REGION Network 14: ACTIVATE HANDWHEEL / ACTIVATE HANDWHEEL 1
   RUNG wire#powerrail
      I_Contact( "DB2001_MODES_GENERAL".MG1.INCREMENTAL."1_MICRA_SELECTED" )
      I_Contact( "DB2001_MODES_GENERAL".MG1.INCREMENTAL."10_MICRA_SELECTED" )
      I_Contact( "DB2001_MODES_GENERAL".MG1.INCREMENTAL."100_MICRA_SELECTED" )
      I_Contact( "DB2001_MODES_GENERAL".MG1.INCREMENTAL."1000_MICRA_SELECTED" )
      Not()
      Contact( #SP.SELECTED )
      Contact( "DB2001_MODES_GENERAL".MG1.INCREMENTAL.INCREMENTAL_MODE_SELECTED )
      Coil( #SpindleDB.A_HW1 )
   END_RUNG
   // the same network as SCL:
   #SpindleDB.A_HW1 := NOT (NOT "DB2001_MODES_GENERAL".MG1.INCREMENTAL."1_MICRA_SELECTED" AND NOT "DB2001_MODES_GENERAL".MG1.INCREMENTAL."10_MICRA_SELECTED" AND NOT "DB2001_MODES_GENERAL".MG1.INCREMENTAL."100_MICRA_SELECTED" AND NOT "DB2001_MODES_GENERAL".MG1.INCREMENTAL."1000_MICRA_SELECTED") AND #SP.SELECTED AND "DB2001_MODES_GENERAL".MG1.INCREMENTAL.INCREMENTAL_MODE_SELECTED;
END_REGION

REGION Network 15: SPINDLE INCREMENTAL MODE SELECTED
   RUNG wire#powerrail
      I_Contact( #SpindleDB.A_INC1 )
      I_Contact( #SpindleDB.A_INC10 )
      I_Contact( #SpindleDB.A_INC100 )
      I_Contact( #SpindleDB.A_INC1000 )
      Not()
      Contact( "DB2001_MODES_GENERAL".MG1.INCREMENTAL.INCREMENTAL_MODE_SELECTED )
      Coil( #SP.CONT_INCRMTL_MODE )
   END_RUNG
   // the same network as SCL:
   #SP.CONT_INCRMTL_MODE := NOT (NOT #SpindleDB.A_INC1 AND NOT #SpindleDB.A_INC10 AND NOT #SpindleDB.A_INC100 AND NOT #SpindleDB.A_INC1000) AND "DB2001_MODES_GENERAL".MG1.INCREMENTAL.INCREMENTAL_MODE_SELECTED;
END_REGION

REGION Network 16: JOG MINUS REQUEST
   RUNG wire#powerrail
      Contact( #HMI_REQ_LINE )
      Contact( "LTLP_HMIProInterfaceData".pMinus )
      wire#w1
      Coil( #SP.HMI_JOG_MINUS_RQ )
   END_RUNG
   RUNG wire#powerrail
      Contact( "DB7224_HMI_AXES".NC_AXES.SOFTKEYS.RIGHT.JOG_MINUS )
      wire#w2
      Contact( "DB2100_GENERAL".MACHINE_READY_POWER_ENABLED )
      Contact( #SP.SELECTED )
   END_RUNG wire#w1
   RUNG wire#powerrail
      Contact( "DB2122_HT10".INPUTS.JOG_MIINUS_I )
   END_RUNG wire#w2
   // the same network as SCL:
   #SP.HMI_JOG_MINUS_RQ := (#HMI_REQ_LINE AND "LTLP_HMIProInterfaceData".pMinus) OR (("DB7224_HMI_AXES".NC_AXES.SOFTKEYS.RIGHT.JOG_MINUS OR "DB2122_HT10".INPUTS.JOG_MIINUS_I) AND "DB2100_GENERAL".MACHINE_READY_POWER_ENABLED AND #SP.SELECTED);
END_REGION

REGION Network 17: JOG MINUS COMMAND
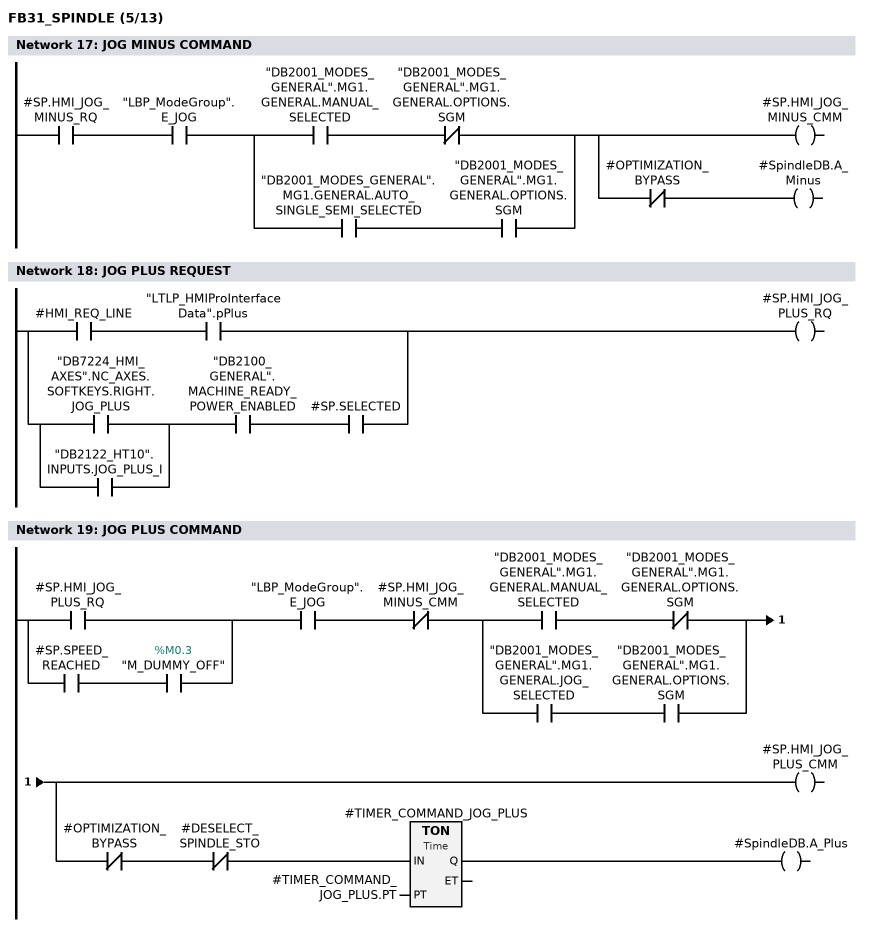
   RUNG wire#powerrail
      Contact( #SP.HMI_JOG_MINUS_RQ )
      Contact( "LBP_ModeGroup".E_JOG )
      wire#w1
      Contact( "DB2001_MODES_GENERAL".MG1.GENERAL.MANUAL_SELECTED )
      I_Contact( "DB2001_MODES_GENERAL".MG1.GENERAL.OPTIONS.SGM )
      wire#w2
      Coil( #SP.HMI_JOG_MINUS_CMM )
   END_RUNG
   RUNG wire#w1
      Contact( "DB2001_MODES_GENERAL".MG1.GENERAL.AUTO_SINGLE_SEMI_SELECTED )
      Contact( "DB2001_MODES_GENERAL".MG1.GENERAL.OPTIONS.SGM )
   END_RUNG wire#w2
   RUNG wire#w2
      I_Contact( #OPTIMIZATION_BYPASS )
      Coil( #SpindleDB.A_Minus )
   END_RUNG
   // the same network as SCL:
   #SP.HMI_JOG_MINUS_CMM := #SP.HMI_JOG_MINUS_RQ AND "LBP_ModeGroup".E_JOG AND (("DB2001_MODES_GENERAL".MG1.GENERAL.MANUAL_SELECTED AND NOT "DB2001_MODES_GENERAL".MG1.GENERAL.OPTIONS.SGM) OR ("DB2001_MODES_GENERAL".MG1.GENERAL.AUTO_SINGLE_SEMI_SELECTED AND "DB2001_MODES_GENERAL".MG1.GENERAL.OPTIONS.SGM));
   #SpindleDB.A_Minus := #SP.HMI_JOG_MINUS_CMM AND NOT #OPTIMIZATION_BYPASS;
END_REGION

REGION Network 18: JOG PLUS REQUEST
   RUNG wire#powerrail
      Contact( #HMI_REQ_LINE )
      Contact( "LTLP_HMIProInterfaceData".pPlus )
      wire#w1
      Coil( #SP.HMI_JOG_PLUS_RQ )
   END_RUNG
   RUNG wire#powerrail
      Contact( "DB7224_HMI_AXES".NC_AXES.SOFTKEYS.RIGHT.JOG_PLUS )
      wire#w2
      Contact( "DB2100_GENERAL".MACHINE_READY_POWER_ENABLED )
      Contact( #SP.SELECTED )
   END_RUNG wire#w1
   RUNG wire#powerrail
      Contact( "DB2122_HT10".INPUTS.JOG_PLUS_I )
   END_RUNG wire#w2
   // the same network as SCL:
   #SP.HMI_JOG_PLUS_RQ := (#HMI_REQ_LINE AND "LTLP_HMIProInterfaceData".pPlus) OR (("DB7224_HMI_AXES".NC_AXES.SOFTKEYS.RIGHT.JOG_PLUS OR "DB2122_HT10".INPUTS.JOG_PLUS_I) AND "DB2100_GENERAL".MACHINE_READY_POWER_ENABLED AND #SP.SELECTED);
END_REGION

REGION Network 19: JOG PLUS COMMAND
   RUNG wire#powerrail
      Contact( #SP.HMI_JOG_PLUS_RQ )
      wire#w1
      Contact( "LBP_ModeGroup".E_JOG )
      I_Contact( #SP.HMI_JOG_MINUS_CMM )
      wire#w2
      Contact( "DB2001_MODES_GENERAL".MG1.GENERAL.MANUAL_SELECTED )
      I_Contact( "DB2001_MODES_GENERAL".MG1.GENERAL.OPTIONS.SGM )
      wire#w3
      Coil( #SP.HMI_JOG_PLUS_CMM )
   END_RUNG
   RUNG wire#powerrail
      Contact( #SP.SPEED_REACHED )
      Contact( "M_DUMMY_OFF" )
   END_RUNG wire#w1
   RUNG wire#w2
      Contact( "DB2001_MODES_GENERAL".MG1.GENERAL.JOG_SELECTED )
      Contact( "DB2001_MODES_GENERAL".MG1.GENERAL.OPTIONS.SGM )
   END_RUNG wire#w3
   RUNG wire#w3
      I_Contact( #OPTIMIZATION_BYPASS )
      I_Contact( #DESELECT_SPINDLE_STO )
      { S7_Templates := "time_type := Time" } #TIMER_COMMAND_JOG_PLUS.TON(pt := #TIMER_COMMAND_JOG_PLUS.PT, et =>)
      Coil( #SpindleDB.A_Plus )
   END_RUNG
   // the same network as SCL:
   #SP.HMI_JOG_PLUS_CMM := (#SP.HMI_JOG_PLUS_RQ OR (#SP.SPEED_REACHED AND "M_DUMMY_OFF")) AND "LBP_ModeGroup".E_JOG AND NOT #SP.HMI_JOG_MINUS_CMM AND (("DB2001_MODES_GENERAL".MG1.GENERAL.MANUAL_SELECTED AND NOT "DB2001_MODES_GENERAL".MG1.GENERAL.OPTIONS.SGM) OR ("DB2001_MODES_GENERAL".MG1.GENERAL.JOG_SELECTED AND "DB2001_MODES_GENERAL".MG1.GENERAL.OPTIONS.SGM));
   #TIMER_COMMAND_JOG_PLUS(IN := #SP.HMI_JOG_PLUS_CMM AND NOT #OPTIMIZATION_BYPASS AND NOT #DESELECT_SPINDLE_STO,   // TON
                           PT := #TIMER_COMMAND_JOG_PLUS.PT);
   #SpindleDB.A_Plus := #TIMER_COMMAND_JOG_PLUS.Q;
END_REGION

REGION Network 20: OVERRIDE / FEED OVERRIDE
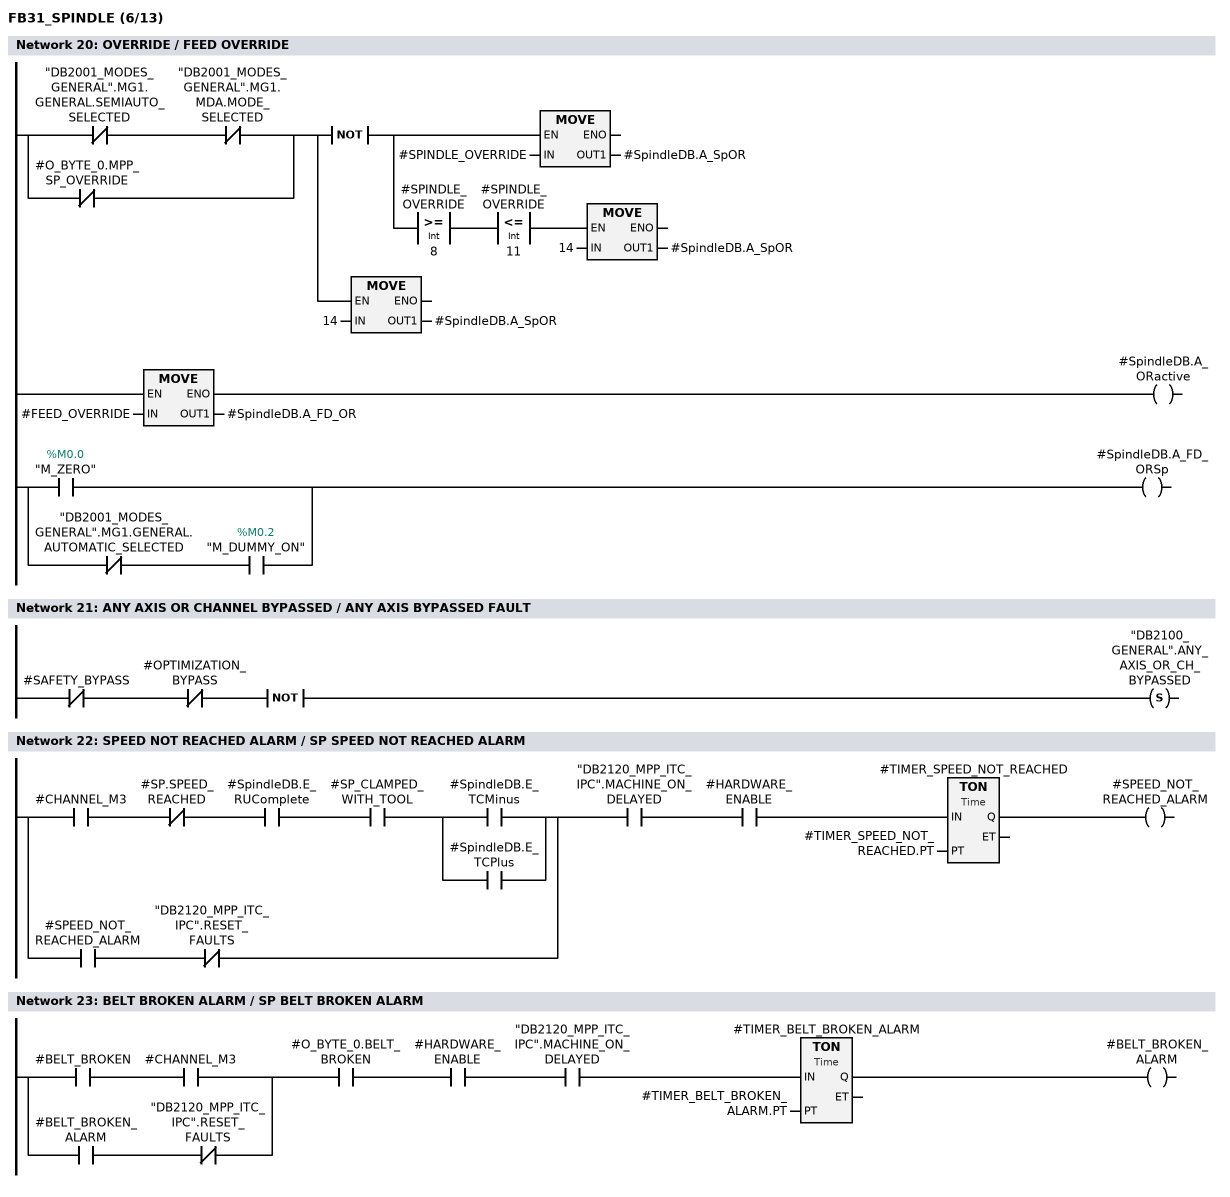
   RUNG wire#powerrail
      I_Contact( "DB2001_MODES_GENERAL".MG1.GENERAL.SEMIAUTO_SELECTED )
      I_Contact( "DB2001_MODES_GENERAL".MG1.MDA.MODE_SELECTED )
      wire#w1
      Not()
      wire#w2
      { S7_GenerateENO := "TRUE" } Move(in := #SPINDLE_OVERRIDE, out1 => #SpindleDB.A_SpOR)
   END_RUNG
   RUNG wire#powerrail
      I_Contact( #O_BYTE_0.MPP_SP_OVERRIDE )
   END_RUNG wire#w1
   RUNG wire#w2
      { S7_Templates := "SrcType := Int" } GE_Contact(in1 := #SPINDLE_OVERRIDE, in2 := 8)
      { S7_Templates := "SrcType := Int" } LE_Contact(in1 := #SPINDLE_OVERRIDE, in2 := 11)
      { S7_GenerateENO := "TRUE" } Move(in := 14, out1 => #SpindleDB.A_SpOR)
   END_RUNG
   RUNG wire#w1
      { S7_GenerateENO := "TRUE" } Move(in := 14, out1 => #SpindleDB.A_SpOR)
   END_RUNG
   RUNG wire#powerrail
      { S7_GenerateENO := "TRUE" } Move(in := #FEED_OVERRIDE, out1 => #SpindleDB.A_FD_OR)
      Coil( #SpindleDB.A_ORactive )
   END_RUNG
   RUNG wire#powerrail
      Contact( "M_ZERO" )
      wire#w3
      Coil( #SpindleDB.A_FD_ORSp )
   END_RUNG
   RUNG wire#powerrail
      I_Contact( "DB2001_MODES_GENERAL".MG1.GENERAL.AUTOMATIC_SELECTED )
      Contact( "M_DUMMY_ON" )
   END_RUNG wire#w3
   // the same network as SCL:
   // ENO of a box is taken as its EN; it also drops when the box reports an error
   #_w1 := (NOT "DB2001_MODES_GENERAL".MG1.GENERAL.SEMIAUTO_SELECTED AND NOT "DB2001_MODES_GENERAL".MG1.MDA.MODE_SELECTED) OR NOT #O_BYTE_0.MPP_SP_OVERRIDE;
   IF NOT #_w1 THEN #SpindleDB.A_SpOR := #SPINDLE_OVERRIDE; END_IF;
   IF NOT #_w1 AND (#SPINDLE_OVERRIDE >= 8) AND (#SPINDLE_OVERRIDE <= 11) THEN
       #SpindleDB.A_SpOR := 14;
   END_IF;
   IF #_w1 THEN #SpindleDB.A_SpOR := 14; END_IF;
   #SpindleDB.A_FD_OR := #FEED_OVERRIDE;
   #SpindleDB.A_ORactive := TRUE;
   #SpindleDB.A_FD_ORSp := "M_ZERO" OR (NOT "DB2001_MODES_GENERAL".MG1.GENERAL.AUTOMATIC_SELECTED AND "M_DUMMY_ON");
END_REGION

REGION Network 21: ANY AXIS OR CHANNEL BYPASSED / ANY AXIS BYPASSED FAULT
   RUNG wire#powerrail
      I_Contact( #SAFETY_BYPASS )
      I_Contact( #OPTIMIZATION_BYPASS )
      Not()
      S_Coil( "DB2100_GENERAL".ANY_AXIS_OR_CH_BYPASSED )
   END_RUNG
   // the same network as SCL:
   IF NOT (NOT #SAFETY_BYPASS AND NOT #OPTIMIZATION_BYPASS) THEN
       "DB2100_GENERAL".ANY_AXIS_OR_CH_BYPASSED := TRUE;
   END_IF;
END_REGION

REGION Network 22: SPEED NOT REACHED ALARM / SP SPEED NOT REACHED ALARM
   RUNG wire#powerrail
      Contact( #CHANNEL_M3 )
      I_Contact( #SP.SPEED_REACHED )
      Contact( #SpindleDB.E_RUComplete )
      Contact( #SP_CLAMPED_WITH_TOOL )
      wire#w1
      Contact( #SpindleDB.E_TCMinus )
      wire#w2
      Contact( "DB2120_MPP_ITC_IPC".MACHINE_ON_DELAYED )
      Contact( #HARDWARE_ENABLE )
      { S7_Templates := "time_type := Time" } #TIMER_SPEED_NOT_REACHED.TON(pt := #TIMER_SPEED_NOT_REACHED.PT, et =>)
      Coil( #SPEED_NOT_REACHED_ALARM )
   END_RUNG
   RUNG wire#w1
      Contact( #SpindleDB.E_TCPlus )
   END_RUNG wire#w2
   RUNG wire#powerrail
      Contact( #SPEED_NOT_REACHED_ALARM )
      I_Contact( "DB2120_MPP_ITC_IPC".RESET_FAULTS )
   END_RUNG wire#w2
   // the same network as SCL:
   #TIMER_SPEED_NOT_REACHED(IN := ((#CHANNEL_M3 AND NOT #SP.SPEED_REACHED AND #SpindleDB.E_RUComplete AND #SP_CLAMPED_WITH_TOOL AND (#SpindleDB.E_TCMinus OR #SpindleDB.E_TCPlus)) OR (#SPEED_NOT_REACHED_ALARM AND NOT "DB2120_MPP_ITC_IPC".RESET_FAULTS)) AND "DB2120_MPP_ITC_IPC".MACHINE_ON_DELAYED AND #HARDWARE_ENABLE,   // TON
                           PT := #TIMER_SPEED_NOT_REACHED.PT);
   #SPEED_NOT_REACHED_ALARM := #TIMER_SPEED_NOT_REACHED.Q;
END_REGION

REGION Network 23: BELT BROKEN ALARM / SP BELT BROKEN ALARM
   RUNG wire#powerrail
      Contact( #BELT_BROKEN )
      Contact( #CHANNEL_M3 )
      wire#w1
      Contact( #O_BYTE_0.BELT_BROKEN )
      Contact( #HARDWARE_ENABLE )
      Contact( "DB2120_MPP_ITC_IPC".MACHINE_ON_DELAYED )
      { S7_Templates := "time_type := Time" } #TIMER_BELT_BROKEN_ALARM.TON(pt := #TIMER_BELT_BROKEN_ALARM.PT, et =>)
      Coil( #BELT_BROKEN_ALARM )
   END_RUNG
   RUNG wire#powerrail
      Contact( #BELT_BROKEN_ALARM )
      I_Contact( "DB2120_MPP_ITC_IPC".RESET_FAULTS )
   END_RUNG wire#w1
   // the same network as SCL:
   #TIMER_BELT_BROKEN_ALARM(IN := ((#BELT_BROKEN AND #CHANNEL_M3) OR (#BELT_BROKEN_ALARM AND NOT "DB2120_MPP_ITC_IPC".RESET_FAULTS)) AND #O_BYTE_0.BELT_BROKEN AND #HARDWARE_ENABLE AND "DB2120_MPP_ITC_IPC".MACHINE_ON_DELAYED,   // TON
                           PT := #TIMER_BELT_BROKEN_ALARM.PT);
   #BELT_BROKEN_ALARM := #TIMER_BELT_BROKEN_ALARM.Q;
END_REGION

REGION Network 24: COOLING ALARM / SP COOLING ALARM
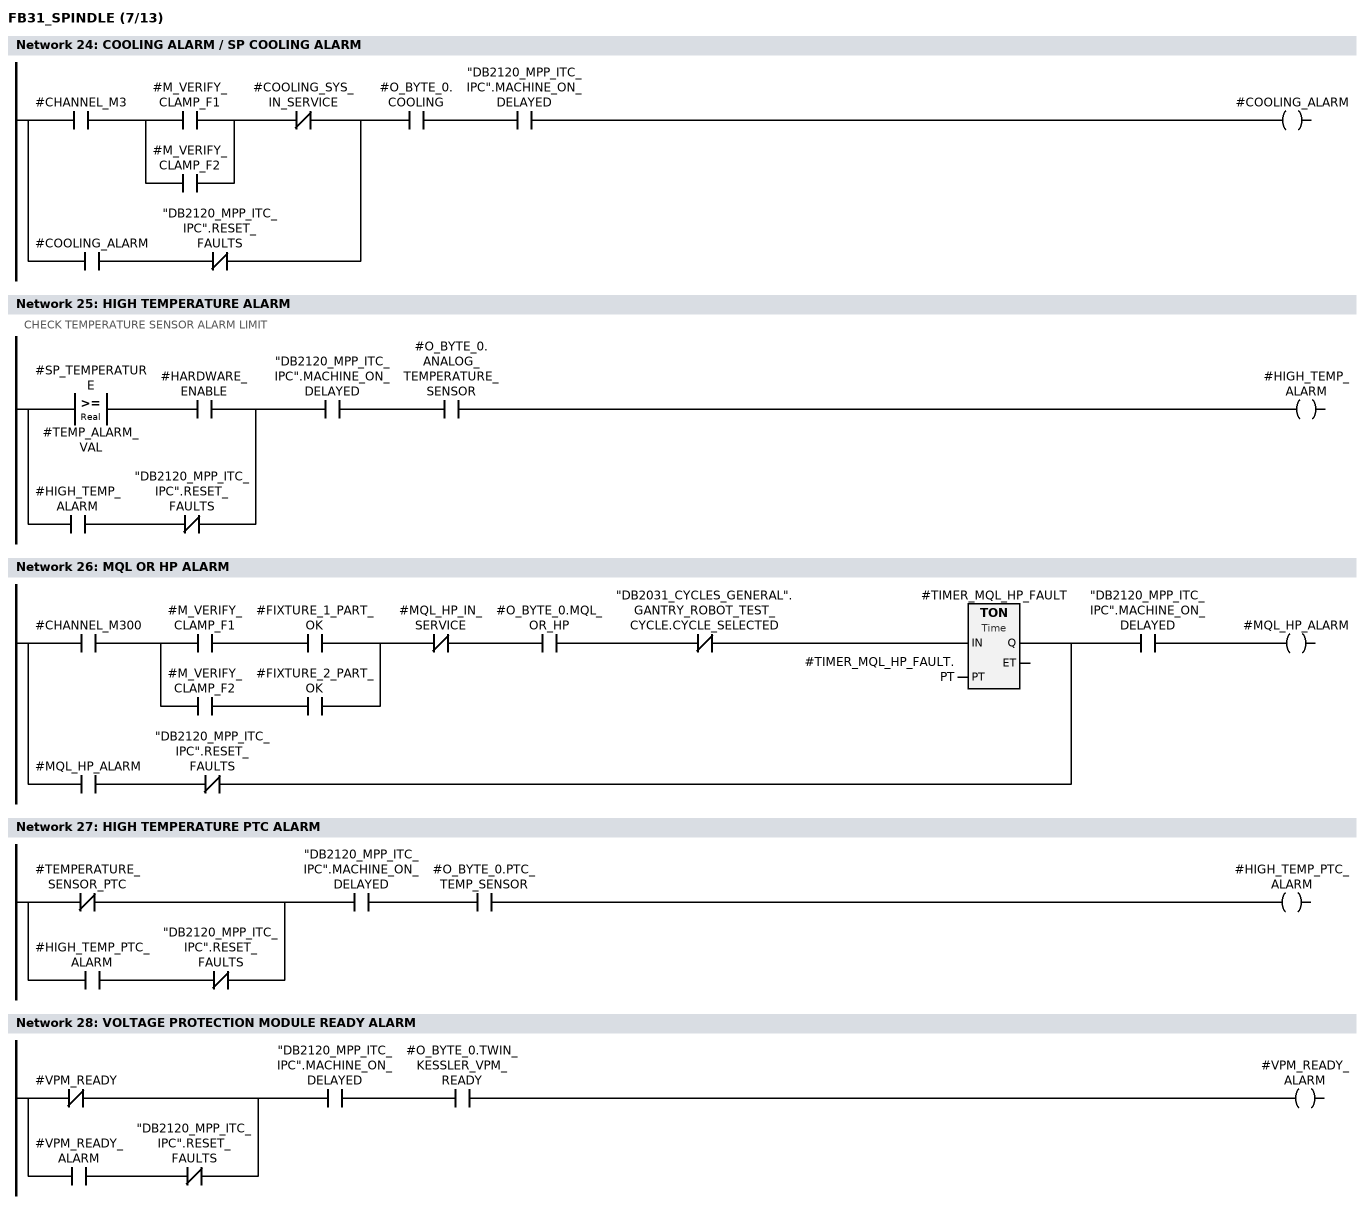
   RUNG wire#powerrail
      Contact( #CHANNEL_M3 )
      wire#w1
      Contact( #M_VERIFY_CLAMP_F1 )
      wire#w2
      I_Contact( #COOLING_SYS_IN_SERVICE )
      wire#w3
      Contact( #O_BYTE_0.COOLING )
      Contact( "DB2120_MPP_ITC_IPC".MACHINE_ON_DELAYED )
      Coil( #COOLING_ALARM )
   END_RUNG
   RUNG wire#w1
      Contact( #M_VERIFY_CLAMP_F2 )
   END_RUNG wire#w2
   RUNG wire#powerrail
      Contact( #COOLING_ALARM )
      I_Contact( "DB2120_MPP_ITC_IPC".RESET_FAULTS )
   END_RUNG wire#w3
   // the same network as SCL:
   #COOLING_ALARM := ((#CHANNEL_M3 AND (#M_VERIFY_CLAMP_F1 OR #M_VERIFY_CLAMP_F2) AND NOT #COOLING_SYS_IN_SERVICE) OR (#COOLING_ALARM AND NOT "DB2120_MPP_ITC_IPC".RESET_FAULTS)) AND #O_BYTE_0.COOLING AND "DB2120_MPP_ITC_IPC".MACHINE_ON_DELAYED;
END_REGION

REGION Network 25: HIGH TEMPERATURE ALARM
   // CHECK TEMPERATURE SENSOR ALARM LIMIT
   RUNG wire#powerrail
      { S7_Templates := "SrcType := Real" } GE_Contact(in1 := #SP_TEMPERATURE, in2 := #TEMP_ALARM_VAL)
      Contact( #HARDWARE_ENABLE )
      wire#w1
      Contact( "DB2120_MPP_ITC_IPC".MACHINE_ON_DELAYED )
      Contact( #O_BYTE_0.ANALOG_TEMPERATURE_SENSOR )
      Coil( #HIGH_TEMP_ALARM )
   END_RUNG
   RUNG wire#powerrail
      Contact( #HIGH_TEMP_ALARM )
      I_Contact( "DB2120_MPP_ITC_IPC".RESET_FAULTS )
   END_RUNG wire#w1
   // the same network as SCL:
   #HIGH_TEMP_ALARM := (((#SP_TEMPERATURE >= #TEMP_ALARM_VAL) AND #HARDWARE_ENABLE) OR (#HIGH_TEMP_ALARM AND NOT "DB2120_MPP_ITC_IPC".RESET_FAULTS)) AND "DB2120_MPP_ITC_IPC".MACHINE_ON_DELAYED AND #O_BYTE_0.ANALOG_TEMPERATURE_SENSOR;
END_REGION

REGION Network 26: MQL OR HP ALARM
   RUNG wire#powerrail
      Contact( #CHANNEL_M300 )
      wire#w1
      Contact( #M_VERIFY_CLAMP_F1 )
      Contact( #FIXTURE_1_PART_OK )
      wire#w2
      I_Contact( #MQL_HP_IN_SERVICE )
      Contact( #O_BYTE_0.MQL_OR_HP )
      I_Contact( "DB2031_CYCLES_GENERAL".GANTRY_ROBOT_TEST_CYCLE.CYCLE_SELECTED )
      { S7_Templates := "time_type := Time" } #TIMER_MQL_HP_FAULT.TON(pt := #TIMER_MQL_HP_FAULT.PT, et =>)
      wire#w3
      Contact( "DB2120_MPP_ITC_IPC".MACHINE_ON_DELAYED )
      Coil( #MQL_HP_ALARM )
   END_RUNG
   RUNG wire#w1
      Contact( #M_VERIFY_CLAMP_F2 )
      Contact( #FIXTURE_2_PART_OK )
   END_RUNG wire#w2
   RUNG wire#powerrail
      Contact( #MQL_HP_ALARM )
      I_Contact( "DB2120_MPP_ITC_IPC".RESET_FAULTS )
   END_RUNG wire#w3
   // the same network as SCL:
   #TIMER_MQL_HP_FAULT(IN := #CHANNEL_M300 AND ((#M_VERIFY_CLAMP_F1 AND #FIXTURE_1_PART_OK) OR (#M_VERIFY_CLAMP_F2 AND #FIXTURE_2_PART_OK)) AND NOT #MQL_HP_IN_SERVICE AND #O_BYTE_0.MQL_OR_HP AND NOT "DB2031_CYCLES_GENERAL".GANTRY_ROBOT_TEST_CYCLE.CYCLE_SELECTED,   // TON
                       PT := #TIMER_MQL_HP_FAULT.PT);
   #MQL_HP_ALARM := (#TIMER_MQL_HP_FAULT.Q OR (#MQL_HP_ALARM AND NOT "DB2120_MPP_ITC_IPC".RESET_FAULTS)) AND "DB2120_MPP_ITC_IPC".MACHINE_ON_DELAYED;
END_REGION

REGION Network 27: HIGH TEMPERATURE PTC ALARM
   RUNG wire#powerrail
      I_Contact( #TEMPERATURE_SENSOR_PTC )
      wire#w1
      Contact( "DB2120_MPP_ITC_IPC".MACHINE_ON_DELAYED )
      Contact( #O_BYTE_0.PTC_TEMP_SENSOR )
      Coil( #HIGH_TEMP_PTC_ALARM )
   END_RUNG
   RUNG wire#powerrail
      Contact( #HIGH_TEMP_PTC_ALARM )
      I_Contact( "DB2120_MPP_ITC_IPC".RESET_FAULTS )
   END_RUNG wire#w1
   // the same network as SCL:
   #HIGH_TEMP_PTC_ALARM := (NOT #TEMPERATURE_SENSOR_PTC OR (#HIGH_TEMP_PTC_ALARM AND NOT "DB2120_MPP_ITC_IPC".RESET_FAULTS)) AND "DB2120_MPP_ITC_IPC".MACHINE_ON_DELAYED AND #O_BYTE_0.PTC_TEMP_SENSOR;
END_REGION

REGION Network 28: VOLTAGE PROTECTION MODULE READY ALARM
   RUNG wire#powerrail
      I_Contact( #VPM_READY )
      wire#w1
      Contact( "DB2120_MPP_ITC_IPC".MACHINE_ON_DELAYED )
      Contact( #O_BYTE_0.TWIN_KESSLER_VPM_READY )
      Coil( #VPM_READY_ALARM )
   END_RUNG
   RUNG wire#powerrail
      Contact( #VPM_READY_ALARM )
      I_Contact( "DB2120_MPP_ITC_IPC".RESET_FAULTS )
   END_RUNG wire#w1
   // the same network as SCL:
   #VPM_READY_ALARM := (NOT #VPM_READY OR (#VPM_READY_ALARM AND NOT "DB2120_MPP_ITC_IPC".RESET_FAULTS)) AND "DB2120_MPP_ITC_IPC".MACHINE_ON_DELAYED AND #O_BYTE_0.TWIN_KESSLER_VPM_READY;
END_REGION

REGION Network 29: RETURN HOME POSITION AND STOP END OF CYCLE ALARMS / RHP&SEOC ALARMS
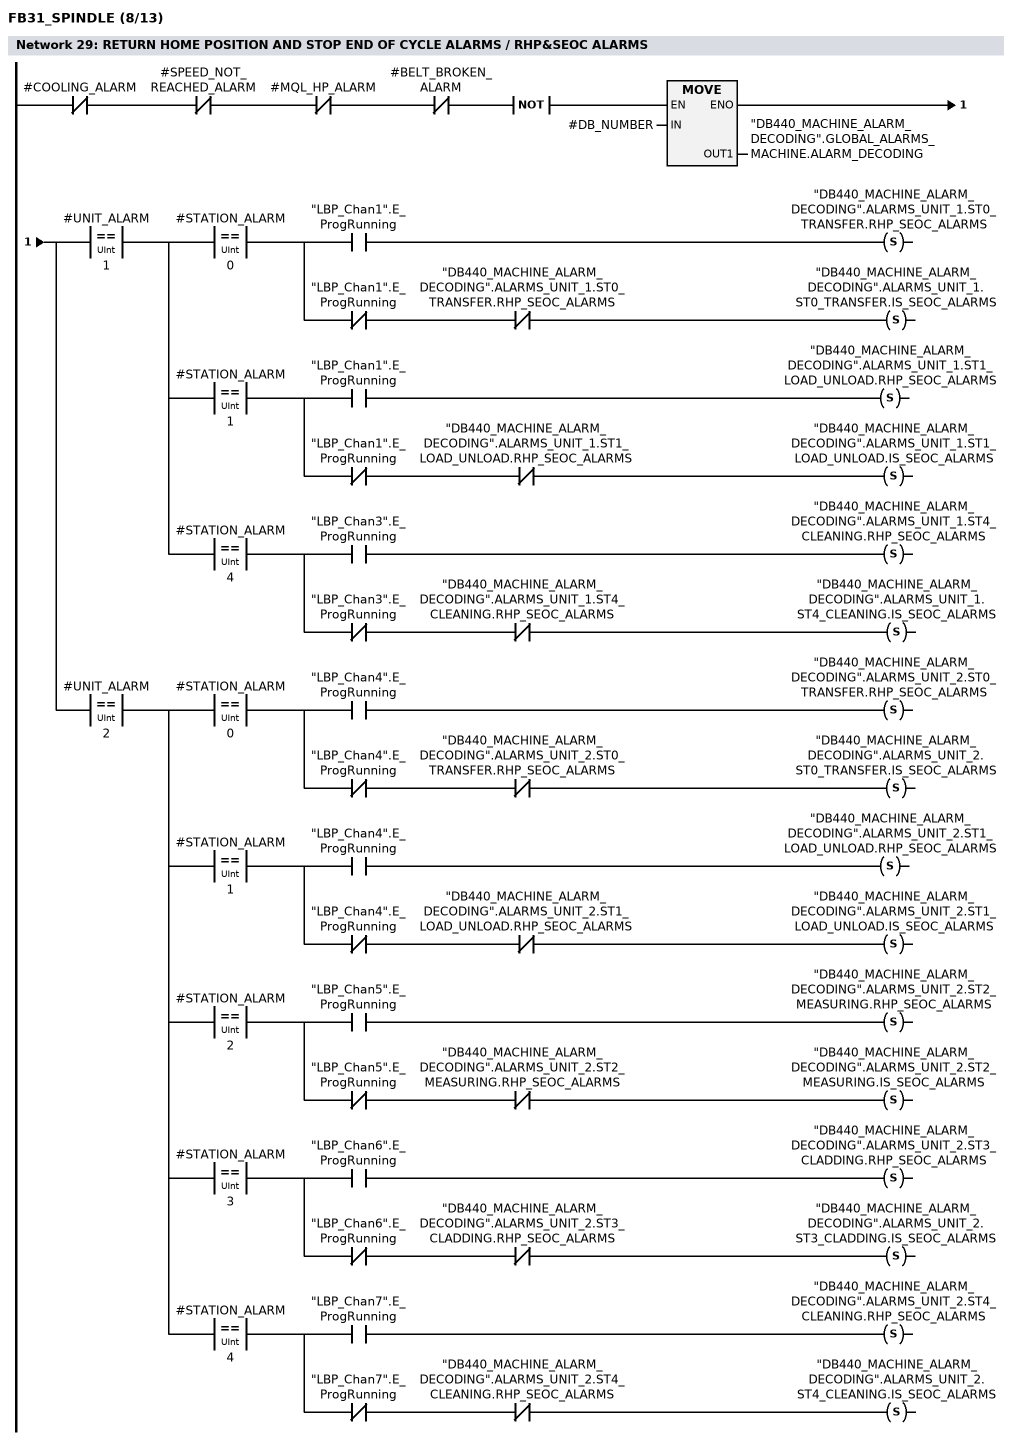
   RUNG wire#powerrail
      I_Contact( #COOLING_ALARM )
      I_Contact( #SPEED_NOT_REACHED_ALARM )
      I_Contact( #MQL_HP_ALARM )
      I_Contact( #BELT_BROKEN_ALARM )
      Not()
      { S7_GenerateENO := "TRUE" } Move(in := #DB_NUMBER, out1 => "DB440_MACHINE_ALARM_DECODING".GLOBAL_ALARMS_MACHINE.ALARM_DECODING)
      wire#w1
      { S7_Templates := "SrcType := UInt" } EQ_Contact(in1 := #UNIT_ALARM, in2 := 1)
      wire#w2
      { S7_Templates := "SrcType := UInt" } EQ_Contact(in1 := #STATION_ALARM, in2 := 0)
      wire#w3
      Contact( "LBP_Chan1".E_ProgRunning )
      S_Coil( "DB440_MACHINE_ALARM_DECODING".ALARMS_UNIT_1.ST0_TRANSFER.RHP_SEOC_ALARMS )
   END_RUNG
   RUNG wire#w3
      I_Contact( "LBP_Chan1".E_ProgRunning )
      I_Contact( "DB440_MACHINE_ALARM_DECODING".ALARMS_UNIT_1.ST0_TRANSFER.RHP_SEOC_ALARMS )
      S_Coil( "DB440_MACHINE_ALARM_DECODING".ALARMS_UNIT_1.ST0_TRANSFER.IS_SEOC_ALARMS )
   END_RUNG
   RUNG wire#w2
      { S7_Templates := "SrcType := UInt" } EQ_Contact(in1 := #STATION_ALARM, in2 := 1)
      wire#w4
      Contact( "LBP_Chan1".E_ProgRunning )
      S_Coil( "DB440_MACHINE_ALARM_DECODING".ALARMS_UNIT_1.ST1_LOAD_UNLOAD.RHP_SEOC_ALARMS )
   END_RUNG
   RUNG wire#w4
      I_Contact( "LBP_Chan1".E_ProgRunning )
      I_Contact( "DB440_MACHINE_ALARM_DECODING".ALARMS_UNIT_1.ST1_LOAD_UNLOAD.RHP_SEOC_ALARMS )
      S_Coil( "DB440_MACHINE_ALARM_DECODING".ALARMS_UNIT_1.ST1_LOAD_UNLOAD.IS_SEOC_ALARMS )
   END_RUNG
   RUNG wire#w2
      { S7_Templates := "SrcType := UInt" } EQ_Contact(in1 := #STATION_ALARM, in2 := 4)
      wire#w5
      Contact( "LBP_Chan3".E_ProgRunning )
      S_Coil( "DB440_MACHINE_ALARM_DECODING".ALARMS_UNIT_1.ST4_CLEANING.RHP_SEOC_ALARMS )
   END_RUNG
   RUNG wire#w5
      I_Contact( "LBP_Chan3".E_ProgRunning )
      I_Contact( "DB440_MACHINE_ALARM_DECODING".ALARMS_UNIT_1.ST4_CLEANING.RHP_SEOC_ALARMS )
      S_Coil( "DB440_MACHINE_ALARM_DECODING".ALARMS_UNIT_1.ST4_CLEANING.IS_SEOC_ALARMS )
   END_RUNG
   RUNG wire#w1
      { S7_Templates := "SrcType := UInt" } EQ_Contact(in1 := #UNIT_ALARM, in2 := 2)
      wire#w6
      { S7_Templates := "SrcType := UInt" } EQ_Contact(in1 := #STATION_ALARM, in2 := 0)
      wire#w7
      Contact( "LBP_Chan4".E_ProgRunning )
      S_Coil( "DB440_MACHINE_ALARM_DECODING".ALARMS_UNIT_2.ST0_TRANSFER.RHP_SEOC_ALARMS )
   END_RUNG
   RUNG wire#w7
      I_Contact( "LBP_Chan4".E_ProgRunning )
      I_Contact( "DB440_MACHINE_ALARM_DECODING".ALARMS_UNIT_2.ST0_TRANSFER.RHP_SEOC_ALARMS )
      S_Coil( "DB440_MACHINE_ALARM_DECODING".ALARMS_UNIT_2.ST0_TRANSFER.IS_SEOC_ALARMS )
   END_RUNG
   RUNG wire#w6
      { S7_Templates := "SrcType := UInt" } EQ_Contact(in1 := #STATION_ALARM, in2 := 1)
      wire#w8
      Contact( "LBP_Chan4".E_ProgRunning )
      S_Coil( "DB440_MACHINE_ALARM_DECODING".ALARMS_UNIT_2.ST1_LOAD_UNLOAD.RHP_SEOC_ALARMS )
   END_RUNG
   RUNG wire#w8
      I_Contact( "LBP_Chan4".E_ProgRunning )
      I_Contact( "DB440_MACHINE_ALARM_DECODING".ALARMS_UNIT_2.ST1_LOAD_UNLOAD.RHP_SEOC_ALARMS )
      S_Coil( "DB440_MACHINE_ALARM_DECODING".ALARMS_UNIT_2.ST1_LOAD_UNLOAD.IS_SEOC_ALARMS )
   END_RUNG
   RUNG wire#w6
      { S7_Templates := "SrcType := UInt" } EQ_Contact(in1 := #STATION_ALARM, in2 := 2)
      wire#w9
      Contact( "LBP_Chan5".E_ProgRunning )
      S_Coil( "DB440_MACHINE_ALARM_DECODING".ALARMS_UNIT_2.ST2_MEASURING.RHP_SEOC_ALARMS )
   END_RUNG
   RUNG wire#w9
      I_Contact( "LBP_Chan5".E_ProgRunning )
      I_Contact( "DB440_MACHINE_ALARM_DECODING".ALARMS_UNIT_2.ST2_MEASURING.RHP_SEOC_ALARMS )
      S_Coil( "DB440_MACHINE_ALARM_DECODING".ALARMS_UNIT_2.ST2_MEASURING.IS_SEOC_ALARMS )
   END_RUNG
   RUNG wire#w6
      { S7_Templates := "SrcType := UInt" } EQ_Contact(in1 := #STATION_ALARM, in2 := 3)
      wire#w10
      Contact( "LBP_Chan6".E_ProgRunning )
      S_Coil( "DB440_MACHINE_ALARM_DECODING".ALARMS_UNIT_2.ST3_CLADDING.RHP_SEOC_ALARMS )
   END_RUNG
   RUNG wire#w10
      I_Contact( "LBP_Chan6".E_ProgRunning )
      I_Contact( "DB440_MACHINE_ALARM_DECODING".ALARMS_UNIT_2.ST3_CLADDING.RHP_SEOC_ALARMS )
      S_Coil( "DB440_MACHINE_ALARM_DECODING".ALARMS_UNIT_2.ST3_CLADDING.IS_SEOC_ALARMS )
   END_RUNG
   RUNG wire#w6
      { S7_Templates := "SrcType := UInt" } EQ_Contact(in1 := #STATION_ALARM, in2 := 4)
      wire#w11
      Contact( "LBP_Chan7".E_ProgRunning )
      S_Coil( "DB440_MACHINE_ALARM_DECODING".ALARMS_UNIT_2.ST4_CLEANING.RHP_SEOC_ALARMS )
   END_RUNG
   RUNG wire#w11
      I_Contact( "LBP_Chan7".E_ProgRunning )
      I_Contact( "DB440_MACHINE_ALARM_DECODING".ALARMS_UNIT_2.ST4_CLEANING.RHP_SEOC_ALARMS )
      S_Coil( "DB440_MACHINE_ALARM_DECODING".ALARMS_UNIT_2.ST4_CLEANING.IS_SEOC_ALARMS )
   END_RUNG
   // the same network as SCL:
   // ENO of a box is taken as its EN; it also drops when the box reports an error
   #_w1 := NOT (NOT #COOLING_ALARM AND NOT #SPEED_NOT_REACHED_ALARM AND NOT #MQL_HP_ALARM AND NOT #BELT_BROKEN_ALARM);
   IF #_w1 THEN "DB440_MACHINE_ALARM_DECODING".GLOBAL_ALARMS_MACHINE.ALARM_DECODING := #DB_NUMBER; END_IF;
   #_w2 := #_w1 AND (#UNIT_ALARM = 1);
   #_w3 := #_w2 AND (#STATION_ALARM = 0);
   IF #_w3 AND "LBP_Chan1".E_ProgRunning THEN
       "DB440_MACHINE_ALARM_DECODING".ALARMS_UNIT_1.ST0_TRANSFER.RHP_SEOC_ALARMS := TRUE;
   END_IF;
   IF #_w3 AND NOT "LBP_Chan1".E_ProgRunning AND NOT "DB440_MACHINE_ALARM_DECODING".ALARMS_UNIT_1.ST0_TRANSFER.RHP_SEOC_ALARMS THEN
       "DB440_MACHINE_ALARM_DECODING".ALARMS_UNIT_1.ST0_TRANSFER.IS_SEOC_ALARMS := TRUE;
   END_IF;
   #_w4 := #_w2 AND (#STATION_ALARM = 1);
   IF #_w4 AND "LBP_Chan1".E_ProgRunning THEN
       "DB440_MACHINE_ALARM_DECODING".ALARMS_UNIT_1.ST1_LOAD_UNLOAD.RHP_SEOC_ALARMS := TRUE;
   END_IF;
   IF #_w4 AND NOT "LBP_Chan1".E_ProgRunning AND NOT "DB440_MACHINE_ALARM_DECODING".ALARMS_UNIT_1.ST1_LOAD_UNLOAD.RHP_SEOC_ALARMS THEN
       "DB440_MACHINE_ALARM_DECODING".ALARMS_UNIT_1.ST1_LOAD_UNLOAD.IS_SEOC_ALARMS := TRUE;
   END_IF;
   #_w5 := #_w2 AND (#STATION_ALARM = 4);
   IF #_w5 AND "LBP_Chan3".E_ProgRunning THEN
       "DB440_MACHINE_ALARM_DECODING".ALARMS_UNIT_1.ST4_CLEANING.RHP_SEOC_ALARMS := TRUE;
   END_IF;
   IF #_w5 AND NOT "LBP_Chan3".E_ProgRunning AND NOT "DB440_MACHINE_ALARM_DECODING".ALARMS_UNIT_1.ST4_CLEANING.RHP_SEOC_ALARMS THEN
       "DB440_MACHINE_ALARM_DECODING".ALARMS_UNIT_1.ST4_CLEANING.IS_SEOC_ALARMS := TRUE;
   END_IF;
   #_w6 := #_w1 AND (#UNIT_ALARM = 2);
   #_w7 := #_w6 AND (#STATION_ALARM = 0);
   IF #_w7 AND "LBP_Chan4".E_ProgRunning THEN
       "DB440_MACHINE_ALARM_DECODING".ALARMS_UNIT_2.ST0_TRANSFER.RHP_SEOC_ALARMS := TRUE;
   END_IF;
   IF #_w7 AND NOT "LBP_Chan4".E_ProgRunning AND NOT "DB440_MACHINE_ALARM_DECODING".ALARMS_UNIT_2.ST0_TRANSFER.RHP_SEOC_ALARMS THEN
       "DB440_MACHINE_ALARM_DECODING".ALARMS_UNIT_2.ST0_TRANSFER.IS_SEOC_ALARMS := TRUE;
   END_IF;
   #_w8 := #_w6 AND (#STATION_ALARM = 1);
   IF #_w8 AND "LBP_Chan4".E_ProgRunning THEN
       "DB440_MACHINE_ALARM_DECODING".ALARMS_UNIT_2.ST1_LOAD_UNLOAD.RHP_SEOC_ALARMS := TRUE;
   END_IF;
   IF #_w8 AND NOT "LBP_Chan4".E_ProgRunning AND NOT "DB440_MACHINE_ALARM_DECODING".ALARMS_UNIT_2.ST1_LOAD_UNLOAD.RHP_SEOC_ALARMS THEN
       "DB440_MACHINE_ALARM_DECODING".ALARMS_UNIT_2.ST1_LOAD_UNLOAD.IS_SEOC_ALARMS := TRUE;
   END_IF;
   #_w9 := #_w6 AND (#STATION_ALARM = 2);
   IF #_w9 AND "LBP_Chan5".E_ProgRunning THEN
       "DB440_MACHINE_ALARM_DECODING".ALARMS_UNIT_2.ST2_MEASURING.RHP_SEOC_ALARMS := TRUE;
   END_IF;
   IF #_w9 AND NOT "LBP_Chan5".E_ProgRunning AND NOT "DB440_MACHINE_ALARM_DECODING".ALARMS_UNIT_2.ST2_MEASURING.RHP_SEOC_ALARMS THEN
       "DB440_MACHINE_ALARM_DECODING".ALARMS_UNIT_2.ST2_MEASURING.IS_SEOC_ALARMS := TRUE;
   END_IF;
   #_w10 := #_w6 AND (#STATION_ALARM = 3);
   IF #_w10 AND "LBP_Chan6".E_ProgRunning THEN
       "DB440_MACHINE_ALARM_DECODING".ALARMS_UNIT_2.ST3_CLADDING.RHP_SEOC_ALARMS := TRUE;
   END_IF;
   IF #_w10 AND NOT "LBP_Chan6".E_ProgRunning AND NOT "DB440_MACHINE_ALARM_DECODING".ALARMS_UNIT_2.ST3_CLADDING.RHP_SEOC_ALARMS THEN
       "DB440_MACHINE_ALARM_DECODING".ALARMS_UNIT_2.ST3_CLADDING.IS_SEOC_ALARMS := TRUE;
   END_IF;
   #_w11 := #_w6 AND (#STATION_ALARM = 4);
   IF #_w11 AND "LBP_Chan7".E_ProgRunning THEN
       "DB440_MACHINE_ALARM_DECODING".ALARMS_UNIT_2.ST4_CLEANING.RHP_SEOC_ALARMS := TRUE;
   END_IF;
   IF #_w11 AND NOT "LBP_Chan7".E_ProgRunning AND NOT "DB440_MACHINE_ALARM_DECODING".ALARMS_UNIT_2.ST4_CLEANING.RHP_SEOC_ALARMS THEN
       "DB440_MACHINE_ALARM_DECODING".ALARMS_UNIT_2.ST4_CLEANING.IS_SEOC_ALARMS := TRUE;
   END_IF;
END_REGION

REGION Network 30: STOP END OF CYCLE ALARMS / SEOC ALARMS
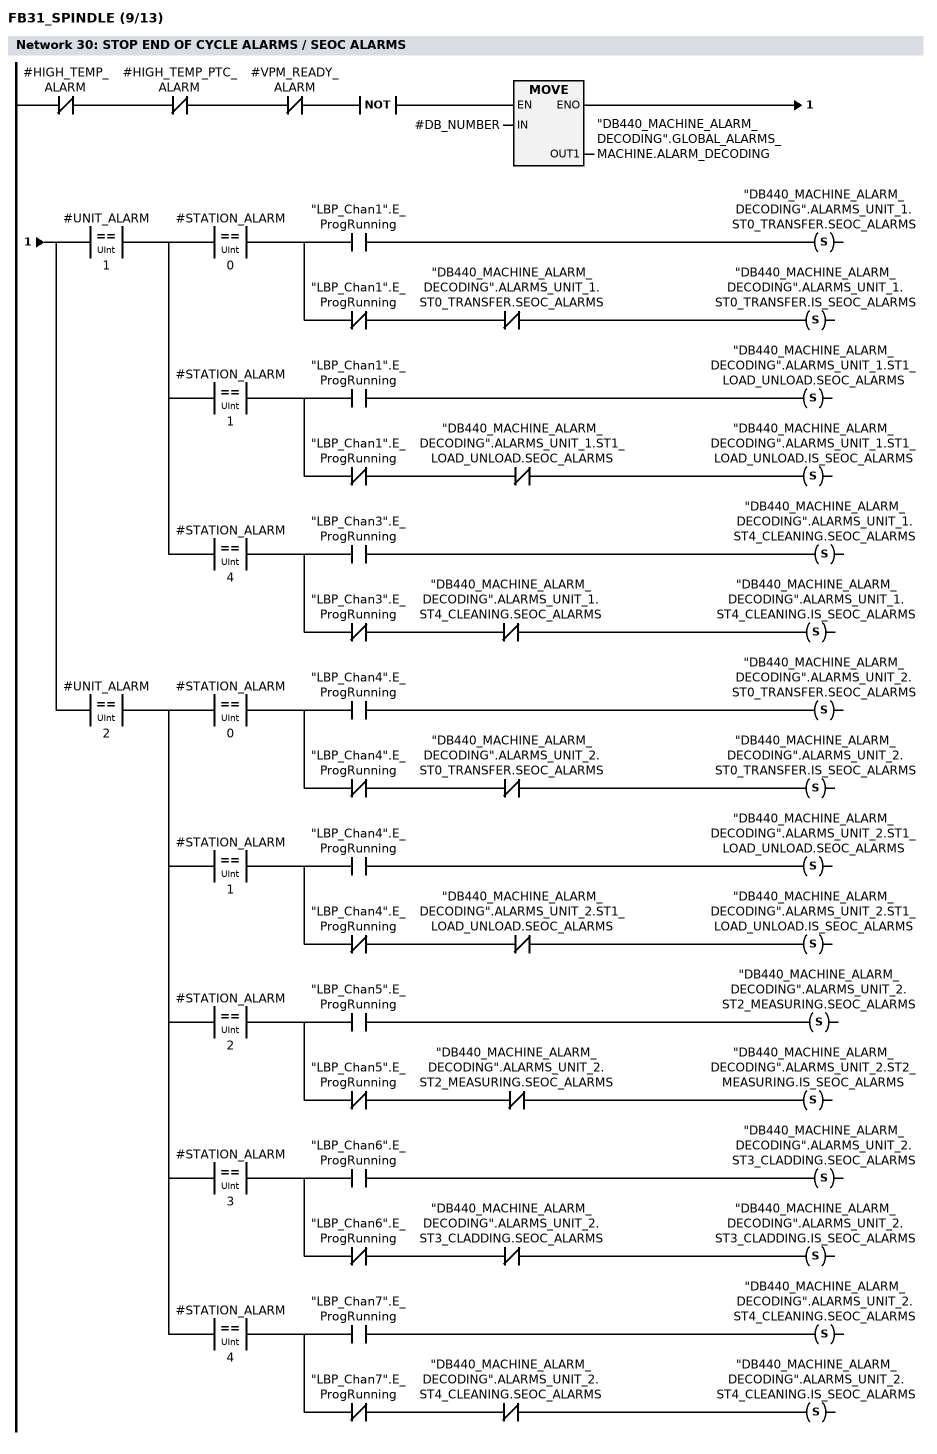
   RUNG wire#powerrail
      I_Contact( #HIGH_TEMP_ALARM )
      I_Contact( #HIGH_TEMP_PTC_ALARM )
      I_Contact( #VPM_READY_ALARM )
      Not()
      { S7_GenerateENO := "TRUE" } Move(in := #DB_NUMBER, out1 => "DB440_MACHINE_ALARM_DECODING".GLOBAL_ALARMS_MACHINE.ALARM_DECODING)
      wire#w1
      { S7_Templates := "SrcType := UInt" } EQ_Contact(in1 := #UNIT_ALARM, in2 := 1)
      wire#w2
      { S7_Templates := "SrcType := UInt" } EQ_Contact(in1 := #STATION_ALARM, in2 := 0)
      wire#w3
      Contact( "LBP_Chan1".E_ProgRunning )
      S_Coil( "DB440_MACHINE_ALARM_DECODING".ALARMS_UNIT_1.ST0_TRANSFER.SEOC_ALARMS )
   END_RUNG
   RUNG wire#w3
      I_Contact( "LBP_Chan1".E_ProgRunning )
      I_Contact( "DB440_MACHINE_ALARM_DECODING".ALARMS_UNIT_1.ST0_TRANSFER.SEOC_ALARMS )
      S_Coil( "DB440_MACHINE_ALARM_DECODING".ALARMS_UNIT_1.ST0_TRANSFER.IS_SEOC_ALARMS )
   END_RUNG
   RUNG wire#w2
      { S7_Templates := "SrcType := UInt" } EQ_Contact(in1 := #STATION_ALARM, in2 := 1)
      wire#w4
      Contact( "LBP_Chan1".E_ProgRunning )
      S_Coil( "DB440_MACHINE_ALARM_DECODING".ALARMS_UNIT_1.ST1_LOAD_UNLOAD.SEOC_ALARMS )
   END_RUNG
   RUNG wire#w4
      I_Contact( "LBP_Chan1".E_ProgRunning )
      I_Contact( "DB440_MACHINE_ALARM_DECODING".ALARMS_UNIT_1.ST1_LOAD_UNLOAD.SEOC_ALARMS )
      S_Coil( "DB440_MACHINE_ALARM_DECODING".ALARMS_UNIT_1.ST1_LOAD_UNLOAD.IS_SEOC_ALARMS )
   END_RUNG
   RUNG wire#w2
      { S7_Templates := "SrcType := UInt" } EQ_Contact(in1 := #STATION_ALARM, in2 := 4)
      wire#w5
      Contact( "LBP_Chan3".E_ProgRunning )
      S_Coil( "DB440_MACHINE_ALARM_DECODING".ALARMS_UNIT_1.ST4_CLEANING.SEOC_ALARMS )
   END_RUNG
   RUNG wire#w5
      I_Contact( "LBP_Chan3".E_ProgRunning )
      I_Contact( "DB440_MACHINE_ALARM_DECODING".ALARMS_UNIT_1.ST4_CLEANING.SEOC_ALARMS )
      S_Coil( "DB440_MACHINE_ALARM_DECODING".ALARMS_UNIT_1.ST4_CLEANING.IS_SEOC_ALARMS )
   END_RUNG
   RUNG wire#w1
      { S7_Templates := "SrcType := UInt" } EQ_Contact(in1 := #UNIT_ALARM, in2 := 2)
      wire#w6
      { S7_Templates := "SrcType := UInt" } EQ_Contact(in1 := #STATION_ALARM, in2 := 0)
      wire#w7
      Contact( "LBP_Chan4".E_ProgRunning )
      S_Coil( "DB440_MACHINE_ALARM_DECODING".ALARMS_UNIT_2.ST0_TRANSFER.SEOC_ALARMS )
   END_RUNG
   RUNG wire#w7
      I_Contact( "LBP_Chan4".E_ProgRunning )
      I_Contact( "DB440_MACHINE_ALARM_DECODING".ALARMS_UNIT_2.ST0_TRANSFER.SEOC_ALARMS )
      S_Coil( "DB440_MACHINE_ALARM_DECODING".ALARMS_UNIT_2.ST0_TRANSFER.IS_SEOC_ALARMS )
   END_RUNG
   RUNG wire#w6
      { S7_Templates := "SrcType := UInt" } EQ_Contact(in1 := #STATION_ALARM, in2 := 1)
      wire#w8
      Contact( "LBP_Chan4".E_ProgRunning )
      S_Coil( "DB440_MACHINE_ALARM_DECODING".ALARMS_UNIT_2.ST1_LOAD_UNLOAD.SEOC_ALARMS )
   END_RUNG
   RUNG wire#w8
      I_Contact( "LBP_Chan4".E_ProgRunning )
      I_Contact( "DB440_MACHINE_ALARM_DECODING".ALARMS_UNIT_2.ST1_LOAD_UNLOAD.SEOC_ALARMS )
      S_Coil( "DB440_MACHINE_ALARM_DECODING".ALARMS_UNIT_2.ST1_LOAD_UNLOAD.IS_SEOC_ALARMS )
   END_RUNG
   RUNG wire#w6
      { S7_Templates := "SrcType := UInt" } EQ_Contact(in1 := #STATION_ALARM, in2 := 2)
      wire#w9
      Contact( "LBP_Chan5".E_ProgRunning )
      S_Coil( "DB440_MACHINE_ALARM_DECODING".ALARMS_UNIT_2.ST2_MEASURING.SEOC_ALARMS )
   END_RUNG
   RUNG wire#w9
      I_Contact( "LBP_Chan5".E_ProgRunning )
      I_Contact( "DB440_MACHINE_ALARM_DECODING".ALARMS_UNIT_2.ST2_MEASURING.SEOC_ALARMS )
      S_Coil( "DB440_MACHINE_ALARM_DECODING".ALARMS_UNIT_2.ST2_MEASURING.IS_SEOC_ALARMS )
   END_RUNG
   RUNG wire#w6
      { S7_Templates := "SrcType := UInt" } EQ_Contact(in1 := #STATION_ALARM, in2 := 3)
      wire#w10
      Contact( "LBP_Chan6".E_ProgRunning )
      S_Coil( "DB440_MACHINE_ALARM_DECODING".ALARMS_UNIT_2.ST3_CLADDING.SEOC_ALARMS )
   END_RUNG
   RUNG wire#w10
      I_Contact( "LBP_Chan6".E_ProgRunning )
      I_Contact( "DB440_MACHINE_ALARM_DECODING".ALARMS_UNIT_2.ST3_CLADDING.SEOC_ALARMS )
      S_Coil( "DB440_MACHINE_ALARM_DECODING".ALARMS_UNIT_2.ST3_CLADDING.IS_SEOC_ALARMS )
   END_RUNG
   RUNG wire#w6
      { S7_Templates := "SrcType := UInt" } EQ_Contact(in1 := #STATION_ALARM, in2 := 4)
      wire#w11
      Contact( "LBP_Chan7".E_ProgRunning )
      S_Coil( "DB440_MACHINE_ALARM_DECODING".ALARMS_UNIT_2.ST4_CLEANING.SEOC_ALARMS )
   END_RUNG
   RUNG wire#w11
      I_Contact( "LBP_Chan7".E_ProgRunning )
      I_Contact( "DB440_MACHINE_ALARM_DECODING".ALARMS_UNIT_2.ST4_CLEANING.SEOC_ALARMS )
      S_Coil( "DB440_MACHINE_ALARM_DECODING".ALARMS_UNIT_2.ST4_CLEANING.IS_SEOC_ALARMS )
   END_RUNG
   // the same network as SCL:
   // ENO of a box is taken as its EN; it also drops when the box reports an error
   #_w1 := NOT (NOT #HIGH_TEMP_ALARM AND NOT #HIGH_TEMP_PTC_ALARM AND NOT #VPM_READY_ALARM);
   IF #_w1 THEN "DB440_MACHINE_ALARM_DECODING".GLOBAL_ALARMS_MACHINE.ALARM_DECODING := #DB_NUMBER; END_IF;
   #_w2 := #_w1 AND (#UNIT_ALARM = 1);
   #_w3 := #_w2 AND (#STATION_ALARM = 0);
   IF #_w3 AND "LBP_Chan1".E_ProgRunning THEN
       "DB440_MACHINE_ALARM_DECODING".ALARMS_UNIT_1.ST0_TRANSFER.SEOC_ALARMS := TRUE;
   END_IF;
   IF #_w3 AND NOT "LBP_Chan1".E_ProgRunning AND NOT "DB440_MACHINE_ALARM_DECODING".ALARMS_UNIT_1.ST0_TRANSFER.SEOC_ALARMS THEN
       "DB440_MACHINE_ALARM_DECODING".ALARMS_UNIT_1.ST0_TRANSFER.IS_SEOC_ALARMS := TRUE;
   END_IF;
   #_w4 := #_w2 AND (#STATION_ALARM = 1);
   IF #_w4 AND "LBP_Chan1".E_ProgRunning THEN
       "DB440_MACHINE_ALARM_DECODING".ALARMS_UNIT_1.ST1_LOAD_UNLOAD.SEOC_ALARMS := TRUE;
   END_IF;
   IF #_w4 AND NOT "LBP_Chan1".E_ProgRunning AND NOT "DB440_MACHINE_ALARM_DECODING".ALARMS_UNIT_1.ST1_LOAD_UNLOAD.SEOC_ALARMS THEN
       "DB440_MACHINE_ALARM_DECODING".ALARMS_UNIT_1.ST1_LOAD_UNLOAD.IS_SEOC_ALARMS := TRUE;
   END_IF;
   #_w5 := #_w2 AND (#STATION_ALARM = 4);
   IF #_w5 AND "LBP_Chan3".E_ProgRunning THEN
       "DB440_MACHINE_ALARM_DECODING".ALARMS_UNIT_1.ST4_CLEANING.SEOC_ALARMS := TRUE;
   END_IF;
   IF #_w5 AND NOT "LBP_Chan3".E_ProgRunning AND NOT "DB440_MACHINE_ALARM_DECODING".ALARMS_UNIT_1.ST4_CLEANING.SEOC_ALARMS THEN
       "DB440_MACHINE_ALARM_DECODING".ALARMS_UNIT_1.ST4_CLEANING.IS_SEOC_ALARMS := TRUE;
   END_IF;
   #_w6 := #_w1 AND (#UNIT_ALARM = 2);
   #_w7 := #_w6 AND (#STATION_ALARM = 0);
   IF #_w7 AND "LBP_Chan4".E_ProgRunning THEN
       "DB440_MACHINE_ALARM_DECODING".ALARMS_UNIT_2.ST0_TRANSFER.SEOC_ALARMS := TRUE;
   END_IF;
   IF #_w7 AND NOT "LBP_Chan4".E_ProgRunning AND NOT "DB440_MACHINE_ALARM_DECODING".ALARMS_UNIT_2.ST0_TRANSFER.SEOC_ALARMS THEN
       "DB440_MACHINE_ALARM_DECODING".ALARMS_UNIT_2.ST0_TRANSFER.IS_SEOC_ALARMS := TRUE;
   END_IF;
   #_w8 := #_w6 AND (#STATION_ALARM = 1);
   IF #_w8 AND "LBP_Chan4".E_ProgRunning THEN
       "DB440_MACHINE_ALARM_DECODING".ALARMS_UNIT_2.ST1_LOAD_UNLOAD.SEOC_ALARMS := TRUE;
   END_IF;
   IF #_w8 AND NOT "LBP_Chan4".E_ProgRunning AND NOT "DB440_MACHINE_ALARM_DECODING".ALARMS_UNIT_2.ST1_LOAD_UNLOAD.SEOC_ALARMS THEN
       "DB440_MACHINE_ALARM_DECODING".ALARMS_UNIT_2.ST1_LOAD_UNLOAD.IS_SEOC_ALARMS := TRUE;
   END_IF;
   #_w9 := #_w6 AND (#STATION_ALARM = 2);
   IF #_w9 AND "LBP_Chan5".E_ProgRunning THEN
       "DB440_MACHINE_ALARM_DECODING".ALARMS_UNIT_2.ST2_MEASURING.SEOC_ALARMS := TRUE;
   END_IF;
   IF #_w9 AND NOT "LBP_Chan5".E_ProgRunning AND NOT "DB440_MACHINE_ALARM_DECODING".ALARMS_UNIT_2.ST2_MEASURING.SEOC_ALARMS THEN
       "DB440_MACHINE_ALARM_DECODING".ALARMS_UNIT_2.ST2_MEASURING.IS_SEOC_ALARMS := TRUE;
   END_IF;
   #_w10 := #_w6 AND (#STATION_ALARM = 3);
   IF #_w10 AND "LBP_Chan6".E_ProgRunning THEN
       "DB440_MACHINE_ALARM_DECODING".ALARMS_UNIT_2.ST3_CLADDING.SEOC_ALARMS := TRUE;
   END_IF;
   IF #_w10 AND NOT "LBP_Chan6".E_ProgRunning AND NOT "DB440_MACHINE_ALARM_DECODING".ALARMS_UNIT_2.ST3_CLADDING.SEOC_ALARMS THEN
       "DB440_MACHINE_ALARM_DECODING".ALARMS_UNIT_2.ST3_CLADDING.IS_SEOC_ALARMS := TRUE;
   END_IF;
   #_w11 := #_w6 AND (#STATION_ALARM = 4);
   IF #_w11 AND "LBP_Chan7".E_ProgRunning THEN
       "DB440_MACHINE_ALARM_DECODING".ALARMS_UNIT_2.ST4_CLEANING.SEOC_ALARMS := TRUE;
   END_IF;
   IF #_w11 AND NOT "LBP_Chan7".E_ProgRunning AND NOT "DB440_MACHINE_ALARM_DECODING".ALARMS_UNIT_2.ST4_CLEANING.SEOC_ALARMS THEN
       "DB440_MACHINE_ALARM_DECODING".ALARMS_UNIT_2.ST4_CLEANING.IS_SEOC_ALARMS := TRUE;
   END_IF;
END_REGION

REGION Network 31: RETURN HOME POSITION AND RUN OUT ALARMS
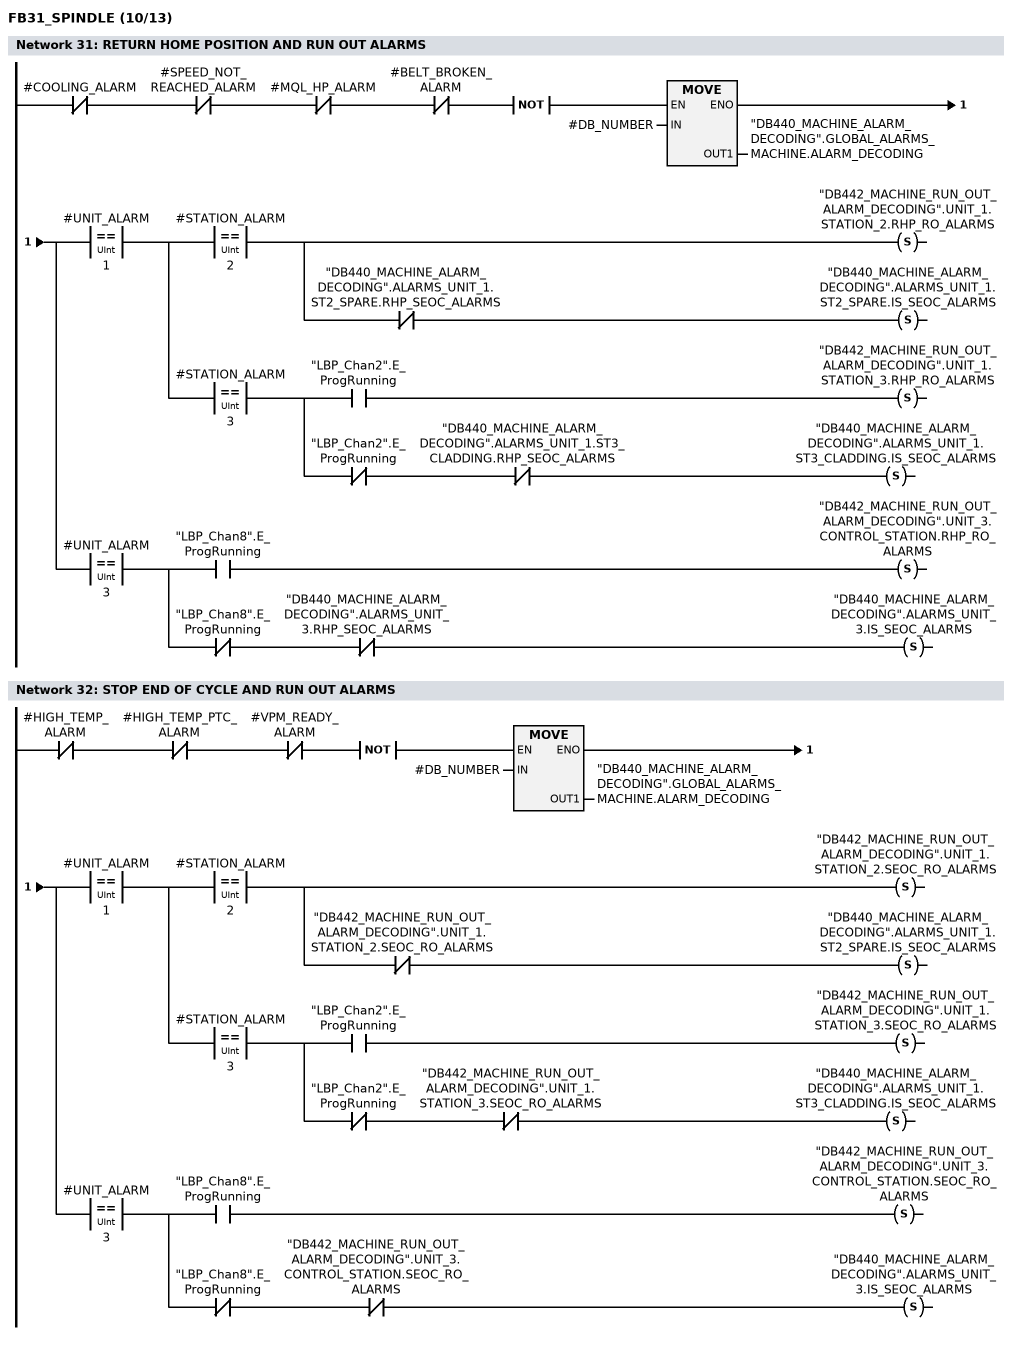
   RUNG wire#powerrail
      I_Contact( #COOLING_ALARM )
      I_Contact( #SPEED_NOT_REACHED_ALARM )
      I_Contact( #MQL_HP_ALARM )
      I_Contact( #BELT_BROKEN_ALARM )
      Not()
      Move(in := #DB_NUMBER, out1 => "DB440_MACHINE_ALARM_DECODING".GLOBAL_ALARMS_MACHINE.ALARM_DECODING)
      wire#w1
      { S7_Templates := "SrcType := UInt" } EQ_Contact(in1 := #UNIT_ALARM, in2 := 1)
      wire#w2
      { S7_Templates := "SrcType := UInt" } EQ_Contact(in1 := #STATION_ALARM, in2 := 2)
      wire#w3
      S_Coil( "DB442_MACHINE_RUN_OUT_ALARM_DECODING".UNIT_1.STATION_2.RHP_RO_ALARMS )
   END_RUNG
   RUNG wire#w3
      I_Contact( "DB440_MACHINE_ALARM_DECODING".ALARMS_UNIT_1.ST2_SPARE.RHP_SEOC_ALARMS )
      S_Coil( "DB440_MACHINE_ALARM_DECODING".ALARMS_UNIT_1.ST2_SPARE.IS_SEOC_ALARMS )
   END_RUNG
   RUNG wire#w2
      { S7_Templates := "SrcType := UInt" } EQ_Contact(in1 := #STATION_ALARM, in2 := 3)
      wire#w4
      Contact( "LBP_Chan2".E_ProgRunning )
      S_Coil( "DB442_MACHINE_RUN_OUT_ALARM_DECODING".UNIT_1.STATION_3.RHP_RO_ALARMS )
   END_RUNG
   RUNG wire#w4
      I_Contact( "LBP_Chan2".E_ProgRunning )
      I_Contact( "DB440_MACHINE_ALARM_DECODING".ALARMS_UNIT_1.ST3_CLADDING.RHP_SEOC_ALARMS )
      S_Coil( "DB440_MACHINE_ALARM_DECODING".ALARMS_UNIT_1.ST3_CLADDING.IS_SEOC_ALARMS )
   END_RUNG
   RUNG wire#w1
      { S7_Templates := "SrcType := UInt" } EQ_Contact(in1 := #UNIT_ALARM, in2 := 3)
      wire#w5
      Contact( "LBP_Chan8".E_ProgRunning )
      S_Coil( "DB442_MACHINE_RUN_OUT_ALARM_DECODING".UNIT_3.CONTROL_STATION.RHP_RO_ALARMS )
   END_RUNG
   RUNG wire#w5
      I_Contact( "LBP_Chan8".E_ProgRunning )
      I_Contact( "DB440_MACHINE_ALARM_DECODING".ALARMS_UNIT_3.RHP_SEOC_ALARMS )
      S_Coil( "DB440_MACHINE_ALARM_DECODING".ALARMS_UNIT_3.IS_SEOC_ALARMS )
   END_RUNG
   // the same network as SCL:
   #_w1 := NOT (NOT #COOLING_ALARM AND NOT #SPEED_NOT_REACHED_ALARM AND NOT #MQL_HP_ALARM AND NOT #BELT_BROKEN_ALARM);
   IF #_w1 THEN "DB440_MACHINE_ALARM_DECODING".GLOBAL_ALARMS_MACHINE.ALARM_DECODING := #DB_NUMBER; END_IF;
   #_w2 := #_w1 AND (#UNIT_ALARM = 1);
   #_w3 := #_w2 AND (#STATION_ALARM = 2);
   IF #_w3 THEN "DB442_MACHINE_RUN_OUT_ALARM_DECODING".UNIT_1.STATION_2.RHP_RO_ALARMS := TRUE; END_IF;
   IF #_w3 AND NOT "DB440_MACHINE_ALARM_DECODING".ALARMS_UNIT_1.ST2_SPARE.RHP_SEOC_ALARMS THEN
       "DB440_MACHINE_ALARM_DECODING".ALARMS_UNIT_1.ST2_SPARE.IS_SEOC_ALARMS := TRUE;
   END_IF;
   #_w4 := #_w2 AND (#STATION_ALARM = 3);
   IF #_w4 AND "LBP_Chan2".E_ProgRunning THEN
       "DB442_MACHINE_RUN_OUT_ALARM_DECODING".UNIT_1.STATION_3.RHP_RO_ALARMS := TRUE;
   END_IF;
   IF #_w4 AND NOT "LBP_Chan2".E_ProgRunning AND NOT "DB440_MACHINE_ALARM_DECODING".ALARMS_UNIT_1.ST3_CLADDING.RHP_SEOC_ALARMS THEN
       "DB440_MACHINE_ALARM_DECODING".ALARMS_UNIT_1.ST3_CLADDING.IS_SEOC_ALARMS := TRUE;
   END_IF;
   #_w5 := #_w1 AND (#UNIT_ALARM = 3);
   IF #_w5 AND "LBP_Chan8".E_ProgRunning THEN
       "DB442_MACHINE_RUN_OUT_ALARM_DECODING".UNIT_3.CONTROL_STATION.RHP_RO_ALARMS := TRUE;
   END_IF;
   IF #_w5 AND NOT "LBP_Chan8".E_ProgRunning AND NOT "DB440_MACHINE_ALARM_DECODING".ALARMS_UNIT_3.RHP_SEOC_ALARMS THEN
       "DB440_MACHINE_ALARM_DECODING".ALARMS_UNIT_3.IS_SEOC_ALARMS := TRUE;
   END_IF;
END_REGION

REGION Network 32: STOP END OF CYCLE AND RUN OUT ALARMS
   RUNG wire#powerrail
      I_Contact( #HIGH_TEMP_ALARM )
      I_Contact( #HIGH_TEMP_PTC_ALARM )
      I_Contact( #VPM_READY_ALARM )
      Not()
      { S7_GenerateENO := "TRUE" } Move(in := #DB_NUMBER, out1 => "DB440_MACHINE_ALARM_DECODING".GLOBAL_ALARMS_MACHINE.ALARM_DECODING)
      wire#w1
      { S7_Templates := "SrcType := UInt" } EQ_Contact(in1 := #UNIT_ALARM, in2 := 1)
      wire#w2
      { S7_Templates := "SrcType := UInt" } EQ_Contact(in1 := #STATION_ALARM, in2 := 2)
      wire#w3
      S_Coil( "DB442_MACHINE_RUN_OUT_ALARM_DECODING".UNIT_1.STATION_2.SEOC_RO_ALARMS )
   END_RUNG
   RUNG wire#w3
      I_Contact( "DB442_MACHINE_RUN_OUT_ALARM_DECODING".UNIT_1.STATION_2.SEOC_RO_ALARMS )
      S_Coil( "DB440_MACHINE_ALARM_DECODING".ALARMS_UNIT_1.ST2_SPARE.IS_SEOC_ALARMS )
   END_RUNG
   RUNG wire#w2
      { S7_Templates := "SrcType := UInt" } EQ_Contact(in1 := #STATION_ALARM, in2 := 3)
      wire#w4
      Contact( "LBP_Chan2".E_ProgRunning )
      S_Coil( "DB442_MACHINE_RUN_OUT_ALARM_DECODING".UNIT_1.STATION_3.SEOC_RO_ALARMS )
   END_RUNG
   RUNG wire#w4
      I_Contact( "LBP_Chan2".E_ProgRunning )
      I_Contact( "DB442_MACHINE_RUN_OUT_ALARM_DECODING".UNIT_1.STATION_3.SEOC_RO_ALARMS )
      S_Coil( "DB440_MACHINE_ALARM_DECODING".ALARMS_UNIT_1.ST3_CLADDING.IS_SEOC_ALARMS )
   END_RUNG
   RUNG wire#w1
      { S7_Templates := "SrcType := UInt" } EQ_Contact(in1 := #UNIT_ALARM, in2 := 3)
      wire#w5
      Contact( "LBP_Chan8".E_ProgRunning )
      S_Coil( "DB442_MACHINE_RUN_OUT_ALARM_DECODING".UNIT_3.CONTROL_STATION.SEOC_RO_ALARMS )
   END_RUNG
   RUNG wire#w5
      I_Contact( "LBP_Chan8".E_ProgRunning )
      I_Contact( "DB442_MACHINE_RUN_OUT_ALARM_DECODING".UNIT_3.CONTROL_STATION.SEOC_RO_ALARMS )
      S_Coil( "DB440_MACHINE_ALARM_DECODING".ALARMS_UNIT_3.IS_SEOC_ALARMS )
   END_RUNG
   // the same network as SCL:
   // ENO of a box is taken as its EN; it also drops when the box reports an error
   #_w1 := NOT (NOT #HIGH_TEMP_ALARM AND NOT #HIGH_TEMP_PTC_ALARM AND NOT #VPM_READY_ALARM);
   IF #_w1 THEN "DB440_MACHINE_ALARM_DECODING".GLOBAL_ALARMS_MACHINE.ALARM_DECODING := #DB_NUMBER; END_IF;
   #_w2 := #_w1 AND (#UNIT_ALARM = 1);
   #_w3 := #_w2 AND (#STATION_ALARM = 2);
   IF #_w3 THEN "DB442_MACHINE_RUN_OUT_ALARM_DECODING".UNIT_1.STATION_2.SEOC_RO_ALARMS := TRUE; END_IF;
   IF #_w3 AND NOT "DB442_MACHINE_RUN_OUT_ALARM_DECODING".UNIT_1.STATION_2.SEOC_RO_ALARMS THEN
       "DB440_MACHINE_ALARM_DECODING".ALARMS_UNIT_1.ST2_SPARE.IS_SEOC_ALARMS := TRUE;
   END_IF;
   #_w4 := #_w2 AND (#STATION_ALARM = 3);
   IF #_w4 AND "LBP_Chan2".E_ProgRunning THEN
       "DB442_MACHINE_RUN_OUT_ALARM_DECODING".UNIT_1.STATION_3.SEOC_RO_ALARMS := TRUE;
   END_IF;
   IF #_w4 AND NOT "LBP_Chan2".E_ProgRunning AND NOT "DB442_MACHINE_RUN_OUT_ALARM_DECODING".UNIT_1.STATION_3.SEOC_RO_ALARMS THEN
       "DB440_MACHINE_ALARM_DECODING".ALARMS_UNIT_1.ST3_CLADDING.IS_SEOC_ALARMS := TRUE;
   END_IF;
   #_w5 := #_w1 AND (#UNIT_ALARM = 3);
   IF #_w5 AND "LBP_Chan8".E_ProgRunning THEN
       "DB442_MACHINE_RUN_OUT_ALARM_DECODING".UNIT_3.CONTROL_STATION.SEOC_RO_ALARMS := TRUE;
   END_IF;
   IF #_w5 AND NOT "LBP_Chan8".E_ProgRunning AND NOT "DB442_MACHINE_RUN_OUT_ALARM_DECODING".UNIT_3.CONTROL_STATION.SEOC_RO_ALARMS THEN
       "DB440_MACHINE_ALARM_DECODING".ALARMS_UNIT_3.IS_SEOC_ALARMS := TRUE;
   END_IF;
END_REGION

REGION Network 33: PROGRESSIVE STOP POWDER ALARMS
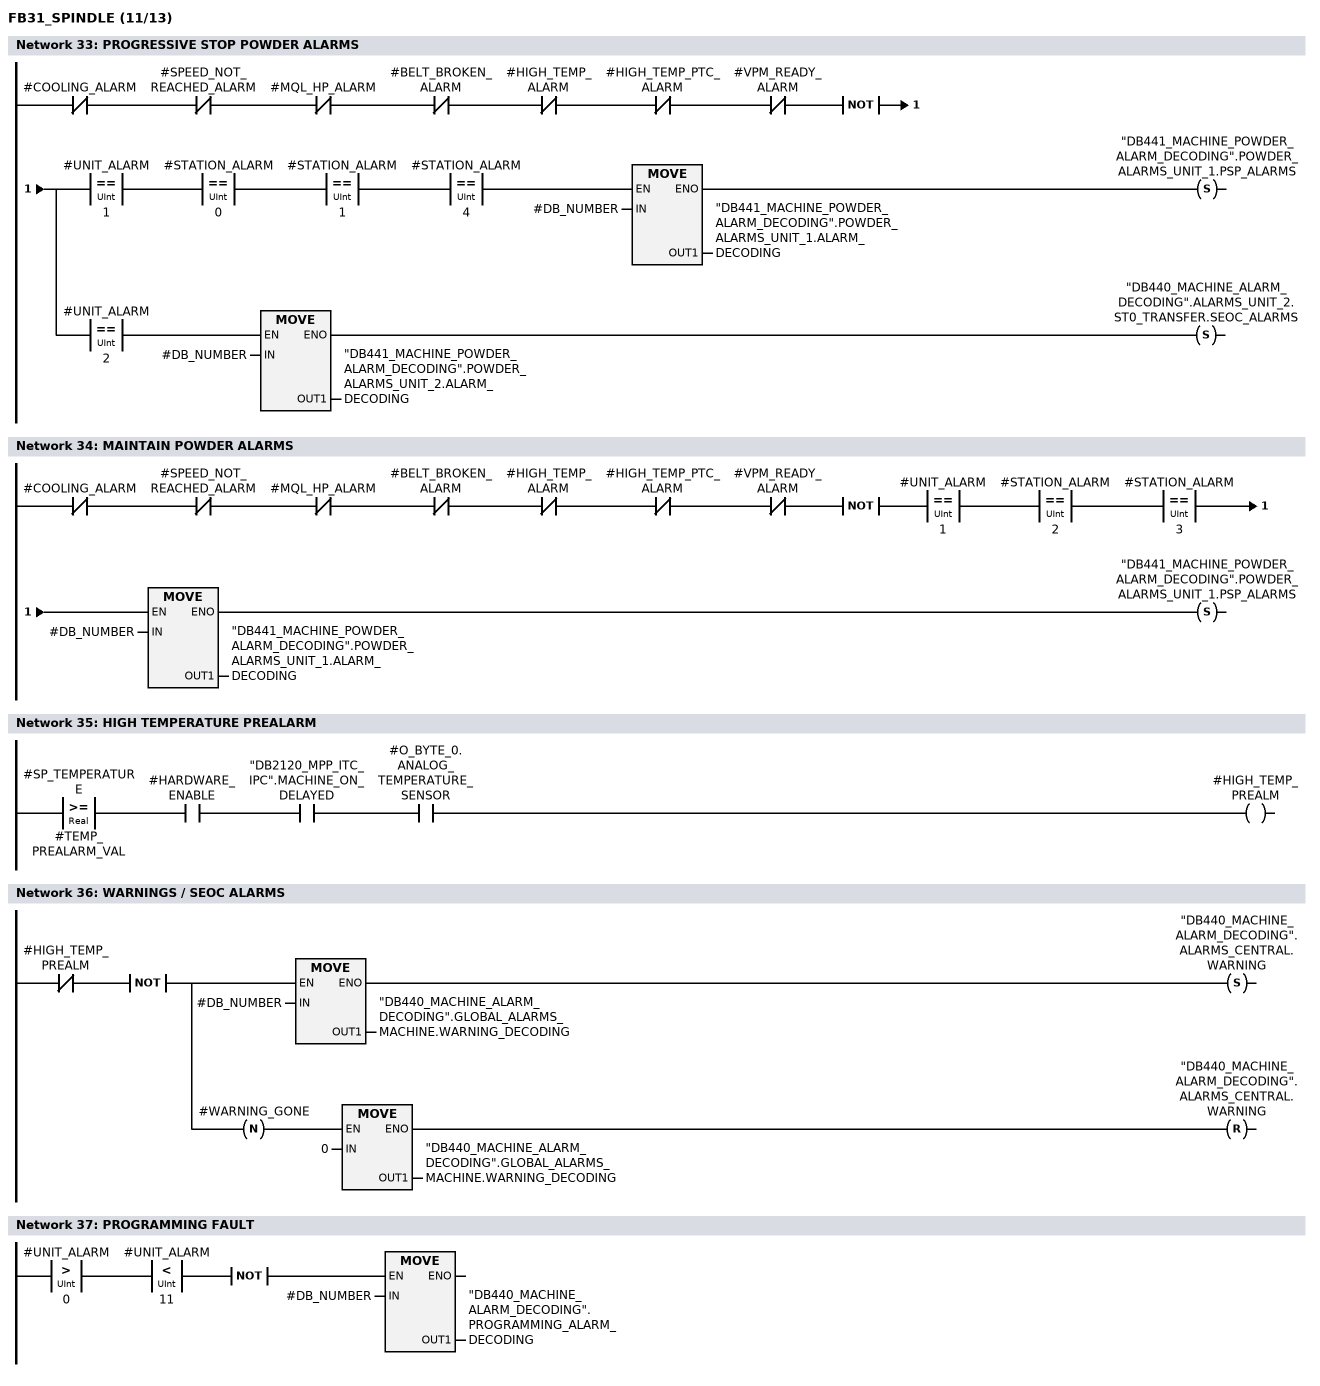
   RUNG wire#powerrail
      I_Contact( #COOLING_ALARM )
      I_Contact( #SPEED_NOT_REACHED_ALARM )
      I_Contact( #MQL_HP_ALARM )
      I_Contact( #BELT_BROKEN_ALARM )
      I_Contact( #HIGH_TEMP_ALARM )
      I_Contact( #HIGH_TEMP_PTC_ALARM )
      I_Contact( #VPM_READY_ALARM )
      Not()
      wire#w1
      { S7_Templates := "SrcType := UInt" } EQ_Contact(in1 := #UNIT_ALARM, in2 := 1)
      { S7_Templates := "SrcType := UInt" } EQ_Contact(in1 := #STATION_ALARM, in2 := 0)
      { S7_Templates := "SrcType := UInt" } EQ_Contact(in1 := #STATION_ALARM, in2 := 1)
      { S7_Templates := "SrcType := UInt" } EQ_Contact(in1 := #STATION_ALARM, in2 := 4)
      { S7_GenerateENO := "TRUE" } Move(in := #DB_NUMBER, out1 => "DB441_MACHINE_POWDER_ALARM_DECODING".POWDER_ALARMS_UNIT_1.ALARM_DECODING)
      S_Coil( "DB441_MACHINE_POWDER_ALARM_DECODING".POWDER_ALARMS_UNIT_1.PSP_ALARMS )
   END_RUNG
   RUNG wire#w1
      { S7_Templates := "SrcType := UInt" } EQ_Contact(in1 := #UNIT_ALARM, in2 := 2)
      { S7_GenerateENO := "TRUE" } Move(in := #DB_NUMBER, out1 => "DB441_MACHINE_POWDER_ALARM_DECODING".POWDER_ALARMS_UNIT_2.ALARM_DECODING)
      S_Coil( "DB440_MACHINE_ALARM_DECODING".ALARMS_UNIT_2.ST0_TRANSFER.SEOC_ALARMS )
   END_RUNG
   // the same network as SCL:
   // ENO of a box is taken as its EN; it also drops when the box reports an error
   #_w1 := NOT (NOT #COOLING_ALARM AND NOT #SPEED_NOT_REACHED_ALARM AND NOT #MQL_HP_ALARM AND NOT #BELT_BROKEN_ALARM AND NOT #HIGH_TEMP_ALARM AND NOT #HIGH_TEMP_PTC_ALARM AND NOT #VPM_READY_ALARM);
   IF #_w1 AND (#UNIT_ALARM = 1) AND (#STATION_ALARM = 0) AND (#STATION_ALARM = 1) AND (#STATION_ALARM = 4) THEN
       "DB441_MACHINE_POWDER_ALARM_DECODING".POWDER_ALARMS_UNIT_1.ALARM_DECODING := #DB_NUMBER;
       "DB441_MACHINE_POWDER_ALARM_DECODING".POWDER_ALARMS_UNIT_1.PSP_ALARMS := TRUE;
   END_IF;
   IF #_w1 AND (#UNIT_ALARM = 2) THEN
       "DB441_MACHINE_POWDER_ALARM_DECODING".POWDER_ALARMS_UNIT_2.ALARM_DECODING := #DB_NUMBER;
       "DB440_MACHINE_ALARM_DECODING".ALARMS_UNIT_2.ST0_TRANSFER.SEOC_ALARMS := TRUE;
   END_IF;
END_REGION

REGION Network 34: MAINTAIN POWDER ALARMS
   RUNG wire#powerrail
      I_Contact( #COOLING_ALARM )
      I_Contact( #SPEED_NOT_REACHED_ALARM )
      I_Contact( #MQL_HP_ALARM )
      I_Contact( #BELT_BROKEN_ALARM )
      I_Contact( #HIGH_TEMP_ALARM )
      I_Contact( #HIGH_TEMP_PTC_ALARM )
      I_Contact( #VPM_READY_ALARM )
      Not()
      { S7_Templates := "SrcType := UInt" } EQ_Contact(in1 := #UNIT_ALARM, in2 := 1)
      { S7_Templates := "SrcType := UInt" } EQ_Contact(in1 := #STATION_ALARM, in2 := 2)
      { S7_Templates := "SrcType := UInt" } EQ_Contact(in1 := #STATION_ALARM, in2 := 3)
      { S7_GenerateENO := "TRUE" } Move(in := #DB_NUMBER, out1 => "DB441_MACHINE_POWDER_ALARM_DECODING".POWDER_ALARMS_UNIT_1.ALARM_DECODING)
      S_Coil( "DB441_MACHINE_POWDER_ALARM_DECODING".POWDER_ALARMS_UNIT_1.PSP_ALARMS )
   END_RUNG
   // the same network as SCL:
   // ENO of a box is taken as its EN; it also drops when the box reports an error
   IF NOT (NOT #COOLING_ALARM AND NOT #SPEED_NOT_REACHED_ALARM AND NOT #MQL_HP_ALARM AND NOT #BELT_BROKEN_ALARM AND NOT #HIGH_TEMP_ALARM AND NOT #HIGH_TEMP_PTC_ALARM AND NOT #VPM_READY_ALARM) AND (#UNIT_ALARM = 1) AND (#STATION_ALARM = 2) AND (#STATION_ALARM = 3) THEN
       "DB441_MACHINE_POWDER_ALARM_DECODING".POWDER_ALARMS_UNIT_1.ALARM_DECODING := #DB_NUMBER;
       "DB441_MACHINE_POWDER_ALARM_DECODING".POWDER_ALARMS_UNIT_1.PSP_ALARMS := TRUE;
   END_IF;
END_REGION

REGION Network 35: HIGH TEMPERATURE PREALARM
   RUNG wire#powerrail
      { S7_Templates := "SrcType := Real" } GE_Contact(in1 := #SP_TEMPERATURE, in2 := #TEMP_PREALARM_VAL)
      Contact( #HARDWARE_ENABLE )
      Contact( "DB2120_MPP_ITC_IPC".MACHINE_ON_DELAYED )
      Contact( #O_BYTE_0.ANALOG_TEMPERATURE_SENSOR )
      Coil( #HIGH_TEMP_PREALM )
   END_RUNG
   // the same network as SCL:
   #HIGH_TEMP_PREALM := (#SP_TEMPERATURE >= #TEMP_PREALARM_VAL) AND #HARDWARE_ENABLE AND "DB2120_MPP_ITC_IPC".MACHINE_ON_DELAYED AND #O_BYTE_0.ANALOG_TEMPERATURE_SENSOR;
END_REGION

REGION Network 36: WARNINGS / SEOC ALARMS
   RUNG wire#powerrail
      I_Contact( #HIGH_TEMP_PREALM )
      Not()
      wire#w1
      { S7_GenerateENO := "TRUE" } Move(in := #DB_NUMBER, out1 => "DB440_MACHINE_ALARM_DECODING".GLOBAL_ALARMS_MACHINE.WARNING_DECODING)
      S_Coil( "DB440_MACHINE_ALARM_DECODING".ALARMS_CENTRAL.WARNING )
   END_RUNG
   RUNG wire#w1
      N_Trig( #WARNING_GONE )
      { S7_GenerateENO := "TRUE" } Move(in := 0, out1 => "DB440_MACHINE_ALARM_DECODING".GLOBAL_ALARMS_MACHINE.WARNING_DECODING)
      R_Coil( "DB440_MACHINE_ALARM_DECODING".ALARMS_CENTRAL.WARNING )
   END_RUNG
   // the same network as SCL:
   // ENO of a box is taken as its EN; it also drops when the box reports an error
   #_w1 := NOT (NOT #HIGH_TEMP_PREALM);
   IF #_w1 THEN
       "DB440_MACHINE_ALARM_DECODING".GLOBAL_ALARMS_MACHINE.WARNING_DECODING := #DB_NUMBER;
       "DB440_MACHINE_ALARM_DECODING".ALARMS_CENTRAL.WARNING := TRUE;
   END_IF;
   #_w2 := NOT #_w1 AND #WARNING_GONE;   // falling edge
   #WARNING_GONE := #_w1;
   IF #_w2 THEN
       "DB440_MACHINE_ALARM_DECODING".GLOBAL_ALARMS_MACHINE.WARNING_DECODING := 0;
       "DB440_MACHINE_ALARM_DECODING".ALARMS_CENTRAL.WARNING := FALSE;
   END_IF;
END_REGION

REGION Network 37: PROGRAMMING FAULT
   RUNG wire#powerrail
      { S7_Templates := "SrcType := UInt" } GT_Contact(in1 := #UNIT_ALARM, in2 := 0)
      { S7_Templates := "SrcType := UInt" } LT_Contact(in1 := #UNIT_ALARM, in2 := 11)
      Not()
      Move(in := #DB_NUMBER, out1 => "DB440_MACHINE_ALARM_DECODING".PROGRAMMING_ALARM_DECODING)
   END_RUNG
   // the same network as SCL:
   IF NOT ((#UNIT_ALARM > 0) AND (#UNIT_ALARM < 11)) THEN
       "DB440_MACHINE_ALARM_DECODING".PROGRAMMING_ALARM_DECODING := #DB_NUMBER;
   END_IF;
END_REGION

REGION Network 38: OPERATOR HELP / HELP
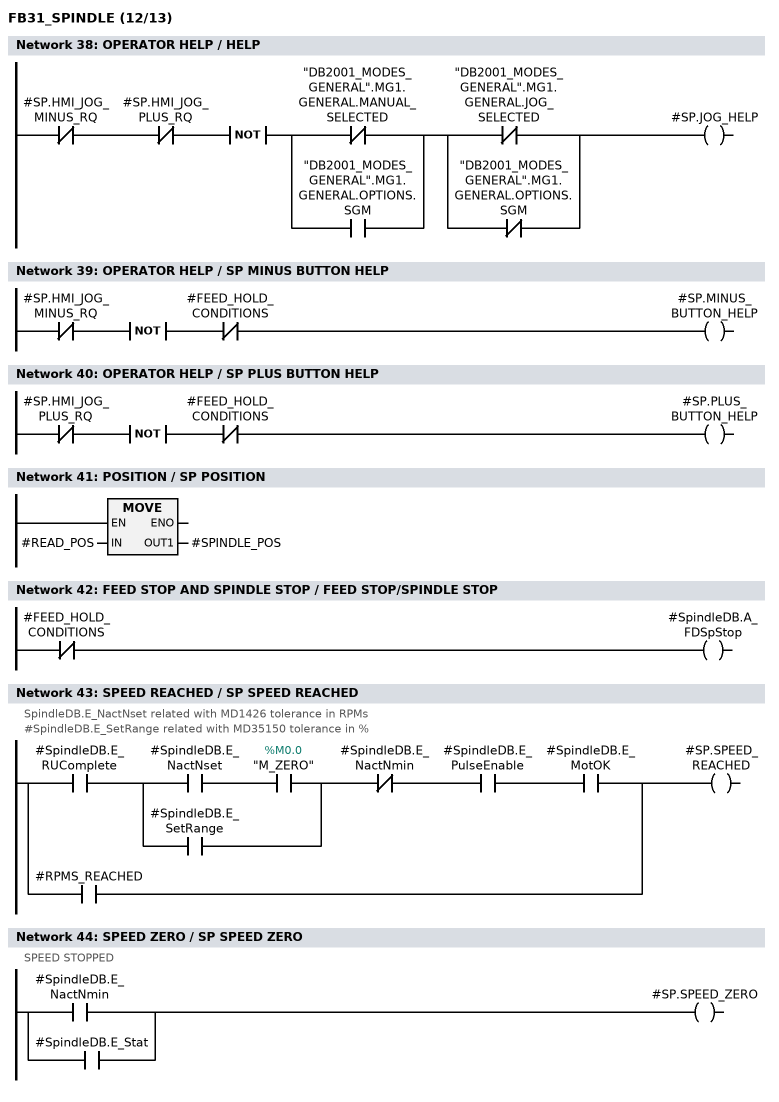
   RUNG wire#powerrail
      I_Contact( #SP.HMI_JOG_MINUS_RQ )
      I_Contact( #SP.HMI_JOG_PLUS_RQ )
      Not()
      wire#w1
      I_Contact( "DB2001_MODES_GENERAL".MG1.GENERAL.MANUAL_SELECTED )
      wire#w2
      I_Contact( "DB2001_MODES_GENERAL".MG1.GENERAL.JOG_SELECTED )
      wire#w3
      Coil( #SP.JOG_HELP )
   END_RUNG
   RUNG wire#w1
      Contact( "DB2001_MODES_GENERAL".MG1.GENERAL.OPTIONS.SGM )
   END_RUNG wire#w2
   RUNG wire#w2
      I_Contact( "DB2001_MODES_GENERAL".MG1.GENERAL.OPTIONS.SGM )
   END_RUNG wire#w3
   // the same network as SCL:
   #SP.JOG_HELP := NOT (NOT #SP.HMI_JOG_MINUS_RQ AND NOT #SP.HMI_JOG_PLUS_RQ) AND (NOT "DB2001_MODES_GENERAL".MG1.GENERAL.MANUAL_SELECTED OR "DB2001_MODES_GENERAL".MG1.GENERAL.OPTIONS.SGM) AND (NOT "DB2001_MODES_GENERAL".MG1.GENERAL.JOG_SELECTED OR NOT "DB2001_MODES_GENERAL".MG1.GENERAL.OPTIONS.SGM);
END_REGION

REGION Network 39: OPERATOR HELP / SP MINUS BUTTON HELP
   RUNG wire#powerrail
      I_Contact( #SP.HMI_JOG_MINUS_RQ )
      Not()
      I_Contact( #FEED_HOLD_CONDITIONS )
      Coil( #SP.MINUS_BUTTON_HELP )
   END_RUNG
   // the same network as SCL:
   #SP.MINUS_BUTTON_HELP := NOT (NOT #SP.HMI_JOG_MINUS_RQ) AND NOT #FEED_HOLD_CONDITIONS;
END_REGION

REGION Network 40: OPERATOR HELP / SP PLUS BUTTON HELP
   RUNG wire#powerrail
      I_Contact( #SP.HMI_JOG_PLUS_RQ )
      Not()
      I_Contact( #FEED_HOLD_CONDITIONS )
      Coil( #SP.PLUS_BUTTON_HELP )
   END_RUNG
   // the same network as SCL:
   #SP.PLUS_BUTTON_HELP := NOT (NOT #SP.HMI_JOG_PLUS_RQ) AND NOT #FEED_HOLD_CONDITIONS;
END_REGION

REGION Network 41: POSITION / SP POSITION
   RUNG wire#powerrail
      { S7_GenerateENO := "TRUE" } Move(in := #READ_POS, out1 => #SPINDLE_POS)
   END_RUNG
   // the same network as SCL:
   #SPINDLE_POS := #READ_POS;
END_REGION

REGION Network 42: FEED STOP AND SPINDLE STOP / FEED STOP/SPINDLE STOP
   RUNG wire#powerrail
      I_Contact( #FEED_HOLD_CONDITIONS )
      Coil( #SpindleDB.A_FDSpStop )
   END_RUNG
   // the same network as SCL:
   #SpindleDB.A_FDSpStop := NOT #FEED_HOLD_CONDITIONS;
END_REGION

REGION Network 43: SPEED REACHED / SP SPEED REACHED
   // SpindleDB.E_NactNset related with MD1426 tolerance in RPMs
   // #SpindleDB.E_SetRange related with MD35150 tolerance in %
   RUNG wire#powerrail
      Contact( #SpindleDB.E_RUComplete )
      wire#w1
      Contact( #SpindleDB.E_NactNset )
      Contact( "M_ZERO" )
      wire#w2
      I_Contact( #SpindleDB.E_NactNmin )
      Contact( #SpindleDB.E_PulseEnable )
      Contact( #SpindleDB.E_MotOK )
      wire#w3
      Coil( #SP.SPEED_REACHED )
   END_RUNG
   RUNG wire#w1
      Contact( #SpindleDB.E_SetRange )
   END_RUNG wire#w2
   RUNG wire#powerrail
      Contact( #RPMS_REACHED )
   END_RUNG wire#w3
   // the same network as SCL:
   #SP.SPEED_REACHED := (#SpindleDB.E_RUComplete AND ((#SpindleDB.E_NactNset AND "M_ZERO") OR #SpindleDB.E_SetRange) AND NOT #SpindleDB.E_NactNmin AND #SpindleDB.E_PulseEnable AND #SpindleDB.E_MotOK) OR #RPMS_REACHED;
END_REGION

REGION Network 44: SPEED ZERO / SP SPEED ZERO
   // SPEED STOPPED
   RUNG wire#powerrail
      Contact( #SpindleDB.E_NactNmin )
      wire#w1
      Coil( #SP.SPEED_ZERO )
   END_RUNG
   RUNG wire#powerrail
      Contact( #SpindleDB.E_Stat )
   END_RUNG wire#w1
   // the same network as SCL:
   #SP.SPEED_ZERO := #SpindleDB.E_NactNmin OR #SpindleDB.E_Stat;
END_REGION

REGION Network 45: CALL FB33 SAFETY POSITIONS
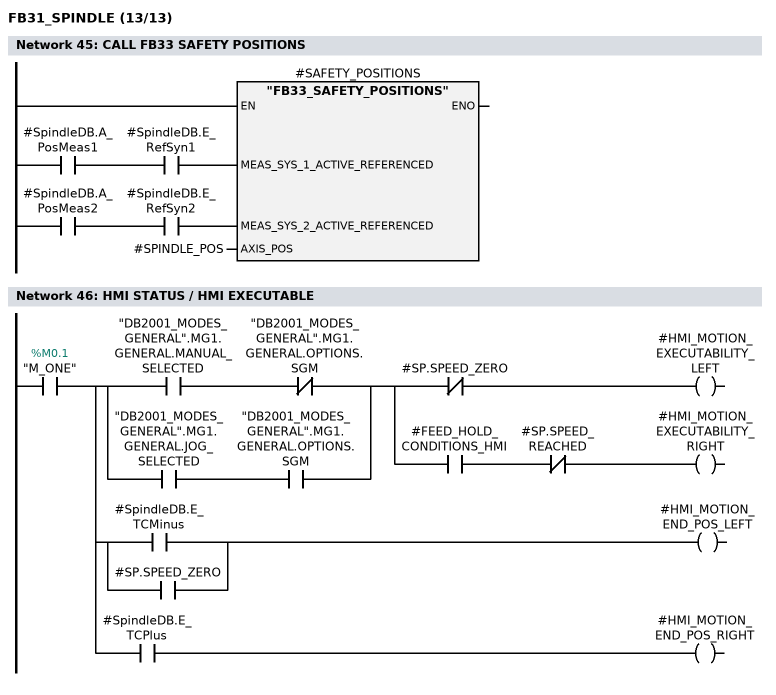
   RUNG wire#powerrail
      #SAFETY_POSITIONS(MEAS_SYS_1_ACTIVE_REFERENCED := wire#w1, MEAS_SYS_2_ACTIVE_REFERENCED := wire#w2, AXIS_POS := #SPINDLE_POS)
   END_RUNG
   RUNG wire#powerrail
      Contact( #SpindleDB.A_PosMeas1 )
      Contact( #SpindleDB.E_RefSyn1 )
   END_RUNG wire#w1
   RUNG wire#powerrail
      Contact( #SpindleDB.A_PosMeas2 )
      Contact( #SpindleDB.E_RefSyn2 )
   END_RUNG wire#w2
   // the same network as SCL:
   #SAFETY_POSITIONS(MEAS_SYS_1_ACTIVE_REFERENCED := #SpindleDB.A_PosMeas1 AND #SpindleDB.E_RefSyn1,   // "FB33_SAFETY_POSITIONS"
                     MEAS_SYS_2_ACTIVE_REFERENCED := #SpindleDB.A_PosMeas2 AND #SpindleDB.E_RefSyn2,
                     AXIS_POS := #SPINDLE_POS);
END_REGION

REGION Network 46: HMI STATUS / HMI EXECUTABLE
   RUNG wire#powerrail
      Contact( "M_ONE" )
      wire#w1
      Contact( "DB2001_MODES_GENERAL".MG1.GENERAL.MANUAL_SELECTED )
      I_Contact( "DB2001_MODES_GENERAL".MG1.GENERAL.OPTIONS.SGM )
      wire#w2
      I_Contact( #SP.SPEED_ZERO )
      Coil( #HMI_MOTION_EXECUTABILITY_LEFT )
   END_RUNG
   RUNG wire#w1
      Contact( "DB2001_MODES_GENERAL".MG1.GENERAL.JOG_SELECTED )
      Contact( "DB2001_MODES_GENERAL".MG1.GENERAL.OPTIONS.SGM )
   END_RUNG wire#w2
   RUNG wire#w2
      Contact( #FEED_HOLD_CONDITIONS_HMI )
      I_Contact( #SP.SPEED_REACHED )
      Coil( #HMI_MOTION_EXECUTABILITY_RIGHT )
   END_RUNG
   RUNG wire#w1
      Contact( #SpindleDB.E_TCMinus )
      wire#w3
      Coil( #HMI_MOTION_END_POS_LEFT )
   END_RUNG
   RUNG wire#w1
      Contact( #SP.SPEED_ZERO )
   END_RUNG wire#w3
   RUNG wire#w1
      Contact( #SpindleDB.E_TCPlus )
      Coil( #HMI_MOTION_END_POS_RIGHT )
   END_RUNG
   // the same network as SCL:
   #_w1 := "M_ONE" AND (("DB2001_MODES_GENERAL".MG1.GENERAL.MANUAL_SELECTED AND NOT "DB2001_MODES_GENERAL".MG1.GENERAL.OPTIONS.SGM) OR ("DB2001_MODES_GENERAL".MG1.GENERAL.JOG_SELECTED AND "DB2001_MODES_GENERAL".MG1.GENERAL.OPTIONS.SGM));
   #HMI_MOTION_EXECUTABILITY_LEFT := #_w1 AND NOT #SP.SPEED_ZERO;
   #HMI_MOTION_EXECUTABILITY_RIGHT := #_w1 AND #FEED_HOLD_CONDITIONS_HMI AND NOT #SP.SPEED_REACHED;
   #HMI_MOTION_END_POS_LEFT := "M_ONE" AND (#SpindleDB.E_TCMinus OR #SP.SPEED_ZERO);
   #HMI_MOTION_END_POS_RIGHT := "M_ONE" AND #SpindleDB.E_TCPlus;
END_REGION
END_FUNCTION_BLOCK

FUNCTION_BLOCK "FB33_SAFETY_POSITIONS"   // FB33, LAD
{ S7_Optimized_Access := 'FALSE' }
VERSION : 0.1
// stored: AutoNumber true, IsIECCheckEnabled false, SetENOAutomatically false, UDAEnableTagReadback false
   VAR_INPUT
      MEAS_SYS_1_ACTIVE_REFERENCED : Bool;   // MEASURING SYSTEM 1 ACTIVE AND REFERENCED
      MEAS_SYS_2_ACTIVE_REFERENCED : Bool;   // MEASURING SYSTEM 2 ACTIVE AND REFERENCED
      AXIS_POS : Real;   // AXIS POSITION
   END_VAR
   VAR DB_SPECIFIC
      AX_POS_0_DEGREES : Struct   // AXIS POSITION 0 DEGREES
         TOLERANCE : Real := 0.005;   // TOLERANCE
         POSITION_0_TOLERANCE_PLUS : Real;   // POSITION TOLERANCE PLUS
         POSITION_0_TOLERANCE_MINUS : Real;   // POSITION TOLERANCE MINUS
         POSITION_360_TOLERANCE_PLUS : Real;   // POSITION TOLERANCE PLUS
         POSITION_360_TOLERANCE_MINUS : Real;   // POSITION TOLERANCE MINUS
         IN_POSITION : Bool;   // AXIS POSITION 0 DEGREES
      END_STRUCT;
      AX_POS_90_DEGREES : Struct   // AXIS POSITION 90 DEGREES
         TOLERANCE : Real := 0.005;   // TOLERANCE
         POSITION_TOLERANCE_PLUS : Real;   // POSITION TOLERANCE PLUS
         POSITION_TOLERANCE_MINUS : Real;   // POSITION TOLERANCE MINUS
         IN_POSITION : Bool;   // AXIS POSITION 90 DEGREES
      END_STRUCT;
      AX_POS_180_DEGREES : Struct   // AXIS POSITION 180 DEGREES
         TOLERANCE : Real := 0.005;   // TOLERANCE
         POSITION_TOLERANCE_PLUS : Real;   // POSITION TOLERANCE PLUS
         POSITION_TOLERANCE_MINUS : Real;   // POSITION TOLERANCE MINUS
         IN_POSITION : Bool;   // AXIS POSITION 180 DEGREES
      END_STRUCT;
      AX_POS_270_DEGREES : Struct   // AXIS POSITION 270 DEGREES
         TOLERANCE : Real := 0.005;   // TOLERANCE
         POSITION_TOLERANCE_PLUS : Real;   // POSITION TOLERANCE PLUS
         POSITION_TOLERANCE_MINUS : Real;   // POSITION TOLERANCE MINUS
         IN_POSITION : Bool;   // AXIS POSITION 270 DEGREES
      END_STRUCT;
      AX_POS_MINUS_90_DEGREES : Bool;   // AXIS POSITION MINUS 90 DEGREES
      AX_POS_MINUS_180_DEGREES : Bool;   // AXIS POSITION MINUS 180 DEGREES
      AX_POS_MINUS_270_DEGREES : Bool;   // AXIS POSITION MINUS 270 DEGREES
      SAFETY_POSITION_1 : Struct   // HOME POSITION
         HMI_POSITION : Real := 1.1;   // HMI POSITION
         TOLERANCE_PLUS : Real := 0.01;   // TOLERANCE PLUS
         TOLERANCE_MINUS : Real := 0.01;   // TOLERANCE MINUS
         POSITION_TOLERANCE_PLUS : Real;   // POSITION TOLERANCE PLUS
         POSITION_TOLERANCE_MINUS : Real;   // POSITION TOLERANCE MINUS
         IN_POSITION : Bool;   // HOME POSITION
         GREATER_TOLERANCE_PLUS : Bool;   // GREATER THAN TOLERANCE PLUS
         GREATER_TOLERANCE_MINUS : Bool;   // GREATER TOLERANCE MINUS
         LOWER_TOLERANCE_PLUS : Bool;   // LOWER TOLERANCE PLUS
         LOWER_TOLERANCE_MINUS : Bool;   // LOWER TOLERANCE MINUS
      END_STRUCT;
      SAFETY_POSITION_2 : Struct   // CLEAR FIXTURE AXIS
         HMI_POSITION : Real := 1.1;   // HMI POSITION
         TOLERANCE_PLUS : Real := 0.01;   // TOLERANCE PLUS
         TOLERANCE_MINUS : Real := 0.01;   // TOLERANCE MINUS
         POSITION_TOLERANCE_PLUS : Real;   // POSITION TOLERANCE PLUS
         POSITION_TOLERANCE_MINUS : Real;   // POSITION TOLERANCE MINUS
         IN_POSITION : Bool;   // IN POSITION
         GREATER_TOLERANCE_PLUS : Bool;   // GREATER TOLERANCE PLUS
         GREATER_TOLERANCE_MINUS : Bool;   // CLEAR FIXTURE AXIS
         LOWER_TOLERANCE_PLUS : Bool;   // LOWER TOLERANCE PLUS
         LOWER_TOLERANCE_MINUS : Bool;   // LOWER TOLERANCE MINUS
      END_STRUCT;
      SAFETY_POSITION_3 : Struct   // TOOL CHANGE POSITION
         HMI_POSITION : Real := 1.1;   // HMI POSITION
         TOLERANCE_PLUS : Real := 0.01;   // TOLERANCE
         TOLERANCE_MINUS : Real := 0.01;   // TOLERANCE MINUS
         POSITION_TOLERANCE_PLUS : Real;   // POSITION TOLERANCE PLUS
         POSITION_TOLERANCE_MINUS : Real;   // POSITION TOLERANCE MINUS
         IN_POSITION : Bool;   // TOOL CHANGE POSITION
         GREATER_TOLERANCE_PLUS : Bool;   // GREATER TOLERANCE PLUS
         GREATER_TOLERANCE_MINUS : Bool;   // GREATER TOLERANCE MINUS
         LOWER_TOLERANCE_PLUS : Bool;   // LOWER TOLERANCE PLUS
         LOWER_TOLERANCE_MINUS : Bool;   // LOWER TOLERANCE MINUS
      END_STRUCT;
      SAFETY_POSITION_4 : Struct   // RETURNED
         HMI_POSITION : Real := 1.1;   // HMI POSITION
         TOLERANCE_PLUS : Real := 0.01;   // TOLERANCE PLUS
         TOLERANCE_MINUS : Real := 0.01;   // TOLERANCE MINUS
         POSITION_TOLERANCE_PLUS : Real;   // POSITION TOLERANCE PLUS
         POSITION_TOLERANCE_MINUS : Real;   // POSITION TOLERANCE MINUS
         IN_POSITION : Bool;   // RETURNED
         GREATER_TOLERANCE_PLUS : Bool;   // GREATER TOLERANCE PLUS
         GREATER_TOLERANCE_MINUS : Bool;   // GREATER TOLERANCE MINUS
         LOWER_TOLERANCE_PLUS : Bool;   // LOWER TOLERANCE PLUS
         LOWER_TOLERANCE_MINUS : Bool;   // LOWER TOLERANCE MINUS
      END_STRUCT;
      SAFETY_POSITION_5 : Struct   // ADVANCED
         HMI_POSITION : Real := 1.1;   // HMI POSITION
         TOLERANCE_PLUS : Real := 0.01;   // TOLERANCE_PLUS
         TOLERANCE_MINUS : Real := 0.01;   // TOLERANCE MINUS
         POSITION_TOLERANCE_PLUS : Real;   // POSITION TOLERANCE PLUS
         POSITION_TOLERANCE_MINUS : Real;   // POSITION TOLERANCE MINUS
         IN_POSITION : Bool;   // ADVANCED
         GREATER_TOLERANCE_PLUS : Bool;   // GREATER TOLERANCE PLUS
         GREATER_TOLERANCE_MINUS : Bool;   // GREATER TOLERANCE MINUS
         LOWER_TOLERANCE_PLUS : Bool;   // LOWER TOLERANCE PLUS
         LOWER_TOLERANCE_MINUS : Bool;   // LOWER TOLERANCE MINUS
      END_STRUCT;
      SAFETY_POSITION_6 : Struct
         HMI_POSITION : Real := 1.1;   // HMI POSITION
         TOLERANCE_PLUS : Real := 0.01;   // TOLERANCE PLUS
         TOLERANCE_MINUS : Real := 0.01;   // TOLERANCE MINUS
         POSITION_TOLERANCE_PLUS : Real;   // POSITION TOLERANCE PLUS
         POSITION_TOLERANCE_MINUS : Real;   // POSITION TOLERANCE MINUS
         IN_POSITION : Bool;   // IN POSITION
         GREATER_TOLERANCE_PLUS : Bool;   // GREATER TOLERANCE PLUS
         GREATER_TOLERANCE_MINUS : Bool;   // GREATER TOLERANCE MINUS
         LOWER_TOLERANCE_PLUS : Bool;   // LOWER TOLERANCE PLUS
         LOWER_TOLERANCE_MINUS : Bool;   // LOWER TOLERANCE MINUS
      END_STRUCT;
      SAFETY_POSITION_7 : Struct
         HMI_POSITION : Real := 1.1;   // HMI POSITION
         TOLERANCE_PLUS : Real := 0.01;   // TOLERANCE PLUS
         TOLERANCE_MINUS : Real := 0.01;   // TOLERANCE MINUS
         POSITION_TOLERANCE_PLUS : Real;   // POSITION TOLERANCE PLUS
         POSITION_TOLERANCE_MINUS : Real;   // POSITION TOLERANCE MINUS
         IN_POSITION : Bool;   // IN POSITION
         GREATER_TOLERANCE_PLUS : Bool;   // GREATER TOLERANCE PLUS
         GREATER_TOLERANCE_MINUS : Bool;   // GREATER TOLERANCE MINUS
         LOWER_TOLERANCE_PLUS : Bool;   // LOWER TOLERANCE PLUS
         LOWER_TOLERANCE_MINUS : Bool;   // LOWER TOLERANCE MINUS
      END_STRUCT;
      SAFETY_POSITION_8 : Struct
         HMI_POSITION : Real := 1.1;   // HMI POSITION
         TOLERANCE_PLUS : Real := 0.01;   // TOLERANCE PLUS
         TOLERANCE_MINUS : Real := 0.01;   // TOLERANCE MINUS
         POSITION_TOLERANCE_PLUS : Real;   // POSITION TOLERANCE PLUS
         POSITION_TOLERANCE_MINUS : Real;   // POSITION TOLERANCE MINUS
         IN_POSITION : Bool;   // IN POSITION
         GREATER_TOLERANCE_PLUS : Bool;   // GREATER TOLERANCE PLUS
         GREATER_TOLERANCE_MINUS : Bool;   // GREATER TOLERANCE MINUS
         LOWER_TOLERANCE_PLUS : Bool;   // LOWER TOLERANCE PLUS
         LOWER_TOLERANCE_MINUS : Bool;   // LOWER TOLERANCE MINUS
      END_STRUCT;
      SAFETY_POSITION_9 : Struct
         HMI_POSITION : Real := 1.1;   // HMI POSITION
         TOLERANCE_PLUS : Real := 0.01;   // TOLERANCE PLUS
         TOLERANCE_MINUS : Real := 0.01;   // TOLERANCE MINUS
         POSITION_TOLERANCE_PLUS : Real;   // POSITION TOLERANCE PLUS
         POSITION_TOLERANCE_MINUS : Real;   // POSITION TOLERANCE MINUS
         IN_POSITION : Bool;   // IN POSITION
         GREATER_TOLERANCE_PLUS : Bool;   // GREATER TOLERANCE PLUS
         GREATER_TOLERANCE_MINUS : Bool;   // GREATER TOLERANCE MINUS
         LOWER_TOLERANCE_PLUS : Bool;   // LOWER TOLERANCE PLUS
         LOWER_TOLERANCE_MINUS : Bool;   // LOWER TOLERANCE MINUS
      END_STRUCT;
      SAFETY_POSITION_10 : Struct
         HMI_POSITION : Real := 1.1;   // HMI POSITION
         TOLERANCE_PLUS : Real := 0.01;   // TOLERANCE PLUS
         TOLERANCE_MINUS : Real := 0.01;   // TOLERANCE MINUS
         POSITION_TOLERANCE_PLUS : Real;   // POSITION TOLERANCE PLUS
         POSITION_TOLERANCE_MINUS : Real;   // POSITION TOLERANCE MINUS
         IN_POSITION : Bool;   // IN POSITION
         GREATER_TOLERANCE_PLUS : Bool;   // GREATER TOLERANCE PLUS
         GREATER_TOLERANCE_MINUS : Bool;   // GREATER TOLERANCE MINUS
         LOWER_TOLERANCE_PLUS : Bool;   // LOWER TOLERANCE PLUS
         LOWER_TOLERANCE_MINUS : Bool;   // LOWER TOLERANCE MINUS
      END_STRUCT;
   END_VAR
   VAR_TEMP   // added for the SCL form of the ladder/FBD networks
      _w1 : Bool;
      _w2 : Bool;
   END_VAR
BEGIN

REGION Network 1: AXIS POSITION 0 DEGREES
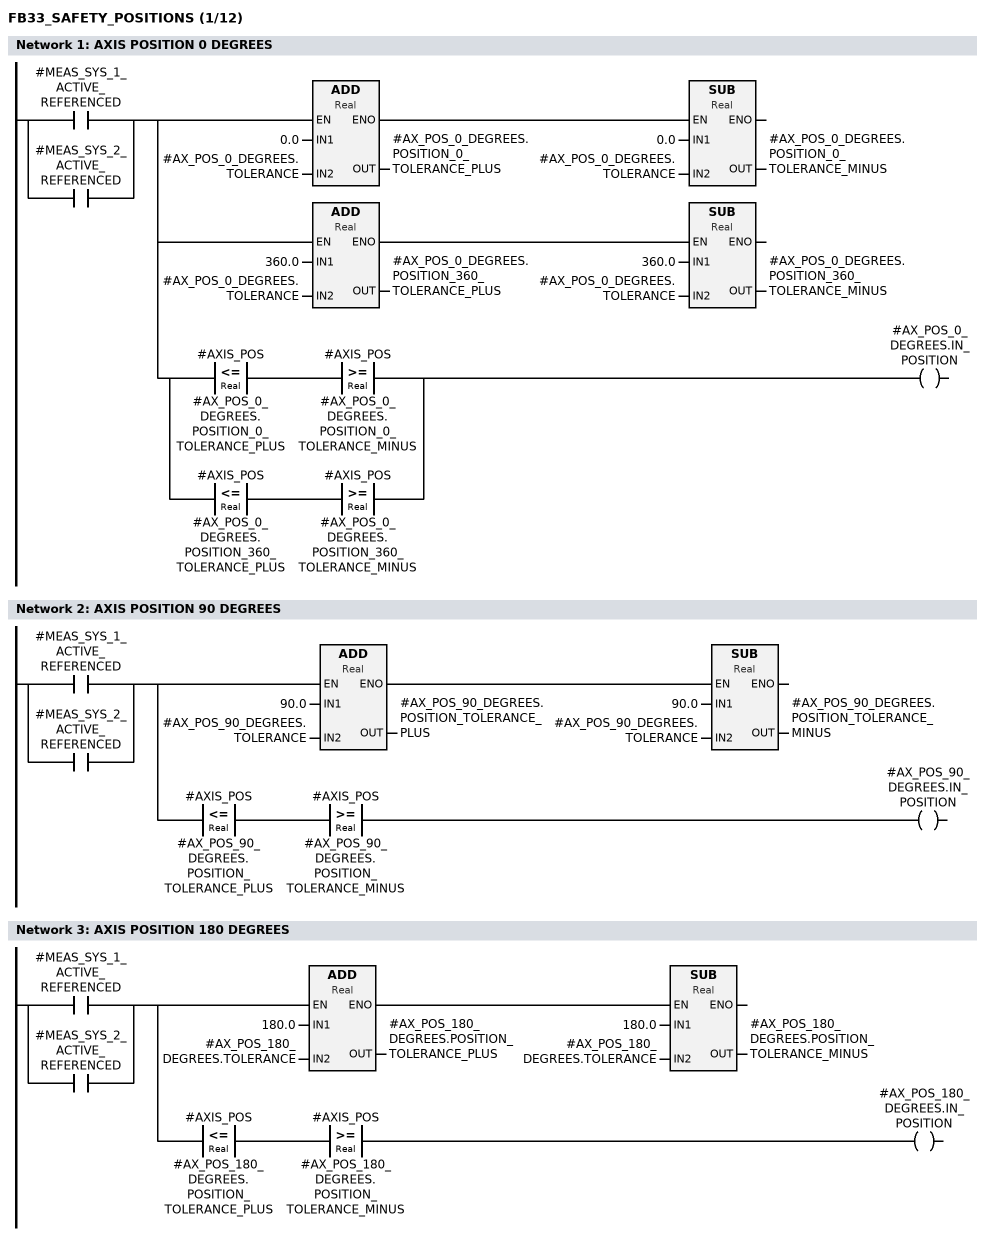
   RUNG wire#powerrail
      Contact( #MEAS_SYS_1_ACTIVE_REFERENCED )
      wire#w1
      { S7_Templates := "SrcType := Real"; S7_GenerateENO := "TRUE" } Add(in1 := 0.0, in2 := #AX_POS_0_DEGREES.TOLERANCE, out => #AX_POS_0_DEGREES.POSITION_0_TOLERANCE_PLUS)
      { S7_Templates := "SrcType := Real"; S7_GenerateENO := "TRUE" } Sub(in1 := 0.0, in2 := #AX_POS_0_DEGREES.TOLERANCE, out => #AX_POS_0_DEGREES.POSITION_0_TOLERANCE_MINUS)
   END_RUNG
   RUNG wire#powerrail
      Contact( #MEAS_SYS_2_ACTIVE_REFERENCED )
   END_RUNG wire#w1
   RUNG wire#w1
      { S7_Templates := "SrcType := Real"; S7_GenerateENO := "TRUE" } Add(in1 := 360.0, in2 := #AX_POS_0_DEGREES.TOLERANCE, out => #AX_POS_0_DEGREES.POSITION_360_TOLERANCE_PLUS)
      { S7_Templates := "SrcType := Real"; S7_GenerateENO := "TRUE" } Sub(in1 := 360.0, in2 := #AX_POS_0_DEGREES.TOLERANCE, out => #AX_POS_0_DEGREES.POSITION_360_TOLERANCE_MINUS)
   END_RUNG
   RUNG wire#w1
      { S7_Templates := "SrcType := Real" } LE_Contact(in1 := #AXIS_POS, in2 := #AX_POS_0_DEGREES.POSITION_0_TOLERANCE_PLUS)
      { S7_Templates := "SrcType := Real" } GE_Contact(in1 := #AXIS_POS, in2 := #AX_POS_0_DEGREES.POSITION_0_TOLERANCE_MINUS)
      wire#w2
      Coil( #AX_POS_0_DEGREES.IN_POSITION )
   END_RUNG
   RUNG wire#w1
      { S7_Templates := "SrcType := Real" } LE_Contact(in1 := #AXIS_POS, in2 := #AX_POS_0_DEGREES.POSITION_360_TOLERANCE_PLUS)
      { S7_Templates := "SrcType := Real" } GE_Contact(in1 := #AXIS_POS, in2 := #AX_POS_0_DEGREES.POSITION_360_TOLERANCE_MINUS)
   END_RUNG wire#w2
   // the same network as SCL:
   // ENO of a box is taken as its EN; it also drops when the box reports an error
   #_w1 := #MEAS_SYS_1_ACTIVE_REFERENCED OR #MEAS_SYS_2_ACTIVE_REFERENCED;
   IF #_w1 THEN
       #AX_POS_0_DEGREES.POSITION_0_TOLERANCE_PLUS := 0.0 + #AX_POS_0_DEGREES.TOLERANCE;
       #AX_POS_0_DEGREES.POSITION_0_TOLERANCE_MINUS := 0.0 - #AX_POS_0_DEGREES.TOLERANCE;
       #AX_POS_0_DEGREES.POSITION_360_TOLERANCE_PLUS := 360.0 + #AX_POS_0_DEGREES.TOLERANCE;
       #AX_POS_0_DEGREES.POSITION_360_TOLERANCE_MINUS := 360.0 - #AX_POS_0_DEGREES.TOLERANCE;
   END_IF;
   #AX_POS_0_DEGREES.IN_POSITION := #_w1 AND (((#AXIS_POS <= #AX_POS_0_DEGREES.POSITION_0_TOLERANCE_PLUS) AND (#AXIS_POS >= #AX_POS_0_DEGREES.POSITION_0_TOLERANCE_MINUS)) OR ((#AXIS_POS <= #AX_POS_0_DEGREES.POSITION_360_TOLERANCE_PLUS) AND (#AXIS_POS >= #AX_POS_0_DEGREES.POSITION_360_TOLERANCE_MINUS)));
END_REGION

REGION Network 2: AXIS POSITION 90 DEGREES
   RUNG wire#powerrail
      Contact( #MEAS_SYS_1_ACTIVE_REFERENCED )
      wire#w1
      { S7_Templates := "SrcType := Real"; S7_GenerateENO := "TRUE" } Add(in1 := 90.0, in2 := #AX_POS_90_DEGREES.TOLERANCE, out => #AX_POS_90_DEGREES.POSITION_TOLERANCE_PLUS)
      { S7_Templates := "SrcType := Real"; S7_GenerateENO := "TRUE" } Sub(in1 := 90.0, in2 := #AX_POS_90_DEGREES.TOLERANCE, out => #AX_POS_90_DEGREES.POSITION_TOLERANCE_MINUS)
   END_RUNG
   RUNG wire#powerrail
      Contact( #MEAS_SYS_2_ACTIVE_REFERENCED )
   END_RUNG wire#w1
   RUNG wire#w1
      { S7_Templates := "SrcType := Real" } LE_Contact(in1 := #AXIS_POS, in2 := #AX_POS_90_DEGREES.POSITION_TOLERANCE_PLUS)
      { S7_Templates := "SrcType := Real" } GE_Contact(in1 := #AXIS_POS, in2 := #AX_POS_90_DEGREES.POSITION_TOLERANCE_MINUS)
      Coil( #AX_POS_90_DEGREES.IN_POSITION )
   END_RUNG
   // the same network as SCL:
   // ENO of a box is taken as its EN; it also drops when the box reports an error
   #_w1 := #MEAS_SYS_1_ACTIVE_REFERENCED OR #MEAS_SYS_2_ACTIVE_REFERENCED;
   IF #_w1 THEN
       #AX_POS_90_DEGREES.POSITION_TOLERANCE_PLUS := 90.0 + #AX_POS_90_DEGREES.TOLERANCE;
       #AX_POS_90_DEGREES.POSITION_TOLERANCE_MINUS := 90.0 - #AX_POS_90_DEGREES.TOLERANCE;
   END_IF;
   #AX_POS_90_DEGREES.IN_POSITION := #_w1 AND (#AXIS_POS <= #AX_POS_90_DEGREES.POSITION_TOLERANCE_PLUS) AND (#AXIS_POS >= #AX_POS_90_DEGREES.POSITION_TOLERANCE_MINUS);
END_REGION

REGION Network 3: AXIS POSITION 180 DEGREES
   RUNG wire#powerrail
      Contact( #MEAS_SYS_1_ACTIVE_REFERENCED )
      wire#w1
      { S7_Templates := "SrcType := Real"; S7_GenerateENO := "TRUE" } Add(in1 := 180.0, in2 := #AX_POS_180_DEGREES.TOLERANCE, out => #AX_POS_180_DEGREES.POSITION_TOLERANCE_PLUS)
      { S7_Templates := "SrcType := Real"; S7_GenerateENO := "TRUE" } Sub(in1 := 180.0, in2 := #AX_POS_180_DEGREES.TOLERANCE, out => #AX_POS_180_DEGREES.POSITION_TOLERANCE_MINUS)
   END_RUNG
   RUNG wire#powerrail
      Contact( #MEAS_SYS_2_ACTIVE_REFERENCED )
   END_RUNG wire#w1
   RUNG wire#w1
      { S7_Templates := "SrcType := Real" } LE_Contact(in1 := #AXIS_POS, in2 := #AX_POS_180_DEGREES.POSITION_TOLERANCE_PLUS)
      { S7_Templates := "SrcType := Real" } GE_Contact(in1 := #AXIS_POS, in2 := #AX_POS_180_DEGREES.POSITION_TOLERANCE_MINUS)
      Coil( #AX_POS_180_DEGREES.IN_POSITION )
   END_RUNG
   // the same network as SCL:
   // ENO of a box is taken as its EN; it also drops when the box reports an error
   #_w1 := #MEAS_SYS_1_ACTIVE_REFERENCED OR #MEAS_SYS_2_ACTIVE_REFERENCED;
   IF #_w1 THEN
       #AX_POS_180_DEGREES.POSITION_TOLERANCE_PLUS := 180.0 + #AX_POS_180_DEGREES.TOLERANCE;
       #AX_POS_180_DEGREES.POSITION_TOLERANCE_MINUS := 180.0 - #AX_POS_180_DEGREES.TOLERANCE;
   END_IF;
   #AX_POS_180_DEGREES.IN_POSITION := #_w1 AND (#AXIS_POS <= #AX_POS_180_DEGREES.POSITION_TOLERANCE_PLUS) AND (#AXIS_POS >= #AX_POS_180_DEGREES.POSITION_TOLERANCE_MINUS);
END_REGION

REGION Network 4: AXIS POSITION 270 DEGREES
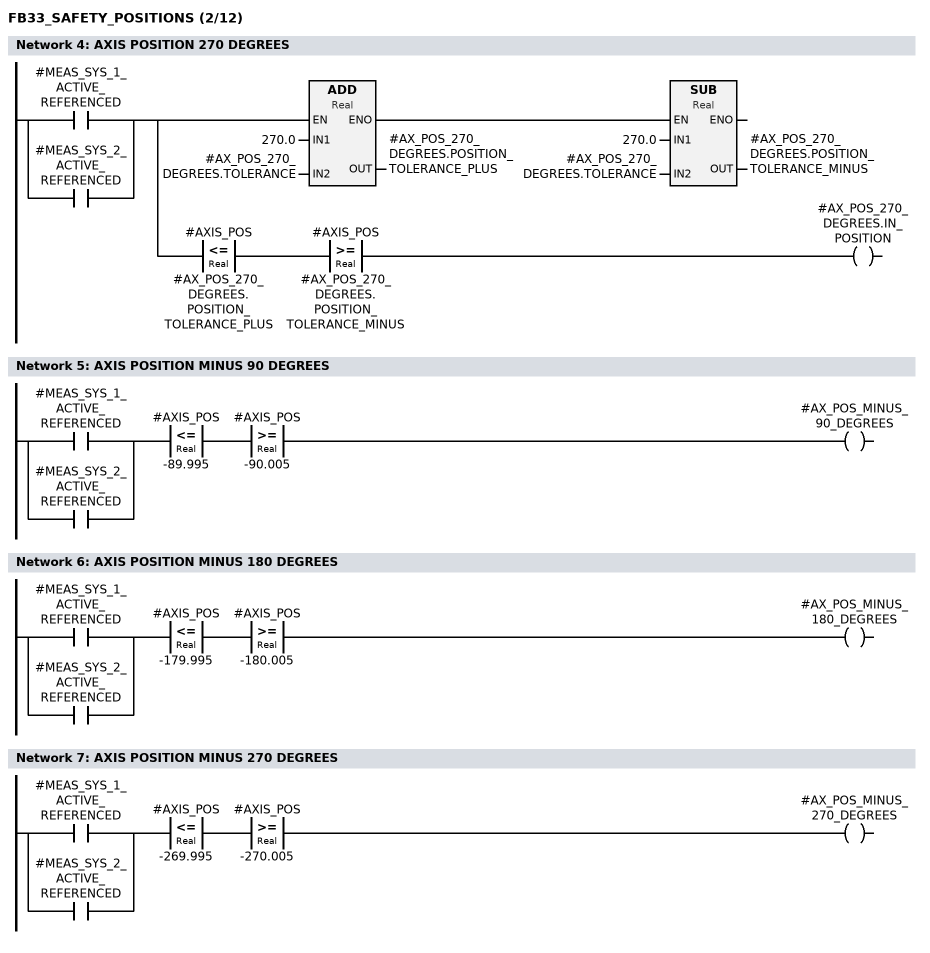
   RUNG wire#powerrail
      Contact( #MEAS_SYS_1_ACTIVE_REFERENCED )
      wire#w1
      { S7_Templates := "SrcType := Real"; S7_GenerateENO := "TRUE" } Add(in1 := 270.0, in2 := #AX_POS_270_DEGREES.TOLERANCE, out => #AX_POS_270_DEGREES.POSITION_TOLERANCE_PLUS)
      { S7_Templates := "SrcType := Real"; S7_GenerateENO := "TRUE" } Sub(in1 := 270.0, in2 := #AX_POS_270_DEGREES.TOLERANCE, out => #AX_POS_270_DEGREES.POSITION_TOLERANCE_MINUS)
   END_RUNG
   RUNG wire#powerrail
      Contact( #MEAS_SYS_2_ACTIVE_REFERENCED )
   END_RUNG wire#w1
   RUNG wire#w1
      { S7_Templates := "SrcType := Real" } LE_Contact(in1 := #AXIS_POS, in2 := #AX_POS_270_DEGREES.POSITION_TOLERANCE_PLUS)
      { S7_Templates := "SrcType := Real" } GE_Contact(in1 := #AXIS_POS, in2 := #AX_POS_270_DEGREES.POSITION_TOLERANCE_MINUS)
      Coil( #AX_POS_270_DEGREES.IN_POSITION )
   END_RUNG
   // the same network as SCL:
   // ENO of a box is taken as its EN; it also drops when the box reports an error
   #_w1 := #MEAS_SYS_1_ACTIVE_REFERENCED OR #MEAS_SYS_2_ACTIVE_REFERENCED;
   IF #_w1 THEN
       #AX_POS_270_DEGREES.POSITION_TOLERANCE_PLUS := 270.0 + #AX_POS_270_DEGREES.TOLERANCE;
       #AX_POS_270_DEGREES.POSITION_TOLERANCE_MINUS := 270.0 - #AX_POS_270_DEGREES.TOLERANCE;
   END_IF;
   #AX_POS_270_DEGREES.IN_POSITION := #_w1 AND (#AXIS_POS <= #AX_POS_270_DEGREES.POSITION_TOLERANCE_PLUS) AND (#AXIS_POS >= #AX_POS_270_DEGREES.POSITION_TOLERANCE_MINUS);
END_REGION

REGION Network 5: AXIS POSITION MINUS 90 DEGREES
   RUNG wire#powerrail
      Contact( #MEAS_SYS_1_ACTIVE_REFERENCED )
      wire#w1
      { S7_Templates := "SrcType := Real" } LE_Contact(in1 := #AXIS_POS, in2 := -89.995)
      { S7_Templates := "SrcType := Real" } GE_Contact(in1 := #AXIS_POS, in2 := -90.005)
      Coil( #AX_POS_MINUS_90_DEGREES )
   END_RUNG
   RUNG wire#powerrail
      Contact( #MEAS_SYS_2_ACTIVE_REFERENCED )
   END_RUNG wire#w1
   // the same network as SCL:
   #AX_POS_MINUS_90_DEGREES := (#MEAS_SYS_1_ACTIVE_REFERENCED OR #MEAS_SYS_2_ACTIVE_REFERENCED) AND (#AXIS_POS <= (-89.995)) AND (#AXIS_POS >= (-90.005));
END_REGION

REGION Network 6: AXIS POSITION MINUS 180 DEGREES
   RUNG wire#powerrail
      Contact( #MEAS_SYS_1_ACTIVE_REFERENCED )
      wire#w1
      { S7_Templates := "SrcType := Real" } LE_Contact(in1 := #AXIS_POS, in2 := -179.995)
      { S7_Templates := "SrcType := Real" } GE_Contact(in1 := #AXIS_POS, in2 := -180.005)
      Coil( #AX_POS_MINUS_180_DEGREES )
   END_RUNG
   RUNG wire#powerrail
      Contact( #MEAS_SYS_2_ACTIVE_REFERENCED )
   END_RUNG wire#w1
   // the same network as SCL:
   #AX_POS_MINUS_180_DEGREES := (#MEAS_SYS_1_ACTIVE_REFERENCED OR #MEAS_SYS_2_ACTIVE_REFERENCED) AND (#AXIS_POS <= (-179.995)) AND (#AXIS_POS >= (-180.005));
END_REGION

REGION Network 7: AXIS POSITION MINUS 270 DEGREES
   RUNG wire#powerrail
      Contact( #MEAS_SYS_1_ACTIVE_REFERENCED )
      wire#w1
      { S7_Templates := "SrcType := Real" } LE_Contact(in1 := #AXIS_POS, in2 := -269.995)
      { S7_Templates := "SrcType := Real" } GE_Contact(in1 := #AXIS_POS, in2 := -270.005)
      Coil( #AX_POS_MINUS_270_DEGREES )
   END_RUNG
   RUNG wire#powerrail
      Contact( #MEAS_SYS_2_ACTIVE_REFERENCED )
   END_RUNG wire#w1
   // the same network as SCL:
   #AX_POS_MINUS_270_DEGREES := (#MEAS_SYS_1_ACTIVE_REFERENCED OR #MEAS_SYS_2_ACTIVE_REFERENCED) AND (#AXIS_POS <= (-269.995)) AND (#AXIS_POS >= (-270.005));
END_REGION

REGION Network 8: SAFETY POSITION 1
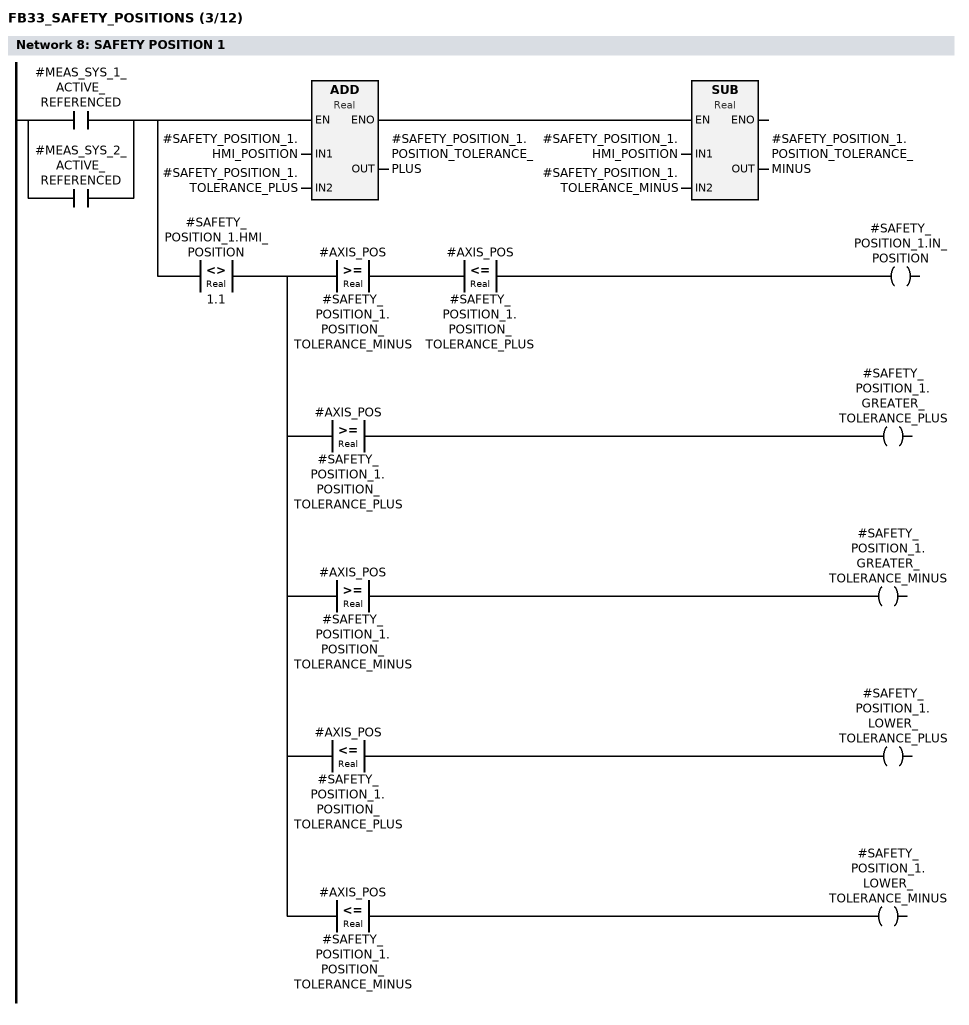
   RUNG wire#powerrail
      Contact( #MEAS_SYS_1_ACTIVE_REFERENCED )
      wire#w1
      { S7_Templates := "SrcType := Real"; S7_GenerateENO := "TRUE" } Add(in1 := #SAFETY_POSITION_1.HMI_POSITION, in2 := #SAFETY_POSITION_1.TOLERANCE_PLUS, out => #SAFETY_POSITION_1.POSITION_TOLERANCE_PLUS)
      { S7_Templates := "SrcType := Real"; S7_GenerateENO := "TRUE" } Sub(in1 := #SAFETY_POSITION_1.HMI_POSITION, in2 := #SAFETY_POSITION_1.TOLERANCE_MINUS, out => #SAFETY_POSITION_1.POSITION_TOLERANCE_MINUS)
   END_RUNG
   RUNG wire#powerrail
      Contact( #MEAS_SYS_2_ACTIVE_REFERENCED )
   END_RUNG wire#w1
   RUNG wire#w1
      { S7_Templates := "SrcType := Real" } NE_Contact(in1 := #SAFETY_POSITION_1.HMI_POSITION, in2 := 1.1)
      wire#w2
      { S7_Templates := "SrcType := Real" } GE_Contact(in1 := #AXIS_POS, in2 := #SAFETY_POSITION_1.POSITION_TOLERANCE_MINUS)
      { S7_Templates := "SrcType := Real" } LE_Contact(in1 := #AXIS_POS, in2 := #SAFETY_POSITION_1.POSITION_TOLERANCE_PLUS)
      Coil( #SAFETY_POSITION_1.IN_POSITION )
   END_RUNG
   RUNG wire#w2
      { S7_Templates := "SrcType := Real" } GE_Contact(in1 := #AXIS_POS, in2 := #SAFETY_POSITION_1.POSITION_TOLERANCE_PLUS)
      Coil( #SAFETY_POSITION_1.GREATER_TOLERANCE_PLUS )
   END_RUNG
   RUNG wire#w2
      { S7_Templates := "SrcType := Real" } GE_Contact(in1 := #AXIS_POS, in2 := #SAFETY_POSITION_1.POSITION_TOLERANCE_MINUS)
      Coil( #SAFETY_POSITION_1.GREATER_TOLERANCE_MINUS )
   END_RUNG
   RUNG wire#w2
      { S7_Templates := "SrcType := Real" } LE_Contact(in1 := #AXIS_POS, in2 := #SAFETY_POSITION_1.POSITION_TOLERANCE_PLUS)
      Coil( #SAFETY_POSITION_1.LOWER_TOLERANCE_PLUS )
   END_RUNG
   RUNG wire#w2
      { S7_Templates := "SrcType := Real" } LE_Contact(in1 := #AXIS_POS, in2 := #SAFETY_POSITION_1.POSITION_TOLERANCE_MINUS)
      Coil( #SAFETY_POSITION_1.LOWER_TOLERANCE_MINUS )
   END_RUNG
   // the same network as SCL:
   // ENO of a box is taken as its EN; it also drops when the box reports an error
   #_w1 := #MEAS_SYS_1_ACTIVE_REFERENCED OR #MEAS_SYS_2_ACTIVE_REFERENCED;
   IF #_w1 THEN
       #SAFETY_POSITION_1.POSITION_TOLERANCE_PLUS := #SAFETY_POSITION_1.HMI_POSITION + #SAFETY_POSITION_1.TOLERANCE_PLUS;
       #SAFETY_POSITION_1.POSITION_TOLERANCE_MINUS := #SAFETY_POSITION_1.HMI_POSITION - #SAFETY_POSITION_1.TOLERANCE_MINUS;
   END_IF;
   #_w2 := #_w1 AND (#SAFETY_POSITION_1.HMI_POSITION <> 1.1);
   #SAFETY_POSITION_1.IN_POSITION := #_w2 AND (#AXIS_POS >= #SAFETY_POSITION_1.POSITION_TOLERANCE_MINUS) AND (#AXIS_POS <= #SAFETY_POSITION_1.POSITION_TOLERANCE_PLUS);
   #SAFETY_POSITION_1.GREATER_TOLERANCE_PLUS := #_w2 AND (#AXIS_POS >= #SAFETY_POSITION_1.POSITION_TOLERANCE_PLUS);
   #SAFETY_POSITION_1.GREATER_TOLERANCE_MINUS := #_w2 AND (#AXIS_POS >= #SAFETY_POSITION_1.POSITION_TOLERANCE_MINUS);
   #SAFETY_POSITION_1.LOWER_TOLERANCE_PLUS := #_w2 AND (#AXIS_POS <= #SAFETY_POSITION_1.POSITION_TOLERANCE_PLUS);
   #SAFETY_POSITION_1.LOWER_TOLERANCE_MINUS := #_w2 AND (#AXIS_POS <= #SAFETY_POSITION_1.POSITION_TOLERANCE_MINUS);
END_REGION

REGION Network 9: SAFETY POSITION 2
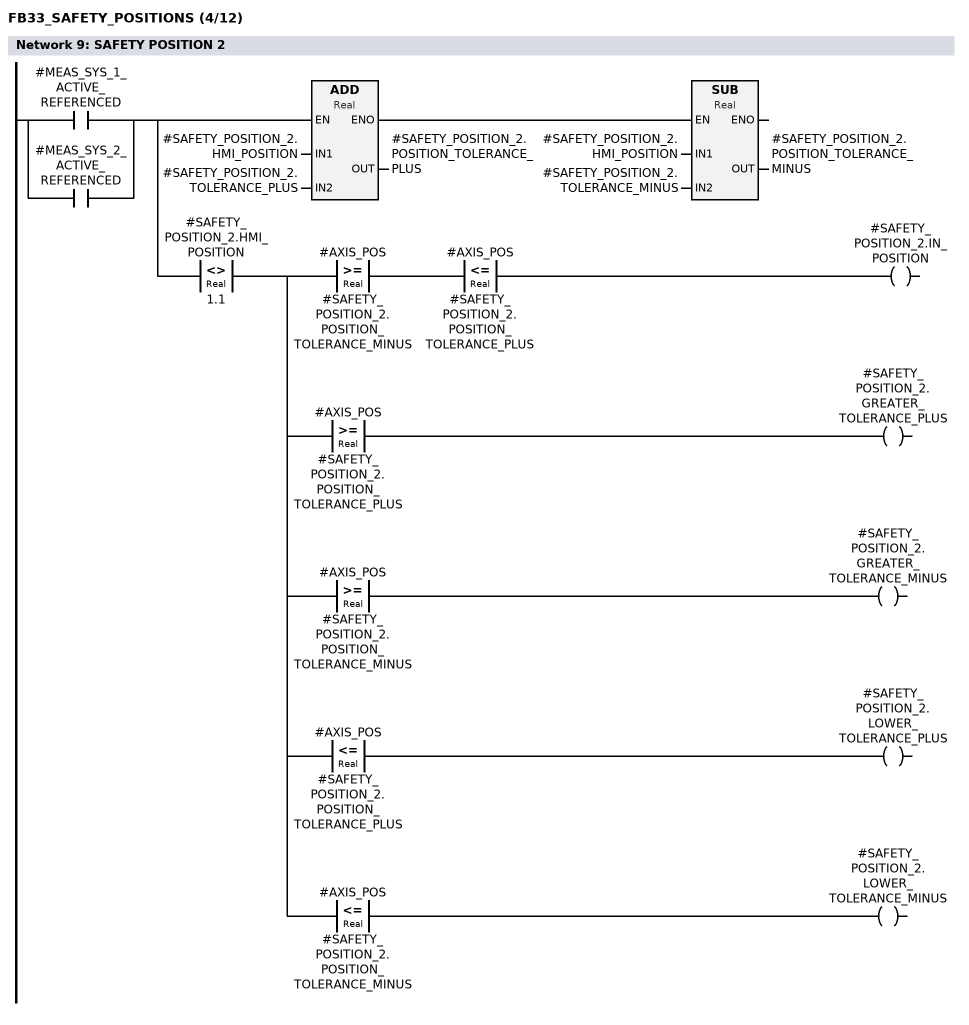
   RUNG wire#powerrail
      Contact( #MEAS_SYS_1_ACTIVE_REFERENCED )
      wire#w1
      { S7_Templates := "SrcType := Real"; S7_GenerateENO := "TRUE" } Add(in1 := #SAFETY_POSITION_2.HMI_POSITION, in2 := #SAFETY_POSITION_2.TOLERANCE_PLUS, out => #SAFETY_POSITION_2.POSITION_TOLERANCE_PLUS)
      { S7_Templates := "SrcType := Real"; S7_GenerateENO := "TRUE" } Sub(in1 := #SAFETY_POSITION_2.HMI_POSITION, in2 := #SAFETY_POSITION_2.TOLERANCE_MINUS, out => #SAFETY_POSITION_2.POSITION_TOLERANCE_MINUS)
   END_RUNG
   RUNG wire#powerrail
      Contact( #MEAS_SYS_2_ACTIVE_REFERENCED )
   END_RUNG wire#w1
   RUNG wire#w1
      { S7_Templates := "SrcType := Real" } NE_Contact(in1 := #SAFETY_POSITION_2.HMI_POSITION, in2 := 1.1)
      wire#w2
      { S7_Templates := "SrcType := Real" } GE_Contact(in1 := #AXIS_POS, in2 := #SAFETY_POSITION_2.POSITION_TOLERANCE_MINUS)
      { S7_Templates := "SrcType := Real" } LE_Contact(in1 := #AXIS_POS, in2 := #SAFETY_POSITION_2.POSITION_TOLERANCE_PLUS)
      Coil( #SAFETY_POSITION_2.IN_POSITION )
   END_RUNG
   RUNG wire#w2
      { S7_Templates := "SrcType := Real" } GE_Contact(in1 := #AXIS_POS, in2 := #SAFETY_POSITION_2.POSITION_TOLERANCE_PLUS)
      Coil( #SAFETY_POSITION_2.GREATER_TOLERANCE_PLUS )
   END_RUNG
   RUNG wire#w2
      { S7_Templates := "SrcType := Real" } GE_Contact(in1 := #AXIS_POS, in2 := #SAFETY_POSITION_2.POSITION_TOLERANCE_MINUS)
      Coil( #SAFETY_POSITION_2.GREATER_TOLERANCE_MINUS )
   END_RUNG
   RUNG wire#w2
      { S7_Templates := "SrcType := Real" } LE_Contact(in1 := #AXIS_POS, in2 := #SAFETY_POSITION_2.POSITION_TOLERANCE_PLUS)
      Coil( #SAFETY_POSITION_2.LOWER_TOLERANCE_PLUS )
   END_RUNG
   RUNG wire#w2
      { S7_Templates := "SrcType := Real" } LE_Contact(in1 := #AXIS_POS, in2 := #SAFETY_POSITION_2.POSITION_TOLERANCE_MINUS)
      Coil( #SAFETY_POSITION_2.LOWER_TOLERANCE_MINUS )
   END_RUNG
   // the same network as SCL:
   // ENO of a box is taken as its EN; it also drops when the box reports an error
   #_w1 := #MEAS_SYS_1_ACTIVE_REFERENCED OR #MEAS_SYS_2_ACTIVE_REFERENCED;
   IF #_w1 THEN
       #SAFETY_POSITION_2.POSITION_TOLERANCE_PLUS := #SAFETY_POSITION_2.HMI_POSITION + #SAFETY_POSITION_2.TOLERANCE_PLUS;
       #SAFETY_POSITION_2.POSITION_TOLERANCE_MINUS := #SAFETY_POSITION_2.HMI_POSITION - #SAFETY_POSITION_2.TOLERANCE_MINUS;
   END_IF;
   #_w2 := #_w1 AND (#SAFETY_POSITION_2.HMI_POSITION <> 1.1);
   #SAFETY_POSITION_2.IN_POSITION := #_w2 AND (#AXIS_POS >= #SAFETY_POSITION_2.POSITION_TOLERANCE_MINUS) AND (#AXIS_POS <= #SAFETY_POSITION_2.POSITION_TOLERANCE_PLUS);
   #SAFETY_POSITION_2.GREATER_TOLERANCE_PLUS := #_w2 AND (#AXIS_POS >= #SAFETY_POSITION_2.POSITION_TOLERANCE_PLUS);
   #SAFETY_POSITION_2.GREATER_TOLERANCE_MINUS := #_w2 AND (#AXIS_POS >= #SAFETY_POSITION_2.POSITION_TOLERANCE_MINUS);
   #SAFETY_POSITION_2.LOWER_TOLERANCE_PLUS := #_w2 AND (#AXIS_POS <= #SAFETY_POSITION_2.POSITION_TOLERANCE_PLUS);
   #SAFETY_POSITION_2.LOWER_TOLERANCE_MINUS := #_w2 AND (#AXIS_POS <= #SAFETY_POSITION_2.POSITION_TOLERANCE_MINUS);
END_REGION

REGION Network 10: SAFETY POSITION 3
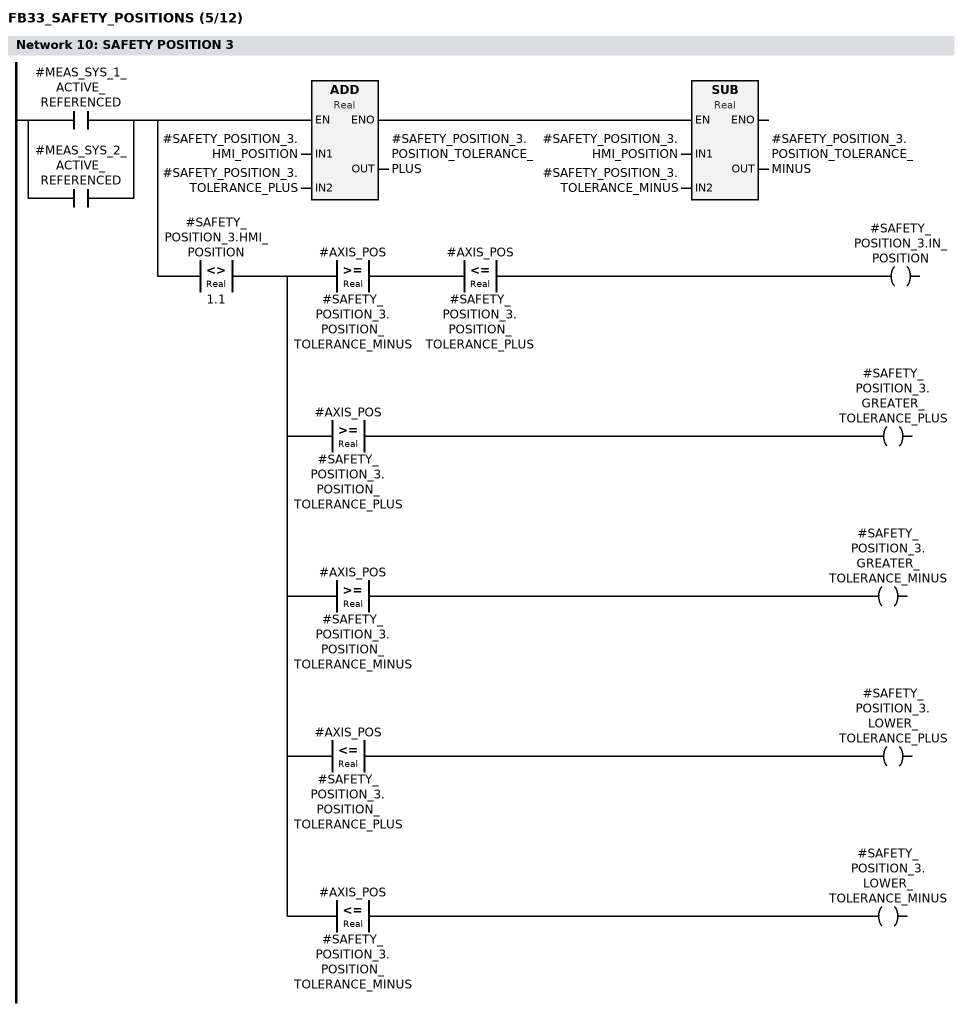
   RUNG wire#powerrail
      Contact( #MEAS_SYS_1_ACTIVE_REFERENCED )
      wire#w1
      { S7_Templates := "SrcType := Real"; S7_GenerateENO := "TRUE" } Add(in1 := #SAFETY_POSITION_3.HMI_POSITION, in2 := #SAFETY_POSITION_3.TOLERANCE_PLUS, out => #SAFETY_POSITION_3.POSITION_TOLERANCE_PLUS)
      { S7_Templates := "SrcType := Real"; S7_GenerateENO := "TRUE" } Sub(in1 := #SAFETY_POSITION_3.HMI_POSITION, in2 := #SAFETY_POSITION_3.TOLERANCE_MINUS, out => #SAFETY_POSITION_3.POSITION_TOLERANCE_MINUS)
   END_RUNG
   RUNG wire#powerrail
      Contact( #MEAS_SYS_2_ACTIVE_REFERENCED )
   END_RUNG wire#w1
   RUNG wire#w1
      { S7_Templates := "SrcType := Real" } NE_Contact(in1 := #SAFETY_POSITION_3.HMI_POSITION, in2 := 1.1)
      wire#w2
      { S7_Templates := "SrcType := Real" } GE_Contact(in1 := #AXIS_POS, in2 := #SAFETY_POSITION_3.POSITION_TOLERANCE_MINUS)
      { S7_Templates := "SrcType := Real" } LE_Contact(in1 := #AXIS_POS, in2 := #SAFETY_POSITION_3.POSITION_TOLERANCE_PLUS)
      Coil( #SAFETY_POSITION_3.IN_POSITION )
   END_RUNG
   RUNG wire#w2
      { S7_Templates := "SrcType := Real" } GE_Contact(in1 := #AXIS_POS, in2 := #SAFETY_POSITION_3.POSITION_TOLERANCE_PLUS)
      Coil( #SAFETY_POSITION_3.GREATER_TOLERANCE_PLUS )
   END_RUNG
   RUNG wire#w2
      { S7_Templates := "SrcType := Real" } GE_Contact(in1 := #AXIS_POS, in2 := #SAFETY_POSITION_3.POSITION_TOLERANCE_MINUS)
      Coil( #SAFETY_POSITION_3.GREATER_TOLERANCE_MINUS )
   END_RUNG
   RUNG wire#w2
      { S7_Templates := "SrcType := Real" } LE_Contact(in1 := #AXIS_POS, in2 := #SAFETY_POSITION_3.POSITION_TOLERANCE_PLUS)
      Coil( #SAFETY_POSITION_3.LOWER_TOLERANCE_PLUS )
   END_RUNG
   RUNG wire#w2
      { S7_Templates := "SrcType := Real" } LE_Contact(in1 := #AXIS_POS, in2 := #SAFETY_POSITION_3.POSITION_TOLERANCE_MINUS)
      Coil( #SAFETY_POSITION_3.LOWER_TOLERANCE_MINUS )
   END_RUNG
   // the same network as SCL:
   // ENO of a box is taken as its EN; it also drops when the box reports an error
   #_w1 := #MEAS_SYS_1_ACTIVE_REFERENCED OR #MEAS_SYS_2_ACTIVE_REFERENCED;
   IF #_w1 THEN
       #SAFETY_POSITION_3.POSITION_TOLERANCE_PLUS := #SAFETY_POSITION_3.HMI_POSITION + #SAFETY_POSITION_3.TOLERANCE_PLUS;
       #SAFETY_POSITION_3.POSITION_TOLERANCE_MINUS := #SAFETY_POSITION_3.HMI_POSITION - #SAFETY_POSITION_3.TOLERANCE_MINUS;
   END_IF;
   #_w2 := #_w1 AND (#SAFETY_POSITION_3.HMI_POSITION <> 1.1);
   #SAFETY_POSITION_3.IN_POSITION := #_w2 AND (#AXIS_POS >= #SAFETY_POSITION_3.POSITION_TOLERANCE_MINUS) AND (#AXIS_POS <= #SAFETY_POSITION_3.POSITION_TOLERANCE_PLUS);
   #SAFETY_POSITION_3.GREATER_TOLERANCE_PLUS := #_w2 AND (#AXIS_POS >= #SAFETY_POSITION_3.POSITION_TOLERANCE_PLUS);
   #SAFETY_POSITION_3.GREATER_TOLERANCE_MINUS := #_w2 AND (#AXIS_POS >= #SAFETY_POSITION_3.POSITION_TOLERANCE_MINUS);
   #SAFETY_POSITION_3.LOWER_TOLERANCE_PLUS := #_w2 AND (#AXIS_POS <= #SAFETY_POSITION_3.POSITION_TOLERANCE_PLUS);
   #SAFETY_POSITION_3.LOWER_TOLERANCE_MINUS := #_w2 AND (#AXIS_POS <= #SAFETY_POSITION_3.POSITION_TOLERANCE_MINUS);
END_REGION

REGION Network 11: SAFETY POSITION 4
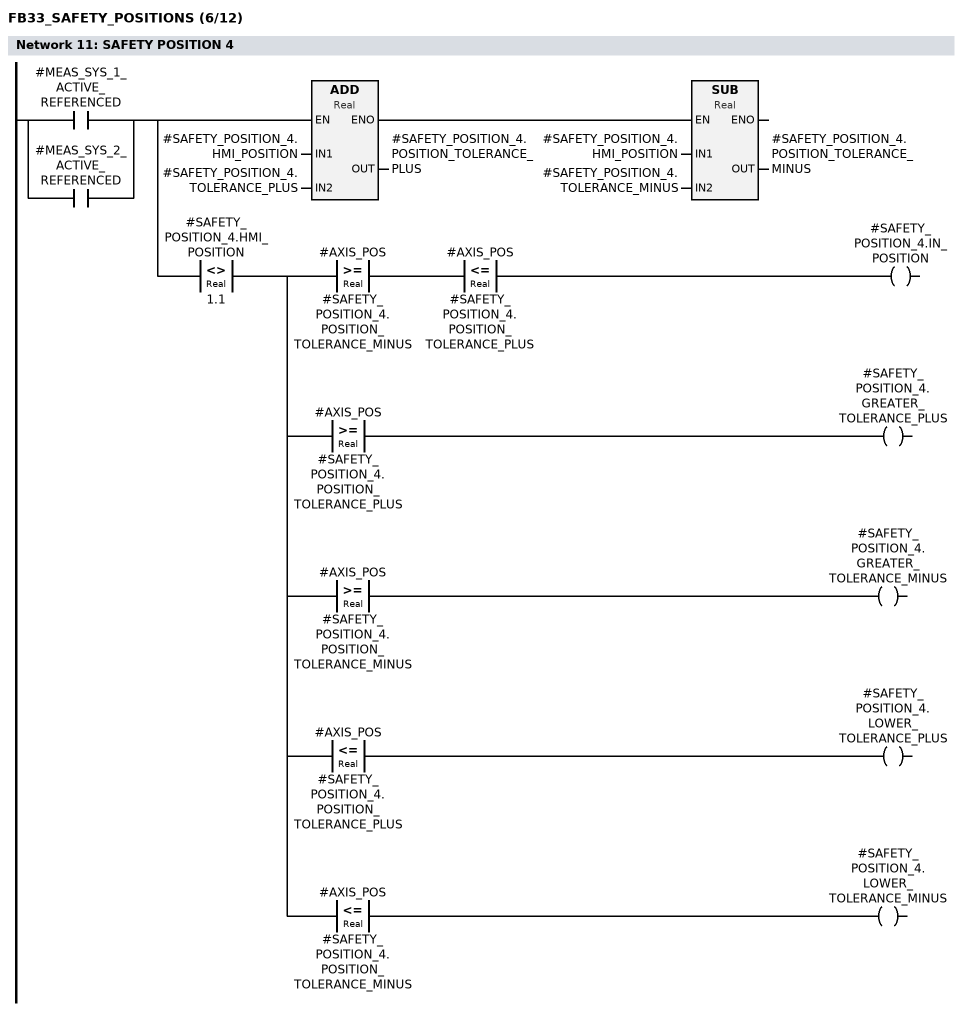
   RUNG wire#powerrail
      Contact( #MEAS_SYS_1_ACTIVE_REFERENCED )
      wire#w1
      { S7_Templates := "SrcType := Real"; S7_GenerateENO := "TRUE" } Add(in1 := #SAFETY_POSITION_4.HMI_POSITION, in2 := #SAFETY_POSITION_4.TOLERANCE_PLUS, out => #SAFETY_POSITION_4.POSITION_TOLERANCE_PLUS)
      { S7_Templates := "SrcType := Real"; S7_GenerateENO := "TRUE" } Sub(in1 := #SAFETY_POSITION_4.HMI_POSITION, in2 := #SAFETY_POSITION_4.TOLERANCE_MINUS, out => #SAFETY_POSITION_4.POSITION_TOLERANCE_MINUS)
   END_RUNG
   RUNG wire#powerrail
      Contact( #MEAS_SYS_2_ACTIVE_REFERENCED )
   END_RUNG wire#w1
   RUNG wire#w1
      { S7_Templates := "SrcType := Real" } NE_Contact(in1 := #SAFETY_POSITION_4.HMI_POSITION, in2 := 1.1)
      wire#w2
      { S7_Templates := "SrcType := Real" } GE_Contact(in1 := #AXIS_POS, in2 := #SAFETY_POSITION_4.POSITION_TOLERANCE_MINUS)
      { S7_Templates := "SrcType := Real" } LE_Contact(in1 := #AXIS_POS, in2 := #SAFETY_POSITION_4.POSITION_TOLERANCE_PLUS)
      Coil( #SAFETY_POSITION_4.IN_POSITION )
   END_RUNG
   RUNG wire#w2
      { S7_Templates := "SrcType := Real" } GE_Contact(in1 := #AXIS_POS, in2 := #SAFETY_POSITION_4.POSITION_TOLERANCE_PLUS)
      Coil( #SAFETY_POSITION_4.GREATER_TOLERANCE_PLUS )
   END_RUNG
   RUNG wire#w2
      { S7_Templates := "SrcType := Real" } GE_Contact(in1 := #AXIS_POS, in2 := #SAFETY_POSITION_4.POSITION_TOLERANCE_MINUS)
      Coil( #SAFETY_POSITION_4.GREATER_TOLERANCE_MINUS )
   END_RUNG
   RUNG wire#w2
      { S7_Templates := "SrcType := Real" } LE_Contact(in1 := #AXIS_POS, in2 := #SAFETY_POSITION_4.POSITION_TOLERANCE_PLUS)
      Coil( #SAFETY_POSITION_4.LOWER_TOLERANCE_PLUS )
   END_RUNG
   RUNG wire#w2
      { S7_Templates := "SrcType := Real" } LE_Contact(in1 := #AXIS_POS, in2 := #SAFETY_POSITION_4.POSITION_TOLERANCE_MINUS)
      Coil( #SAFETY_POSITION_4.LOWER_TOLERANCE_MINUS )
   END_RUNG
   // the same network as SCL:
   // ENO of a box is taken as its EN; it also drops when the box reports an error
   #_w1 := #MEAS_SYS_1_ACTIVE_REFERENCED OR #MEAS_SYS_2_ACTIVE_REFERENCED;
   IF #_w1 THEN
       #SAFETY_POSITION_4.POSITION_TOLERANCE_PLUS := #SAFETY_POSITION_4.HMI_POSITION + #SAFETY_POSITION_4.TOLERANCE_PLUS;
       #SAFETY_POSITION_4.POSITION_TOLERANCE_MINUS := #SAFETY_POSITION_4.HMI_POSITION - #SAFETY_POSITION_4.TOLERANCE_MINUS;
   END_IF;
   #_w2 := #_w1 AND (#SAFETY_POSITION_4.HMI_POSITION <> 1.1);
   #SAFETY_POSITION_4.IN_POSITION := #_w2 AND (#AXIS_POS >= #SAFETY_POSITION_4.POSITION_TOLERANCE_MINUS) AND (#AXIS_POS <= #SAFETY_POSITION_4.POSITION_TOLERANCE_PLUS);
   #SAFETY_POSITION_4.GREATER_TOLERANCE_PLUS := #_w2 AND (#AXIS_POS >= #SAFETY_POSITION_4.POSITION_TOLERANCE_PLUS);
   #SAFETY_POSITION_4.GREATER_TOLERANCE_MINUS := #_w2 AND (#AXIS_POS >= #SAFETY_POSITION_4.POSITION_TOLERANCE_MINUS);
   #SAFETY_POSITION_4.LOWER_TOLERANCE_PLUS := #_w2 AND (#AXIS_POS <= #SAFETY_POSITION_4.POSITION_TOLERANCE_PLUS);
   #SAFETY_POSITION_4.LOWER_TOLERANCE_MINUS := #_w2 AND (#AXIS_POS <= #SAFETY_POSITION_4.POSITION_TOLERANCE_MINUS);
END_REGION

REGION Network 12: SAFETY POSITION 5
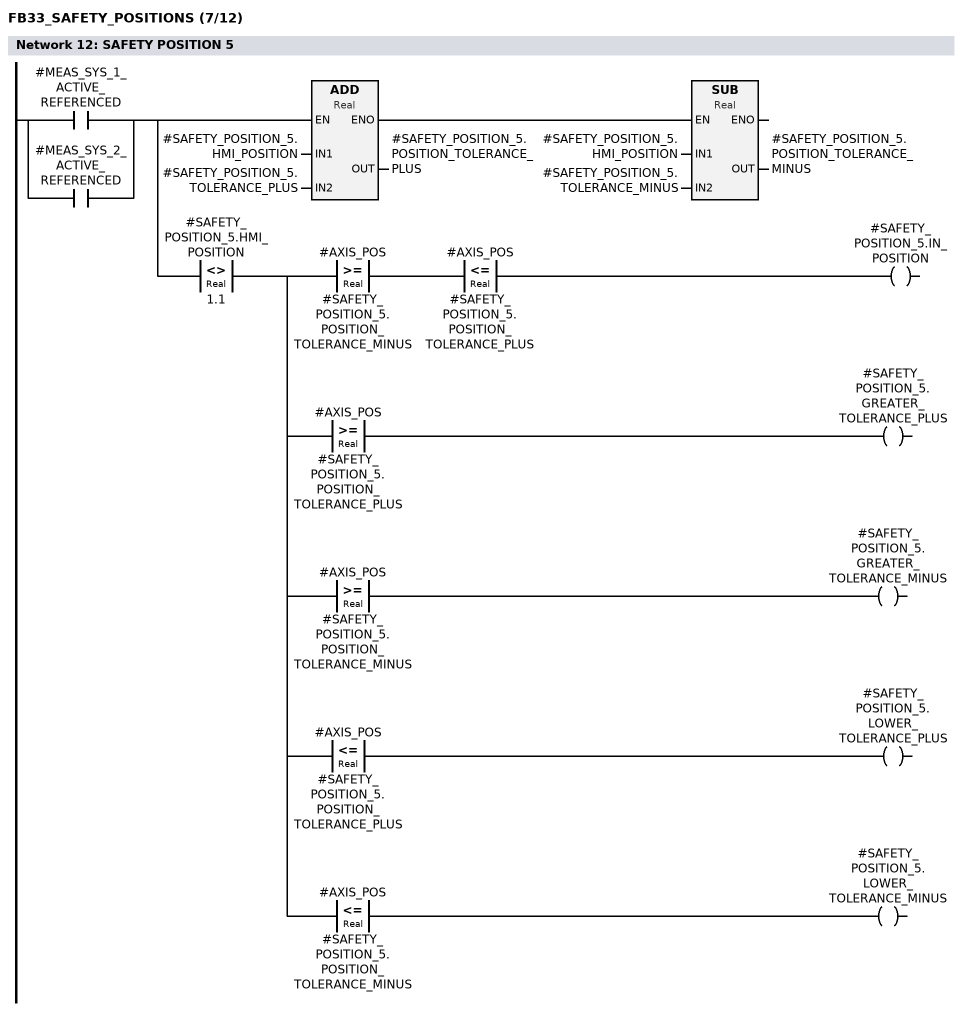
   RUNG wire#powerrail
      Contact( #MEAS_SYS_1_ACTIVE_REFERENCED )
      wire#w1
      { S7_Templates := "SrcType := Real"; S7_GenerateENO := "TRUE" } Add(in1 := #SAFETY_POSITION_5.HMI_POSITION, in2 := #SAFETY_POSITION_5.TOLERANCE_PLUS, out => #SAFETY_POSITION_5.POSITION_TOLERANCE_PLUS)
      { S7_Templates := "SrcType := Real"; S7_GenerateENO := "TRUE" } Sub(in1 := #SAFETY_POSITION_5.HMI_POSITION, in2 := #SAFETY_POSITION_5.TOLERANCE_MINUS, out => #SAFETY_POSITION_5.POSITION_TOLERANCE_MINUS)
   END_RUNG
   RUNG wire#powerrail
      Contact( #MEAS_SYS_2_ACTIVE_REFERENCED )
   END_RUNG wire#w1
   RUNG wire#w1
      { S7_Templates := "SrcType := Real" } NE_Contact(in1 := #SAFETY_POSITION_5.HMI_POSITION, in2 := 1.1)
      wire#w2
      { S7_Templates := "SrcType := Real" } GE_Contact(in1 := #AXIS_POS, in2 := #SAFETY_POSITION_5.POSITION_TOLERANCE_MINUS)
      { S7_Templates := "SrcType := Real" } LE_Contact(in1 := #AXIS_POS, in2 := #SAFETY_POSITION_5.POSITION_TOLERANCE_PLUS)
      Coil( #SAFETY_POSITION_5.IN_POSITION )
   END_RUNG
   RUNG wire#w2
      { S7_Templates := "SrcType := Real" } GE_Contact(in1 := #AXIS_POS, in2 := #SAFETY_POSITION_5.POSITION_TOLERANCE_PLUS)
      Coil( #SAFETY_POSITION_5.GREATER_TOLERANCE_PLUS )
   END_RUNG
   RUNG wire#w2
      { S7_Templates := "SrcType := Real" } GE_Contact(in1 := #AXIS_POS, in2 := #SAFETY_POSITION_5.POSITION_TOLERANCE_MINUS)
      Coil( #SAFETY_POSITION_5.GREATER_TOLERANCE_MINUS )
   END_RUNG
   RUNG wire#w2
      { S7_Templates := "SrcType := Real" } LE_Contact(in1 := #AXIS_POS, in2 := #SAFETY_POSITION_5.POSITION_TOLERANCE_PLUS)
      Coil( #SAFETY_POSITION_5.LOWER_TOLERANCE_PLUS )
   END_RUNG
   RUNG wire#w2
      { S7_Templates := "SrcType := Real" } LE_Contact(in1 := #AXIS_POS, in2 := #SAFETY_POSITION_5.POSITION_TOLERANCE_MINUS)
      Coil( #SAFETY_POSITION_5.LOWER_TOLERANCE_MINUS )
   END_RUNG
   // the same network as SCL:
   // ENO of a box is taken as its EN; it also drops when the box reports an error
   #_w1 := #MEAS_SYS_1_ACTIVE_REFERENCED OR #MEAS_SYS_2_ACTIVE_REFERENCED;
   IF #_w1 THEN
       #SAFETY_POSITION_5.POSITION_TOLERANCE_PLUS := #SAFETY_POSITION_5.HMI_POSITION + #SAFETY_POSITION_5.TOLERANCE_PLUS;
       #SAFETY_POSITION_5.POSITION_TOLERANCE_MINUS := #SAFETY_POSITION_5.HMI_POSITION - #SAFETY_POSITION_5.TOLERANCE_MINUS;
   END_IF;
   #_w2 := #_w1 AND (#SAFETY_POSITION_5.HMI_POSITION <> 1.1);
   #SAFETY_POSITION_5.IN_POSITION := #_w2 AND (#AXIS_POS >= #SAFETY_POSITION_5.POSITION_TOLERANCE_MINUS) AND (#AXIS_POS <= #SAFETY_POSITION_5.POSITION_TOLERANCE_PLUS);
   #SAFETY_POSITION_5.GREATER_TOLERANCE_PLUS := #_w2 AND (#AXIS_POS >= #SAFETY_POSITION_5.POSITION_TOLERANCE_PLUS);
   #SAFETY_POSITION_5.GREATER_TOLERANCE_MINUS := #_w2 AND (#AXIS_POS >= #SAFETY_POSITION_5.POSITION_TOLERANCE_MINUS);
   #SAFETY_POSITION_5.LOWER_TOLERANCE_PLUS := #_w2 AND (#AXIS_POS <= #SAFETY_POSITION_5.POSITION_TOLERANCE_PLUS);
   #SAFETY_POSITION_5.LOWER_TOLERANCE_MINUS := #_w2 AND (#AXIS_POS <= #SAFETY_POSITION_5.POSITION_TOLERANCE_MINUS);
END_REGION

REGION Network 13: SAFETY POSITION 6
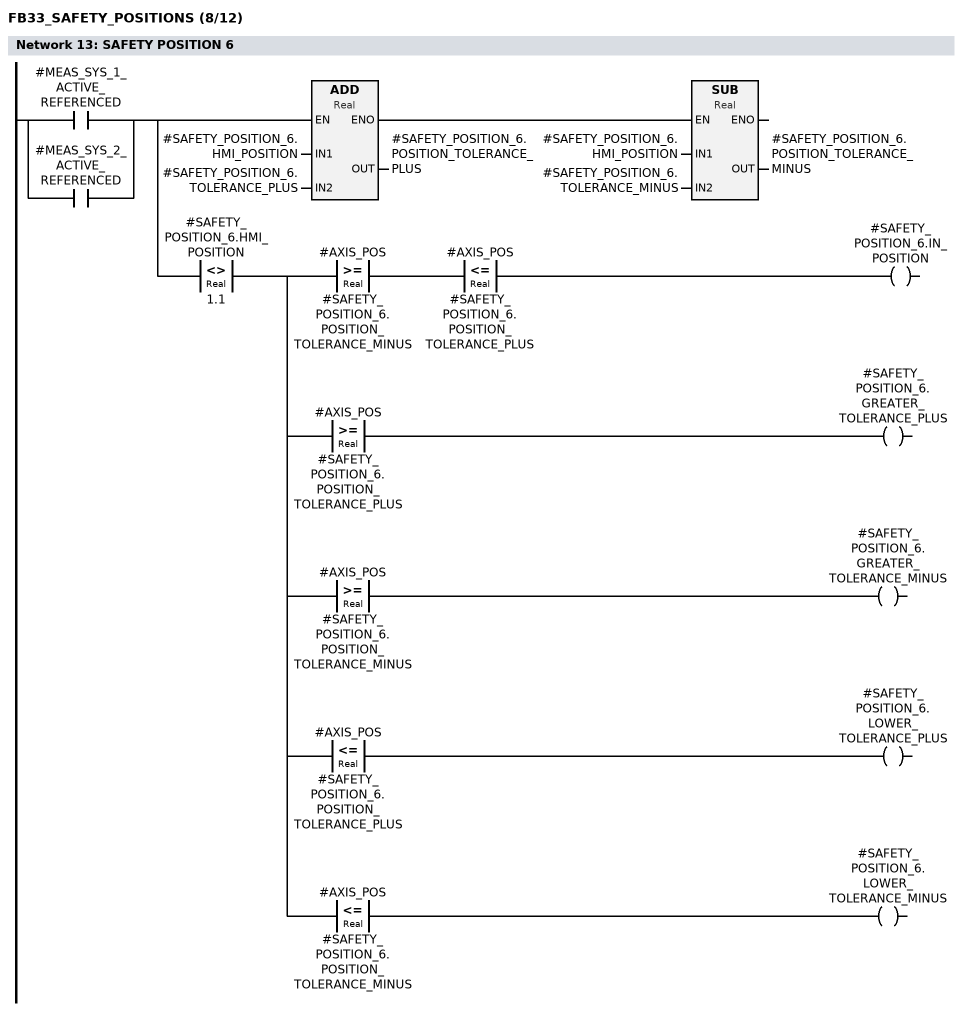
   RUNG wire#powerrail
      Contact( #MEAS_SYS_1_ACTIVE_REFERENCED )
      wire#w1
      { S7_Templates := "SrcType := Real"; S7_GenerateENO := "TRUE" } Add(in1 := #SAFETY_POSITION_6.HMI_POSITION, in2 := #SAFETY_POSITION_6.TOLERANCE_PLUS, out => #SAFETY_POSITION_6.POSITION_TOLERANCE_PLUS)
      { S7_Templates := "SrcType := Real"; S7_GenerateENO := "TRUE" } Sub(in1 := #SAFETY_POSITION_6.HMI_POSITION, in2 := #SAFETY_POSITION_6.TOLERANCE_MINUS, out => #SAFETY_POSITION_6.POSITION_TOLERANCE_MINUS)
   END_RUNG
   RUNG wire#powerrail
      Contact( #MEAS_SYS_2_ACTIVE_REFERENCED )
   END_RUNG wire#w1
   RUNG wire#w1
      { S7_Templates := "SrcType := Real" } NE_Contact(in1 := #SAFETY_POSITION_6.HMI_POSITION, in2 := 1.1)
      wire#w2
      { S7_Templates := "SrcType := Real" } GE_Contact(in1 := #AXIS_POS, in2 := #SAFETY_POSITION_6.POSITION_TOLERANCE_MINUS)
      { S7_Templates := "SrcType := Real" } LE_Contact(in1 := #AXIS_POS, in2 := #SAFETY_POSITION_6.POSITION_TOLERANCE_PLUS)
      Coil( #SAFETY_POSITION_6.IN_POSITION )
   END_RUNG
   RUNG wire#w2
      { S7_Templates := "SrcType := Real" } GE_Contact(in1 := #AXIS_POS, in2 := #SAFETY_POSITION_6.POSITION_TOLERANCE_PLUS)
      Coil( #SAFETY_POSITION_6.GREATER_TOLERANCE_PLUS )
   END_RUNG
   RUNG wire#w2
      { S7_Templates := "SrcType := Real" } GE_Contact(in1 := #AXIS_POS, in2 := #SAFETY_POSITION_6.POSITION_TOLERANCE_MINUS)
      Coil( #SAFETY_POSITION_6.GREATER_TOLERANCE_MINUS )
   END_RUNG
   RUNG wire#w2
      { S7_Templates := "SrcType := Real" } LE_Contact(in1 := #AXIS_POS, in2 := #SAFETY_POSITION_6.POSITION_TOLERANCE_PLUS)
      Coil( #SAFETY_POSITION_6.LOWER_TOLERANCE_PLUS )
   END_RUNG
   RUNG wire#w2
      { S7_Templates := "SrcType := Real" } LE_Contact(in1 := #AXIS_POS, in2 := #SAFETY_POSITION_6.POSITION_TOLERANCE_MINUS)
      Coil( #SAFETY_POSITION_6.LOWER_TOLERANCE_MINUS )
   END_RUNG
   // the same network as SCL:
   // ENO of a box is taken as its EN; it also drops when the box reports an error
   #_w1 := #MEAS_SYS_1_ACTIVE_REFERENCED OR #MEAS_SYS_2_ACTIVE_REFERENCED;
   IF #_w1 THEN
       #SAFETY_POSITION_6.POSITION_TOLERANCE_PLUS := #SAFETY_POSITION_6.HMI_POSITION + #SAFETY_POSITION_6.TOLERANCE_PLUS;
       #SAFETY_POSITION_6.POSITION_TOLERANCE_MINUS := #SAFETY_POSITION_6.HMI_POSITION - #SAFETY_POSITION_6.TOLERANCE_MINUS;
   END_IF;
   #_w2 := #_w1 AND (#SAFETY_POSITION_6.HMI_POSITION <> 1.1);
   #SAFETY_POSITION_6.IN_POSITION := #_w2 AND (#AXIS_POS >= #SAFETY_POSITION_6.POSITION_TOLERANCE_MINUS) AND (#AXIS_POS <= #SAFETY_POSITION_6.POSITION_TOLERANCE_PLUS);
   #SAFETY_POSITION_6.GREATER_TOLERANCE_PLUS := #_w2 AND (#AXIS_POS >= #SAFETY_POSITION_6.POSITION_TOLERANCE_PLUS);
   #SAFETY_POSITION_6.GREATER_TOLERANCE_MINUS := #_w2 AND (#AXIS_POS >= #SAFETY_POSITION_6.POSITION_TOLERANCE_MINUS);
   #SAFETY_POSITION_6.LOWER_TOLERANCE_PLUS := #_w2 AND (#AXIS_POS <= #SAFETY_POSITION_6.POSITION_TOLERANCE_PLUS);
   #SAFETY_POSITION_6.LOWER_TOLERANCE_MINUS := #_w2 AND (#AXIS_POS <= #SAFETY_POSITION_6.POSITION_TOLERANCE_MINUS);
END_REGION

REGION Network 14: SAFETY POSITION 7
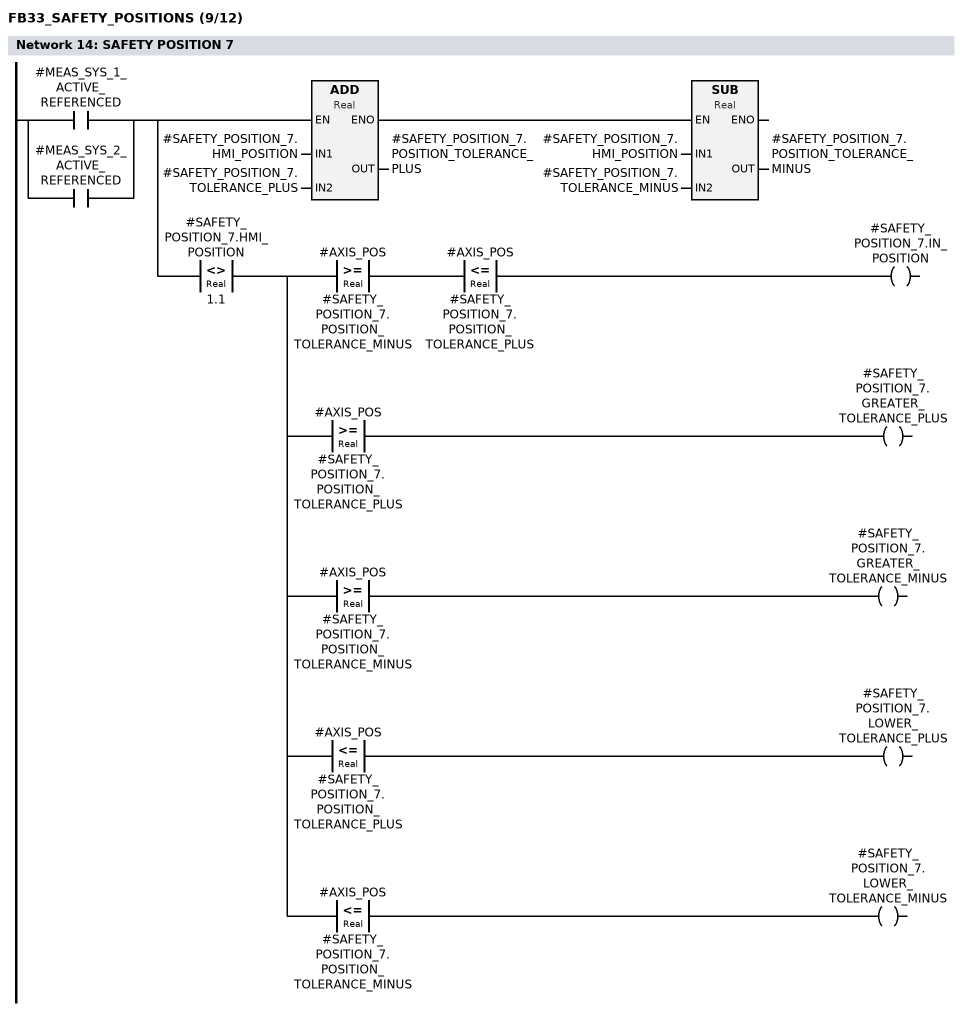
   RUNG wire#powerrail
      Contact( #MEAS_SYS_1_ACTIVE_REFERENCED )
      wire#w1
      { S7_Templates := "SrcType := Real"; S7_GenerateENO := "TRUE" } Add(in1 := #SAFETY_POSITION_7.HMI_POSITION, in2 := #SAFETY_POSITION_7.TOLERANCE_PLUS, out => #SAFETY_POSITION_7.POSITION_TOLERANCE_PLUS)
      { S7_Templates := "SrcType := Real"; S7_GenerateENO := "TRUE" } Sub(in1 := #SAFETY_POSITION_7.HMI_POSITION, in2 := #SAFETY_POSITION_7.TOLERANCE_MINUS, out => #SAFETY_POSITION_7.POSITION_TOLERANCE_MINUS)
   END_RUNG
   RUNG wire#powerrail
      Contact( #MEAS_SYS_2_ACTIVE_REFERENCED )
   END_RUNG wire#w1
   RUNG wire#w1
      { S7_Templates := "SrcType := Real" } NE_Contact(in1 := #SAFETY_POSITION_7.HMI_POSITION, in2 := 1.1)
      wire#w2
      { S7_Templates := "SrcType := Real" } GE_Contact(in1 := #AXIS_POS, in2 := #SAFETY_POSITION_7.POSITION_TOLERANCE_MINUS)
      { S7_Templates := "SrcType := Real" } LE_Contact(in1 := #AXIS_POS, in2 := #SAFETY_POSITION_7.POSITION_TOLERANCE_PLUS)
      Coil( #SAFETY_POSITION_7.IN_POSITION )
   END_RUNG
   RUNG wire#w2
      { S7_Templates := "SrcType := Real" } GE_Contact(in1 := #AXIS_POS, in2 := #SAFETY_POSITION_7.POSITION_TOLERANCE_PLUS)
      Coil( #SAFETY_POSITION_7.GREATER_TOLERANCE_PLUS )
   END_RUNG
   RUNG wire#w2
      { S7_Templates := "SrcType := Real" } GE_Contact(in1 := #AXIS_POS, in2 := #SAFETY_POSITION_7.POSITION_TOLERANCE_MINUS)
      Coil( #SAFETY_POSITION_7.GREATER_TOLERANCE_MINUS )
   END_RUNG
   RUNG wire#w2
      { S7_Templates := "SrcType := Real" } LE_Contact(in1 := #AXIS_POS, in2 := #SAFETY_POSITION_7.POSITION_TOLERANCE_PLUS)
      Coil( #SAFETY_POSITION_7.LOWER_TOLERANCE_PLUS )
   END_RUNG
   RUNG wire#w2
      { S7_Templates := "SrcType := Real" } LE_Contact(in1 := #AXIS_POS, in2 := #SAFETY_POSITION_7.POSITION_TOLERANCE_MINUS)
      Coil( #SAFETY_POSITION_7.LOWER_TOLERANCE_MINUS )
   END_RUNG
   // the same network as SCL:
   // ENO of a box is taken as its EN; it also drops when the box reports an error
   #_w1 := #MEAS_SYS_1_ACTIVE_REFERENCED OR #MEAS_SYS_2_ACTIVE_REFERENCED;
   IF #_w1 THEN
       #SAFETY_POSITION_7.POSITION_TOLERANCE_PLUS := #SAFETY_POSITION_7.HMI_POSITION + #SAFETY_POSITION_7.TOLERANCE_PLUS;
       #SAFETY_POSITION_7.POSITION_TOLERANCE_MINUS := #SAFETY_POSITION_7.HMI_POSITION - #SAFETY_POSITION_7.TOLERANCE_MINUS;
   END_IF;
   #_w2 := #_w1 AND (#SAFETY_POSITION_7.HMI_POSITION <> 1.1);
   #SAFETY_POSITION_7.IN_POSITION := #_w2 AND (#AXIS_POS >= #SAFETY_POSITION_7.POSITION_TOLERANCE_MINUS) AND (#AXIS_POS <= #SAFETY_POSITION_7.POSITION_TOLERANCE_PLUS);
   #SAFETY_POSITION_7.GREATER_TOLERANCE_PLUS := #_w2 AND (#AXIS_POS >= #SAFETY_POSITION_7.POSITION_TOLERANCE_PLUS);
   #SAFETY_POSITION_7.GREATER_TOLERANCE_MINUS := #_w2 AND (#AXIS_POS >= #SAFETY_POSITION_7.POSITION_TOLERANCE_MINUS);
   #SAFETY_POSITION_7.LOWER_TOLERANCE_PLUS := #_w2 AND (#AXIS_POS <= #SAFETY_POSITION_7.POSITION_TOLERANCE_PLUS);
   #SAFETY_POSITION_7.LOWER_TOLERANCE_MINUS := #_w2 AND (#AXIS_POS <= #SAFETY_POSITION_7.POSITION_TOLERANCE_MINUS);
END_REGION

REGION Network 15: SAFETY POSITION 8
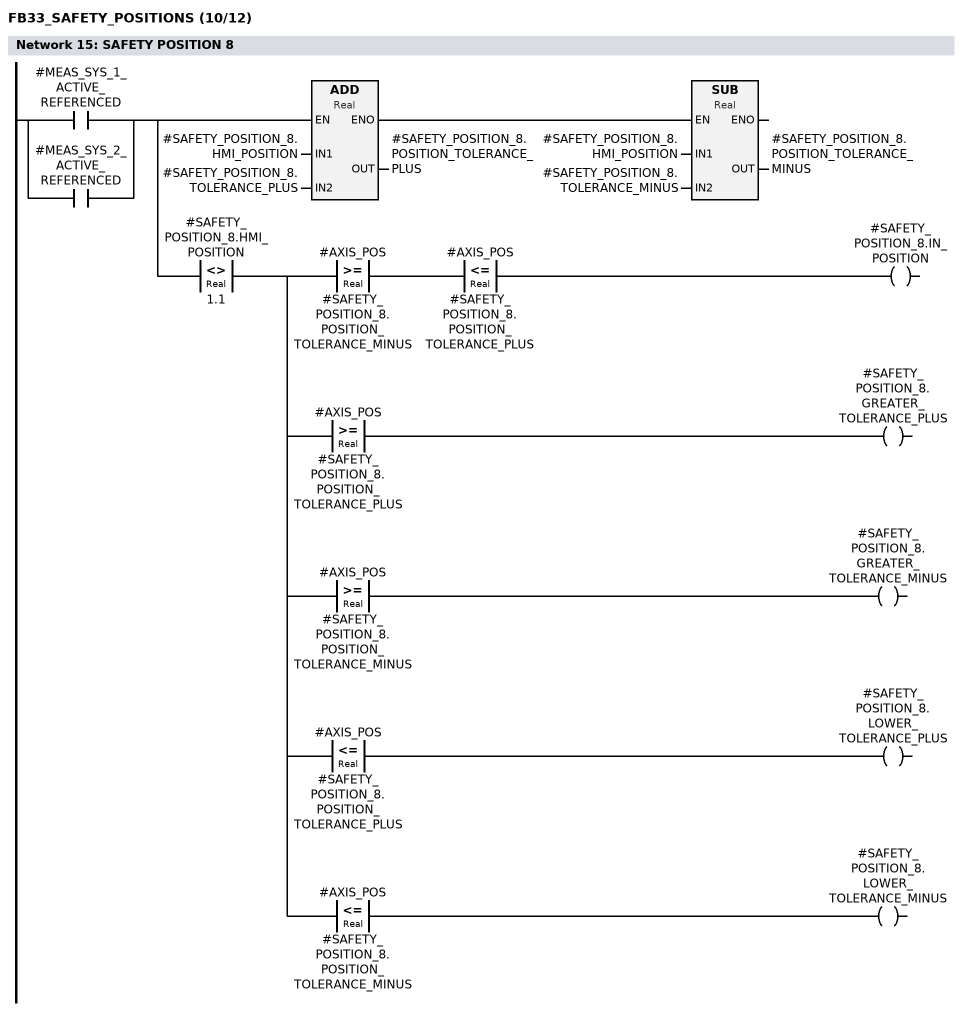
   RUNG wire#powerrail
      Contact( #MEAS_SYS_1_ACTIVE_REFERENCED )
      wire#w1
      { S7_Templates := "SrcType := Real"; S7_GenerateENO := "TRUE" } Add(in1 := #SAFETY_POSITION_8.HMI_POSITION, in2 := #SAFETY_POSITION_8.TOLERANCE_PLUS, out => #SAFETY_POSITION_8.POSITION_TOLERANCE_PLUS)
      { S7_Templates := "SrcType := Real"; S7_GenerateENO := "TRUE" } Sub(in1 := #SAFETY_POSITION_8.HMI_POSITION, in2 := #SAFETY_POSITION_8.TOLERANCE_MINUS, out => #SAFETY_POSITION_8.POSITION_TOLERANCE_MINUS)
   END_RUNG
   RUNG wire#powerrail
      Contact( #MEAS_SYS_2_ACTIVE_REFERENCED )
   END_RUNG wire#w1
   RUNG wire#w1
      { S7_Templates := "SrcType := Real" } NE_Contact(in1 := #SAFETY_POSITION_8.HMI_POSITION, in2 := 1.1)
      wire#w2
      { S7_Templates := "SrcType := Real" } GE_Contact(in1 := #AXIS_POS, in2 := #SAFETY_POSITION_8.POSITION_TOLERANCE_MINUS)
      { S7_Templates := "SrcType := Real" } LE_Contact(in1 := #AXIS_POS, in2 := #SAFETY_POSITION_8.POSITION_TOLERANCE_PLUS)
      Coil( #SAFETY_POSITION_8.IN_POSITION )
   END_RUNG
   RUNG wire#w2
      { S7_Templates := "SrcType := Real" } GE_Contact(in1 := #AXIS_POS, in2 := #SAFETY_POSITION_8.POSITION_TOLERANCE_PLUS)
      Coil( #SAFETY_POSITION_8.GREATER_TOLERANCE_PLUS )
   END_RUNG
   RUNG wire#w2
      { S7_Templates := "SrcType := Real" } GE_Contact(in1 := #AXIS_POS, in2 := #SAFETY_POSITION_8.POSITION_TOLERANCE_MINUS)
      Coil( #SAFETY_POSITION_8.GREATER_TOLERANCE_MINUS )
   END_RUNG
   RUNG wire#w2
      { S7_Templates := "SrcType := Real" } LE_Contact(in1 := #AXIS_POS, in2 := #SAFETY_POSITION_8.POSITION_TOLERANCE_PLUS)
      Coil( #SAFETY_POSITION_8.LOWER_TOLERANCE_PLUS )
   END_RUNG
   RUNG wire#w2
      { S7_Templates := "SrcType := Real" } LE_Contact(in1 := #AXIS_POS, in2 := #SAFETY_POSITION_8.POSITION_TOLERANCE_MINUS)
      Coil( #SAFETY_POSITION_8.LOWER_TOLERANCE_MINUS )
   END_RUNG
   // the same network as SCL:
   // ENO of a box is taken as its EN; it also drops when the box reports an error
   #_w1 := #MEAS_SYS_1_ACTIVE_REFERENCED OR #MEAS_SYS_2_ACTIVE_REFERENCED;
   IF #_w1 THEN
       #SAFETY_POSITION_8.POSITION_TOLERANCE_PLUS := #SAFETY_POSITION_8.HMI_POSITION + #SAFETY_POSITION_8.TOLERANCE_PLUS;
       #SAFETY_POSITION_8.POSITION_TOLERANCE_MINUS := #SAFETY_POSITION_8.HMI_POSITION - #SAFETY_POSITION_8.TOLERANCE_MINUS;
   END_IF;
   #_w2 := #_w1 AND (#SAFETY_POSITION_8.HMI_POSITION <> 1.1);
   #SAFETY_POSITION_8.IN_POSITION := #_w2 AND (#AXIS_POS >= #SAFETY_POSITION_8.POSITION_TOLERANCE_MINUS) AND (#AXIS_POS <= #SAFETY_POSITION_8.POSITION_TOLERANCE_PLUS);
   #SAFETY_POSITION_8.GREATER_TOLERANCE_PLUS := #_w2 AND (#AXIS_POS >= #SAFETY_POSITION_8.POSITION_TOLERANCE_PLUS);
   #SAFETY_POSITION_8.GREATER_TOLERANCE_MINUS := #_w2 AND (#AXIS_POS >= #SAFETY_POSITION_8.POSITION_TOLERANCE_MINUS);
   #SAFETY_POSITION_8.LOWER_TOLERANCE_PLUS := #_w2 AND (#AXIS_POS <= #SAFETY_POSITION_8.POSITION_TOLERANCE_PLUS);
   #SAFETY_POSITION_8.LOWER_TOLERANCE_MINUS := #_w2 AND (#AXIS_POS <= #SAFETY_POSITION_8.POSITION_TOLERANCE_MINUS);
END_REGION

REGION Network 16: SAFETY POSITION 9
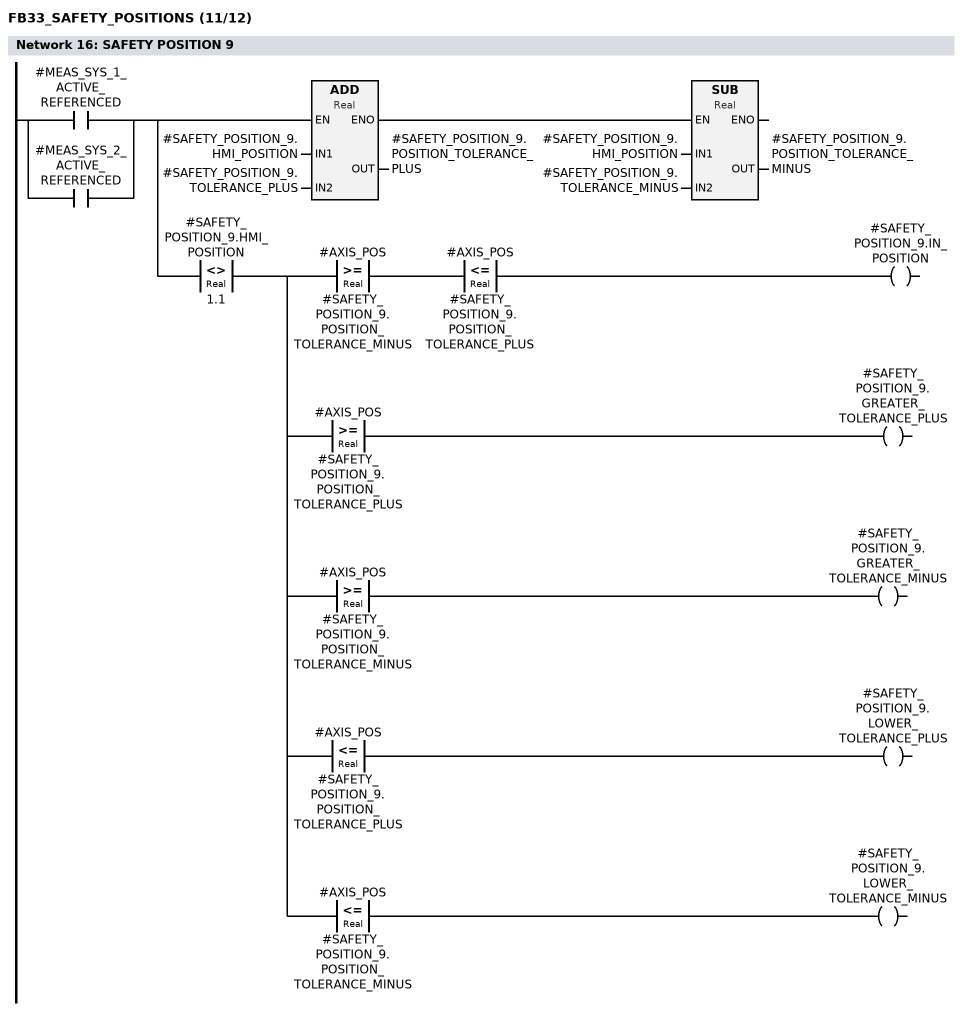
   RUNG wire#powerrail
      Contact( #MEAS_SYS_1_ACTIVE_REFERENCED )
      wire#w1
      { S7_Templates := "SrcType := Real"; S7_GenerateENO := "TRUE" } Add(in1 := #SAFETY_POSITION_9.HMI_POSITION, in2 := #SAFETY_POSITION_9.TOLERANCE_PLUS, out => #SAFETY_POSITION_9.POSITION_TOLERANCE_PLUS)
      { S7_Templates := "SrcType := Real"; S7_GenerateENO := "TRUE" } Sub(in1 := #SAFETY_POSITION_9.HMI_POSITION, in2 := #SAFETY_POSITION_9.TOLERANCE_MINUS, out => #SAFETY_POSITION_9.POSITION_TOLERANCE_MINUS)
   END_RUNG
   RUNG wire#powerrail
      Contact( #MEAS_SYS_2_ACTIVE_REFERENCED )
   END_RUNG wire#w1
   RUNG wire#w1
      { S7_Templates := "SrcType := Real" } NE_Contact(in1 := #SAFETY_POSITION_9.HMI_POSITION, in2 := 1.1)
      wire#w2
      { S7_Templates := "SrcType := Real" } GE_Contact(in1 := #AXIS_POS, in2 := #SAFETY_POSITION_9.POSITION_TOLERANCE_MINUS)
      { S7_Templates := "SrcType := Real" } LE_Contact(in1 := #AXIS_POS, in2 := #SAFETY_POSITION_9.POSITION_TOLERANCE_PLUS)
      Coil( #SAFETY_POSITION_9.IN_POSITION )
   END_RUNG
   RUNG wire#w2
      { S7_Templates := "SrcType := Real" } GE_Contact(in1 := #AXIS_POS, in2 := #SAFETY_POSITION_9.POSITION_TOLERANCE_PLUS)
      Coil( #SAFETY_POSITION_9.GREATER_TOLERANCE_PLUS )
   END_RUNG
   RUNG wire#w2
      { S7_Templates := "SrcType := Real" } GE_Contact(in1 := #AXIS_POS, in2 := #SAFETY_POSITION_9.POSITION_TOLERANCE_MINUS)
      Coil( #SAFETY_POSITION_9.GREATER_TOLERANCE_MINUS )
   END_RUNG
   RUNG wire#w2
      { S7_Templates := "SrcType := Real" } LE_Contact(in1 := #AXIS_POS, in2 := #SAFETY_POSITION_9.POSITION_TOLERANCE_PLUS)
      Coil( #SAFETY_POSITION_9.LOWER_TOLERANCE_PLUS )
   END_RUNG
   RUNG wire#w2
      { S7_Templates := "SrcType := Real" } LE_Contact(in1 := #AXIS_POS, in2 := #SAFETY_POSITION_9.POSITION_TOLERANCE_MINUS)
      Coil( #SAFETY_POSITION_9.LOWER_TOLERANCE_MINUS )
   END_RUNG
   // the same network as SCL:
   // ENO of a box is taken as its EN; it also drops when the box reports an error
   #_w1 := #MEAS_SYS_1_ACTIVE_REFERENCED OR #MEAS_SYS_2_ACTIVE_REFERENCED;
   IF #_w1 THEN
       #SAFETY_POSITION_9.POSITION_TOLERANCE_PLUS := #SAFETY_POSITION_9.HMI_POSITION + #SAFETY_POSITION_9.TOLERANCE_PLUS;
       #SAFETY_POSITION_9.POSITION_TOLERANCE_MINUS := #SAFETY_POSITION_9.HMI_POSITION - #SAFETY_POSITION_9.TOLERANCE_MINUS;
   END_IF;
   #_w2 := #_w1 AND (#SAFETY_POSITION_9.HMI_POSITION <> 1.1);
   #SAFETY_POSITION_9.IN_POSITION := #_w2 AND (#AXIS_POS >= #SAFETY_POSITION_9.POSITION_TOLERANCE_MINUS) AND (#AXIS_POS <= #SAFETY_POSITION_9.POSITION_TOLERANCE_PLUS);
   #SAFETY_POSITION_9.GREATER_TOLERANCE_PLUS := #_w2 AND (#AXIS_POS >= #SAFETY_POSITION_9.POSITION_TOLERANCE_PLUS);
   #SAFETY_POSITION_9.GREATER_TOLERANCE_MINUS := #_w2 AND (#AXIS_POS >= #SAFETY_POSITION_9.POSITION_TOLERANCE_MINUS);
   #SAFETY_POSITION_9.LOWER_TOLERANCE_PLUS := #_w2 AND (#AXIS_POS <= #SAFETY_POSITION_9.POSITION_TOLERANCE_PLUS);
   #SAFETY_POSITION_9.LOWER_TOLERANCE_MINUS := #_w2 AND (#AXIS_POS <= #SAFETY_POSITION_9.POSITION_TOLERANCE_MINUS);
END_REGION

REGION Network 17: SAFETY POSITION 10
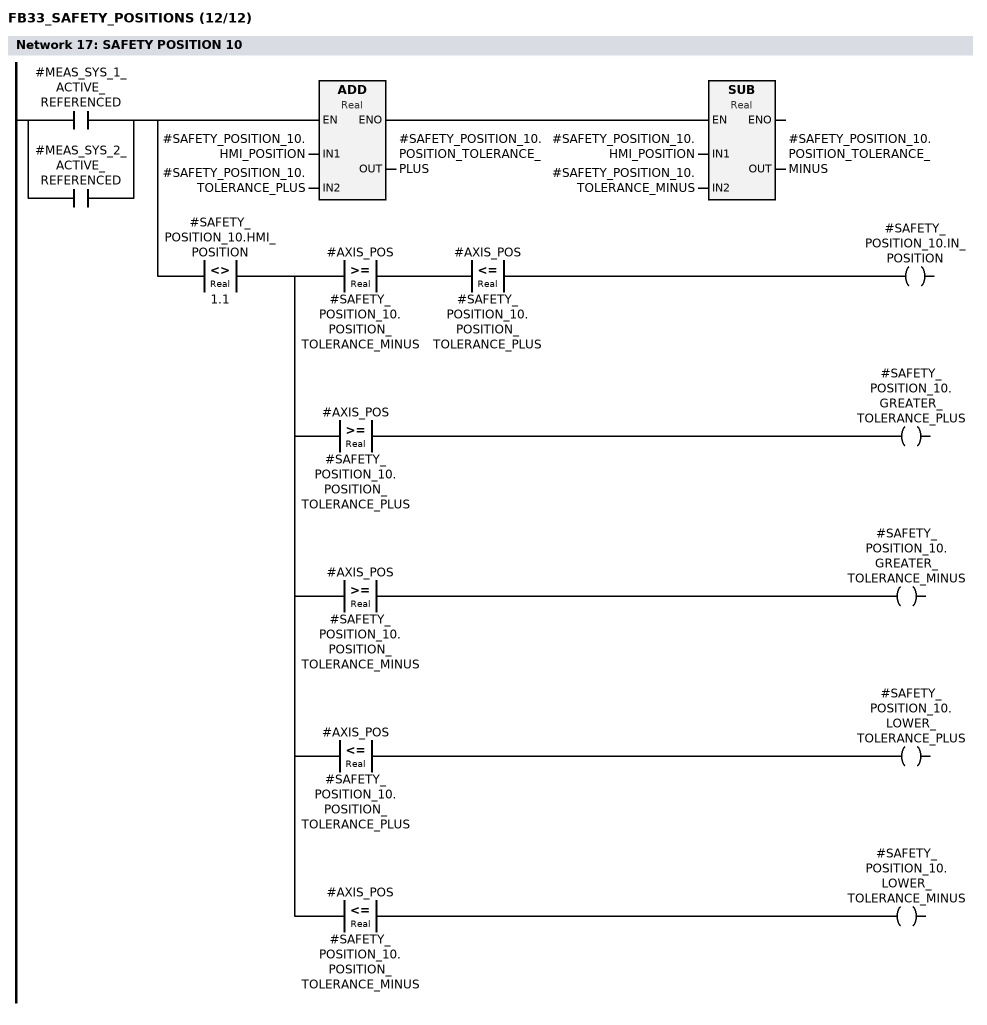
   RUNG wire#powerrail
      Contact( #MEAS_SYS_1_ACTIVE_REFERENCED )
      wire#w1
      { S7_Templates := "SrcType := Real"; S7_GenerateENO := "TRUE" } Add(in1 := #SAFETY_POSITION_10.HMI_POSITION, in2 := #SAFETY_POSITION_10.TOLERANCE_PLUS, out => #SAFETY_POSITION_10.POSITION_TOLERANCE_PLUS)
      { S7_Templates := "SrcType := Real"; S7_GenerateENO := "TRUE" } Sub(in1 := #SAFETY_POSITION_10.HMI_POSITION, in2 := #SAFETY_POSITION_10.TOLERANCE_MINUS, out => #SAFETY_POSITION_10.POSITION_TOLERANCE_MINUS)
   END_RUNG
   RUNG wire#powerrail
      Contact( #MEAS_SYS_2_ACTIVE_REFERENCED )
   END_RUNG wire#w1
   RUNG wire#w1
      { S7_Templates := "SrcType := Real" } NE_Contact(in1 := #SAFETY_POSITION_10.HMI_POSITION, in2 := 1.1)
      wire#w2
      { S7_Templates := "SrcType := Real" } GE_Contact(in1 := #AXIS_POS, in2 := #SAFETY_POSITION_10.POSITION_TOLERANCE_MINUS)
      { S7_Templates := "SrcType := Real" } LE_Contact(in1 := #AXIS_POS, in2 := #SAFETY_POSITION_10.POSITION_TOLERANCE_PLUS)
      Coil( #SAFETY_POSITION_10.IN_POSITION )
   END_RUNG
   RUNG wire#w2
      { S7_Templates := "SrcType := Real" } GE_Contact(in1 := #AXIS_POS, in2 := #SAFETY_POSITION_10.POSITION_TOLERANCE_PLUS)
      Coil( #SAFETY_POSITION_10.GREATER_TOLERANCE_PLUS )
   END_RUNG
   RUNG wire#w2
      { S7_Templates := "SrcType := Real" } GE_Contact(in1 := #AXIS_POS, in2 := #SAFETY_POSITION_10.POSITION_TOLERANCE_MINUS)
      Coil( #SAFETY_POSITION_10.GREATER_TOLERANCE_MINUS )
   END_RUNG
   RUNG wire#w2
      { S7_Templates := "SrcType := Real" } LE_Contact(in1 := #AXIS_POS, in2 := #SAFETY_POSITION_10.POSITION_TOLERANCE_PLUS)
      Coil( #SAFETY_POSITION_10.LOWER_TOLERANCE_PLUS )
   END_RUNG
   RUNG wire#w2
      { S7_Templates := "SrcType := Real" } LE_Contact(in1 := #AXIS_POS, in2 := #SAFETY_POSITION_10.POSITION_TOLERANCE_MINUS)
      Coil( #SAFETY_POSITION_10.LOWER_TOLERANCE_MINUS )
   END_RUNG
   // the same network as SCL:
   // ENO of a box is taken as its EN; it also drops when the box reports an error
   #_w1 := #MEAS_SYS_1_ACTIVE_REFERENCED OR #MEAS_SYS_2_ACTIVE_REFERENCED;
   IF #_w1 THEN
       #SAFETY_POSITION_10.POSITION_TOLERANCE_PLUS := #SAFETY_POSITION_10.HMI_POSITION + #SAFETY_POSITION_10.TOLERANCE_PLUS;
       #SAFETY_POSITION_10.POSITION_TOLERANCE_MINUS := #SAFETY_POSITION_10.HMI_POSITION - #SAFETY_POSITION_10.TOLERANCE_MINUS;
   END_IF;
   #_w2 := #_w1 AND (#SAFETY_POSITION_10.HMI_POSITION <> 1.1);
   #SAFETY_POSITION_10.IN_POSITION := #_w2 AND (#AXIS_POS >= #SAFETY_POSITION_10.POSITION_TOLERANCE_MINUS) AND (#AXIS_POS <= #SAFETY_POSITION_10.POSITION_TOLERANCE_PLUS);
   #SAFETY_POSITION_10.GREATER_TOLERANCE_PLUS := #_w2 AND (#AXIS_POS >= #SAFETY_POSITION_10.POSITION_TOLERANCE_PLUS);
   #SAFETY_POSITION_10.GREATER_TOLERANCE_MINUS := #_w2 AND (#AXIS_POS >= #SAFETY_POSITION_10.POSITION_TOLERANCE_MINUS);
   #SAFETY_POSITION_10.LOWER_TOLERANCE_PLUS := #_w2 AND (#AXIS_POS <= #SAFETY_POSITION_10.POSITION_TOLERANCE_PLUS);
   #SAFETY_POSITION_10.LOWER_TOLERANCE_MINUS := #_w2 AND (#AXIS_POS <= #SAFETY_POSITION_10.POSITION_TOLERANCE_MINUS);
END_REGION
END_FUNCTION_BLOCK

